IF DSA31ArmSpeedProfileCall.bCallCompleted THEN
DSA31ArmSpeedProfileCall.bCallPB := FALSE;
DSfbGnrProductRecipeMemoryOut.DSGnrCalledArmPnpParameter.DSA1DownTransferMovement.lrZone2SpeedVelo := DSA31ArmSpeedProfileCall.Call_DSArmSpdProfile.lrSpeedVelo;
DSfbGnrProductRecipeMemoryOut.DSGnrCalledArmPnpParameter.DSA1DownTransferMovement.lrZone2Acc := DSA31ArmSpeedProfileCall.Call_DSArmSpdProfile.lrAcc;
DSfbGnrProductRecipeMemoryOut.DSGnrCalledArmPnpParameter.DSA1DownTransferMovement.lrZone2Dcc := DSA31ArmSpeedProfileCall.Call_DSArmSpdProfile.lrDcc;

DSfbGnrProductRecipeMemoryOut.iCallCaseNo:=43;
END_IF

IF rebInvalidSpeedProfileMemoryCall.Q THEN
DSA31ArmSpeedProfileCall.bCallPB := FALSE;

DSfbGnrProductRecipeMemoryOut.iCallCaseNo:=82;
END_IF


41: (* Push DownTransfer Zone1  Velo/Acc/Dcc to DownTransfer Movement*)

DSA31ArmSpeedProfileCall.Call_iArmSpdProfile := DSBufferDownTransferPattern.iZone1SpdProfileNo;
DSA31ArmSpeedProfileCall.bCallPB := TRUE;


IF DSA31ArmSpeedProfileCall.bCallCompleted THEN
DSA31ArmSpeedProfileCall.bCallPB := FALSE;
DSfbGnrProductRecipeMemoryOut.DSGnrCalledArmPnpParameter.DSA1DownTransferMovement.lrZone1SpeedVelo := DSA31ArmSpeedProfileCall.Call_DSArmSpdProfile.lrSpeedVelo;
DSfbGnrProductRecipeMemoryOut.DSGnrCalledArmPnpParameter.DSA1DownTransferMovement.lrZone1Acc := DSA31ArmSpeedProfileCall.Call_DSArmSpdProfile.lrAcc;
DSfbGnrProductRecipeMemoryOut.DSGnrCalledArmPnpParameter.DSA1DownTransferMovement.lrZone1Dcc := DSA31ArmSpeedProfileCall.Call_DSArmSpdProfile.lrDcc;

DSfbGnrProductRecipeMemoryOut.iCallCaseNo:=42;
END_IF

IF rebInvalidSpeedProfileMemoryCall.Q THEN
DSA31ArmSpeedProfileCall.bCallPB := FALSE;

DSfbGnrProductRecipeMemoryOut.iCallCaseNo:=82;
END_IF

(*[][][][][][][][][][][][][][][][][][][][][][][][][][][][][][][][][][][][][][][][][][][][][][][][][][][][][][][][][][][][][][][][][][][][][][][][][][][][][][][][][][][][][][][][][][][][][][][][][][][]*)

(*[][][][][][][][][][][][][][][][][][][][][][][][][][][][][][][][][][][][][][][][][][][][][][][][][][][][][][][][][][][][][][][][][][][][][][][][][][][][][][][][][][][][][][][][][][][][][][][][][][][]*)
34: (* Push UpPick Zone4  Velo/Acc/Dcc to UpPick Movement*)

DSA31ArmSpeedProfileCall.Call_iArmSpdProfile := DSBufferUpPickPattern.iZone4SpdProfileNo;
DSA31ArmSpeedProfileCall.bCallPB := TRUE;


IF DSA31ArmSpeedProfileCall.bCallCompleted THEN
DSA31ArmSpeedProfileCall.bCallPB := FALSE;
DSfbGnrProductRecipeMemoryOut.DSGnrCalledArmPnpParameter.DSA1UpPickMovement.lrZone4SpeedVelo := DSA31ArmSpeedProfileCall.Call_DSArmSpdProfile.lrSpeedVelo;
DSfbGnrProductRecipeMemoryOut.DSGnrCalledArmPnpParameter.DSA1UpPickMovement.lrZone4Acc := DSA31ArmSpeedProfileCall.Call_DSArmSpdProfile.lrAcc;
DSfbGnrProductRecipeMemoryOut.DSGnrCalledArmPnpParameter.DSA1UpPickMovement.lrZone4Dcc := DSA31ArmSpeedProfileCall.Call_DSArmSpdProfile.lrDcc;

DSfbGnrProductRecipeMemoryOut.iCallCaseNo:=41;
END_IF

IF rebInvalidSpeedProfileMemoryCall.Q THEN
DSA31ArmSpeedProfileCall.bCallPB := FALSE;

DSfbGnrProductRecipeMemoryOut.iCallCaseNo:=82;
END_IF



33: (* Push UpPick Zone3  Velo/Acc/Dcc to UpPick Movement*)

DSA31ArmSpeedProfileCall.Call_iArmSpdProfile := DSBufferUpPickPattern.iZone3SpdProfileNo;
DSA31ArmSpeedProfileCall.bCallPB := TRUE;


IF DSA31ArmSpeedProfileCall.bCallCompleted THEN
DSA31ArmSpeedProfileCall.bCallPB := FALSE;
DSfbGnrProductRecipeMemoryOut.DSGnrCalledArmPnpParameter.DSA1UpPickMovement.lrZone3SpeedVelo := DSA31ArmSpeedProfileCall.Call_DSArmSpdProfile.lrSpeedVelo;
DSfbGnrProductRecipeMemoryOut.DSGnrCalledArmPnpParameter.DSA1UpPickMovement.lrZone3Acc := DSA31ArmSpeedProfileCall.Call_DSArmSpdProfile.lrAcc;
DSfbGnrProductRecipeMemoryOut.DSGnrCalledArmPnpParameter.DSA1UpPickMovement.lrZone3Dcc := DSA31ArmSpeedProfileCall.Call_DSArmSpdProfile.lrDcc;

DSfbGnrProductRecipeMemoryOut.iCallCaseNo:=34;
END_IF

IF rebInvalidSpeedProfileMemoryCall.Q THEN
DSA31ArmSpeedProfileCall.bCallPB := FALSE;

DSfbGnrProductRecipeMemoryOut.iCallCaseNo:=82;
END_IF



32: (* Push UpPick Zone2  Velo/Acc/Dcc to UpPick Movement*)

DSA31ArmSpeedProfileCall.Call_iArmSpdProfile := DSBufferUpPickPattern.iZone2SpdProfileNo;
DSA31ArmSpeedProfileCall.bCallPB := TRUE;


IF DSA31ArmSpeedProfileCall.bCallCompleted THEN
DSA31ArmSpeedProfileCall.bCallPB := FALSE;
DSfbGnrProductRecipeMemoryOut.DSGnrCalledArmPnpParameter.DSA1UpPickMovement.lrZone2SpeedVelo := DSA31ArmSpeedProfileCall.Call_DSArmSpdProfile.lrSpeedVelo;
DSfbGnrProductRecipeMemoryOut.DSGnrCalledArmPnpParameter.DSA1UpPickMovement.lrZone2Acc := DSA31ArmSpeedProfileCall.Call_DSArmSpdProfile.lrAcc;
DSfbGnrProductRecipeMemoryOut.DSGnrCalledArmPnpParameter.DSA1UpPickMovement.lrZone2Dcc := DSA31ArmSpeedProfileCall.Call_DSArmSpdProfile.lrDcc;

DSfbGnrProductRecipeMemoryOut.iCallCaseNo:=33;
END_IF

IF rebInvalidSpeedProfileMemoryCall.Q THEN
DSA31ArmSpeedProfileCall.bCallPB := FALSE;

DSfbGnrProductRecipeMemoryOut.iCallCaseNo:=82;
END_IF


31: (* Push UpPick Zone1  Velo/Acc/Dcc to UpPick Movement*)

DSA31ArmSpeedProfileCall.Call_iArmSpdProfile := DSBufferUpPickPattern.iZone1SpdProfileNo;
DSA31ArmSpeedProfileCall.bCallPB := TRUE;


IF DSA31ArmSpeedProfileCall.bCallCompleted THEN
DSA31ArmSpeedProfileCall.bCallPB := FALSE;
DSfbGnrProductRecipeMemoryOut.DSGnrCalledArmPnpParameter.DSA1UpPickMovement.lrZone1SpeedVelo := DSA31ArmSpeedProfileCall.Call_DSArmSpdProfile.lrSpeedVelo;
DSfbGnrProductRecipeMemoryOut.DSGnrCalledArmPnpParameter.DSA1UpPickMovement.lrZone1Acc := DSA31ArmSpeedProfileCall.Call_DSArmSpdProfile.lrAcc;
DSfbGnrProductRecipeMemoryOut.DSGnrCalledArmPnpParameter.DSA1UpPickMovement.lrZone1Dcc := DSA31ArmSpeedProfileCall.Call_DSArmSpdProfile.lrDcc;

DSfbGnrProductRecipeMemoryOut.iCallCaseNo:=32;
END_IF

IF rebInvalidSpeedProfileMemoryCall.Q THEN
DSA31ArmSpeedProfileCall.bCallPB := FALSE;

DSfbGnrProductRecipeMemoryOut.iCallCaseNo:=82;
END_IF

(*[][][][][][][][][][][][][][][][][][][][][][][][][][][][][][][][][][][][][][][][][][][][][][][][][][][][][][][][][][][][][][][][][][][][][][][][][][][][][][][][][][][][][][][][][][][][][][][][][][][]*)


(*[][][][][][][][][][][][][][][][][][][][][][][][][][][][][][][][][][][][][][][][][][][][][][][][][][][][][][][][][][][][][][][][][][][][][][][][][][][][][][][][][][][][][][][][][][][][][][][][][][][]*)
24: (* Push DownPick Zone4  Velo/Acc/Dcc to DownPick Movement*)

DSA31ArmSpeedProfileCall.Call_iArmSpdProfile := DSBufferDownPickPattern.iZone4SpdProfileNo;
DSA31ArmSpeedProfileCall.bCallPB := TRUE;


IF DSA31ArmSpeedProfileCall.bCallCompleted THEN
DSA31ArmSpeedProfileCall.bCallPB := FALSE;
DSfbGnrProductRecipeMemoryOut.DSGnrCalledArmPnpParameter.DSA1DownPickMovement.lrZone4SpeedVelo := DSA31ArmSpeedProfileCall.Call_DSArmSpdProfile.lrSpeedVelo;
DSfbGnrProductRecipeMemoryOut.DSGnrCalledArmPnpParameter.DSA1DownPickMovement.lrZone4Acc := DSA31ArmSpeedProfileCall.Call_DSArmSpdProfile.lrAcc;
DSfbGnrProductRecipeMemoryOut.DSGnrCalledArmPnpParameter.DSA1DownPickMovement.lrZone4Dcc := DSA31ArmSpeedProfileCall.Call_DSArmSpdProfile.lrDcc;

DSfbGnrProductRecipeMemoryOut.iCallCaseNo:=31;
END_IF

IF rebInvalidSpeedProfileMemoryCall.Q THEN
DSA31ArmSpeedProfileCall.bCallPB := FALSE;

DSfbGnrProductRecipeMemoryOut.iCallCaseNo:=82;
END_IF



23: (* Push DownPick Zone3  Velo/Acc/Dcc to DownPick Movement*)

DSA31ArmSpeedProfileCall.Call_iArmSpdProfile := DSBufferDownPickPattern.iZone3SpdProfileNo;
DSA31ArmSpeedProfileCall.bCallPB := TRUE;


IF DSA31ArmSpeedProfileCall.bCallCompleted THEN
DSA31ArmSpeedProfileCall.bCallPB := FALSE;
DSfbGnrProductRecipeMemoryOut.DSGnrCalledArmPnpParameter.DSA1DownPickMovement.lrZone3SpeedVelo := DSA31ArmSpeedProfileCall.Call_DSArmSpdProfile.lrSpeedVelo;
DSfbGnrProductRecipeMemoryOut.DSGnrCalledArmPnpParameter.DSA1DownPickMovement.lrZone3Acc := DSA31ArmSpeedProfileCall.Call_DSArmSpdProfile.lrAcc;
DSfbGnrProductRecipeMemoryOut.DSGnrCalledArmPnpParameter.DSA1DownPickMovement.lrZone3Dcc := DSA31ArmSpeedProfileCall.Call_DSArmSpdProfile.lrDcc;

DSfbGnrProductRecipeMemoryOut.iCallCaseNo:=24;
END_IF

IF rebInvalidSpeedProfileMemoryCall.Q THEN
DSA31ArmSpeedProfileCall.bCallPB := FALSE;

DSfbGnrProductRecipeMemoryOut.iCallCaseNo:=82;
END_IF



22: (* Push DownPick Zone2  Velo/Acc/Dcc to DownPick Movement*)

DSA31ArmSpeedProfileCall.Call_iArmSpdProfile := DSBufferDownPickPattern.iZone2SpdProfileNo;
DSA31ArmSpeedProfileCall.bCallPB := TRUE;


IF DSA31ArmSpeedProfileCall.bCallCompleted THEN
DSA31ArmSpeedProfileCall.bCallPB := FALSE;
DSfbGnrProductRecipeMemoryOut.DSGnrCalledArmPnpParameter.DSA1DownPickMovement.lrZone2SpeedVelo := DSA31ArmSpeedProfileCall.Call_DSArmSpdProfile.lrSpeedVelo;
DSfbGnrProductRecipeMemoryOut.DSGnrCalledArmPnpParameter.DSA1DownPickMovement.lrZone2Acc := DSA31ArmSpeedProfileCall.Call_DSArmSpdProfile.lrAcc;
DSfbGnrProductRecipeMemoryOut.DSGnrCalledArmPnpParameter.DSA1DownPickMovement.lrZone2Dcc := DSA31ArmSpeedProfileCall.Call_DSArmSpdProfile.lrDcc;

DSfbGnrProductRecipeMemoryOut.iCallCaseNo:=23;
END_IF

IF rebInvalidSpeedProfileMemoryCall.Q THEN
DSA31ArmSpeedProfileCall.bCallPB := FALSE;

DSfbGnrProductRecipeMemoryOut.iCallCaseNo:=82;
END_IF


21: (* Push DownPick Zone1  Velo/Acc/Dcc to DownPick Movement*)

DSA31ArmSpeedProfileCall.Call_iArmSpdProfile := DSBufferDownPickPattern.iZone1SpdProfileNo;
DSA31ArmSpeedProfileCall.bCallPB := TRUE;


IF DSA31ArmSpeedProfileCall.bCallCompleted THEN
DSA31ArmSpeedProfileCall.bCallPB := FALSE;
DSfbGnrProductRecipeMemoryOut.DSGnrCalledArmPnpParameter.DSA1DownPickMovement.lrZone1SpeedVelo := DSA31ArmSpeedProfileCall.Call_DSArmSpdProfile.lrSpeedVelo;
DSfbGnrProductRecipeMemoryOut.DSGnrCalledArmPnpParameter.DSA1DownPickMovement.lrZone1Acc := DSA31ArmSpeedProfileCall.Call_DSArmSpdProfile.lrAcc;
DSfbGnrProductRecipeMemoryOut.DSGnrCalledArmPnpParameter.DSA1DownPickMovement.lrZone1Dcc := DSA31ArmSpeedProfileCall.Call_DSArmSpdProfile.lrDcc;

DSfbGnrProductRecipeMemoryOut.iCallCaseNo:=22;
END_IF

IF rebInvalidSpeedProfileMemoryCall.Q THEN
DSA31ArmSpeedProfileCall.bCallPB := FALSE;

DSfbGnrProductRecipeMemoryOut.iCallCaseNo:=82;
END_IF

(*[][][][][][][][][][][][][][][][][][][][][][][][][][][][][][][][][][][][][][][][][][][][][][][][][][][][][][][][][][][][][][][][][][][][][][][][][][][][][][][][][][][][][][][][][][][][][][][][][][][]*)



14: (* Call UpPickPattern*)
DSA21UpDownPatternCall.Call_iUpDownPatternNo := DSA1fbPnpSequenceMemoryCall.Call_DsPnpSequenceMemory.ARiUpTransferPatternNo[iProductRecipeStepCall];
DSA21UpDownPatternCall.bCallPB := TRUE;


IF DSA21UpDownPatternCall.bCallCompleted THEN
DSA21UpDownPatternCall.bCallPB := FALSE;
DSBufferUpTransferPattern := DSA21UpDownPatternCall.Call_DsUpDownPattern;
DSfbGnrProductRecipeMemoryOut.DSGnrCalledArmPnpParameter.DSA1UpTransferMovement.sUpDownPatternDescription := DSA21UpDownPatternCall.Call_DsUpDownPattern.sDescription;
DSfbGnrProductRecipeMemoryOut.iCallCaseNo:=21;
END_IF

13: (* Call DownTransferPattern*)
DSA21UpDownPatternCall.Call_iUpDownPatternNo := DSA1fbPnpSequenceMemoryCall.Call_DsPnpSequenceMemory.ARiDownTransferPatternNo[iProductRecipeStepCall];
DSA21UpDownPatternCall.bCallPB := TRUE;


IF DSA21UpDownPatternCall.bCallCompleted THEN
DSA21UpDownPatternCall.bCallPB := FALSE;
DSBufferDownTransferPattern := DSA21UpDownPatternCall.Call_DsUpDownPattern;
DSfbGnrProductRecipeMemoryOut.DSGnrCalledArmPnpParameter.DSA1DownTransferMovement.sUpDownPatternDescription := DSA21UpDownPatternCall.Call_DsUpDownPattern.sDescription;
DSfbGnrProductRecipeMemoryOut.iCallCaseNo:=14;
END_IF

IF rebInvalidUpDownPatternMemoryCall.Q THEN
DSA21UpDownPatternCall.bCallPB := FALSE;

DSfbGnrProductRecipeMemoryOut.iCallCaseNo:=81;
END_IF

12: (* Call UpPickPattern*)
DSA21UpDownPatternCall.Call_iUpDownPatternNo := DSA1fbPnpSequenceMemoryCall.Call_DsPnpSequenceMemory.ARiUpPickPatternNo[iProductRecipeStepCall];
DSA21UpDownPatternCall.bCallPB := TRUE;


IF DSA21UpDownPatternCall.bCallCompleted THEN
DSA21UpDownPatternCall.bCallPB := FALSE;
DSBufferUpPickPattern := DSA21UpDownPatternCall.Call_DsUpDownPattern;
DSfbGnrProductRecipeMemoryOut.DSGnrCalledArmPnpParameter.DSA1UpPickMovement.sUpDownPatternDescription := DSA21UpDownPatternCall.Call_DsUpDownPattern.sDescription;
DSfbGnrProductRecipeMemoryOut.iCallCaseNo:=13;
END_IF

IF rebInvalidUpDownPatternMemoryCall.Q THEN
DSA21UpDownPatternCall.bCallPB := FALSE;

DSfbGnrProductRecipeMemoryOut.iCallCaseNo:=81;
END_IF

11: (* Call DownPickPattern*)
DSA21UpDownPatternCall.Call_iUpDownPatternNo := DSA1fbPnpSequenceMemoryCall.Call_DsPnpSequenceMemory.ARiDownPickPatternNo[iProductRecipeStepCall];
DSA21UpDownPatternCall.bCallPB := TRUE;


IF DSA21UpDownPatternCall.bCallCompleted THEN
DSA21UpDownPatternCall.bCallPB := FALSE;
DSBufferDownPickPattern := DSA21UpDownPatternCall.Call_DsUpDownPattern;
DSfbGnrProductRecipeMemoryOut.DSGnrCalledArmPnpParameter.DSA1DownPickMovement.sUpDownPatternDescription := DSA21UpDownPatternCall.Call_DsUpDownPattern.sDescription;
DSfbGnrProductRecipeMemoryOut.iCallCaseNo:=12;
END_IF

IF rebInvalidUpDownPatternMemoryCall.Q THEN
DSA21UpDownPatternCall.bCallPB := FALSE;

DSfbGnrProductRecipeMemoryOut.iCallCaseNo:=81;
END_IF


10: (*Push UpDownPattern to Buffer*)
iBufferPickStationNo := DSA1fbPnpSequenceMemoryCall.Call_DsPnpSequenceMemory.ARiPickStationNo[iProductRecipeStepCall];
iBufferTransferStationNo := DSA1fbPnpSequenceMemoryCall.Call_DsPnpSequenceMemory.ARiTransferStationNo[iProductRecipeStepCall];

iBufferDownPickPatternNo := DSA1fbPnpSequenceMemoryCall.Call_DsPnpSequenceMemory.ARiDownPickPatternNo[iProductRecipeStepCall];
iBufferUpPickPatternNo := DSA1fbPnpSequenceMemoryCall.Call_DsPnpSequenceMemory.ARiUpPickPatternNo[iProductRecipeStepCall];
iBufferDownTransferPatternNo := DSA1fbPnpSequenceMemoryCall.Call_DsPnpSequenceMemory.ARiDownTransferPatternNo[iProductRecipeStepCall];
iBufferUpTransferPatternNo := DSA1fbPnpSequenceMemoryCall.Call_DsPnpSequenceMemory.ARiUpTransferPatternNo[iProductRecipeStepCall];

DSfbGnrProductRecipeMemoryOut.DSGnrCalledArmPnpParameter.iStnSeqRecipeNo := DSA1fbPnpSequenceMemoryCall.Call_DsPnpSequenceMemory.ARiStnSeqRepNo[iProductRecipeStepCall];

DSfbGnrProductRecipeMemoryOut.sProductRecipeDescription := DSA1fbPnpSequenceMemoryCall.Call_DsPnpSequenceMemory.sDescription;

DSfbGnrProductRecipeMemoryOut.iCallCaseNo:=11;


71: (*Complete Data Called*)

	IF bEnableCallArmNo THEN
	DSfbGnrProductRecipeMemoryOut.DSGnrCalledArmPnpParameter.iCallArmNo := iCallArmNo;
	ELSE
	DSfbGnrProductRecipeMemoryOut.DSGnrCalledArmPnpParameter.iCallArmNo := DSA1fbPnpSequenceMemoryCall.Call_DsPnpSequenceMemory.ARiCallArmNo[iProductRecipeStepCall];
	END_IF

DSfbGnrProductRecipeMemoryOut.bCallCompleted := TRUE;
CallSelfCheckHR := FALSE;
DSfbGnrProductRecipeMemoryOut.iCallCaseNo:=72;

72:; (*Done without error*)

81:
(*iPreviousProcessStep := iCurrentProcessStep;*)
CallSelfCheckHR := FALSE;
DSfbGnrProductRecipeMemoryOut.bCallUpDownPatternMemoryErr := TRUE;
DSfbGnrProductRecipeMemoryOut.iCallCaseNo:=91;

82:
(*iPreviousProcessStep := iCurrentProcessStep;*)
DSfbGnrProductRecipeMemoryOut.bCallArmSpeedProfileMemoryErr := TRUE;
CallSelfCheckHR := FALSE;
DSfbGnrProductRecipeMemoryOut.iCallCaseNo:=92;

83:
(*iPreviousProcessStep := iCurrentProcessStep;*)
DSfbGnrProductRecipeMemoryOut.bCallPickStationNoErr := TRUE;
CallSelfCheckHR := FALSE;
DSfbGnrProductRecipeMemoryOut.iCallCaseNo:=93;

84:
(*iPreviousProcessStep := iCurrentProcessStep;*)
DSfbGnrProductRecipeMemoryOut.bCallTransferStationNoErr := TRUE;
CallSelfCheckHR := FALSE;
DSfbGnrProductRecipeMemoryOut.iCallCaseNo:=94;



91:; (*Found UpDownPatternMemoryError and Task Not Complete *)

92:; (*Found ArmSpeedProfileMemoryErr and Task Not Complete *)

93:; (*Found PickStationNoErr and Task Not Complete *)

94:; (*Found TransferStationNoErr and Task Not Complete *)



END_CASE

END_FUNCTION_BLOCK

// ---- FBs/B_JKS_NewFB/FBP-Memory_Sub/fbA1_PnpSequenceMemory.TcPOU
FUNCTION_BLOCK fbA1_PnpSequenceMemory

VAR CONSTANT
END_VAR

VAR_INPUT
	bSavePB : BOOL;
	bLoadPB : BOOL;
	bCopyPB : BOOL;
	iCopyToProductRecipeNo : INT;
(*	iLdStnID: INT;
	iUldStnID: INT;
*)END_VAR


VAR_IN_OUT PERSISTENT

	iProductRecipeNo: INT; (* 10 sets of UpDownPattern *)
	DSA1inPnpSequenceMemory : DSA1_PnpSequenceMemory;

	Call_iProductRecipeNo : INT;
	bCallPB: BOOL;

END_VAR
VAR_OUTPUT
	bSaveInd: BOOL;
	bLoadInd: BOOL;
	bCallCompleted : BOOL;
	bInvalidCallProductRecipeNoHold: BOOL;
	bInvalidCallProductRecipeNoPulse: BOOL;
	Call_DSA1PnpSequenceMemory : DSA1_PnpSequenceMemory;

END_VAR
VAR
	SaveIndHr: BOOL;
	LoadIndHr: BOOL;

	SaveTimerDelay: TON;
	LoadTimerDelay: TON;
	SelfCheckTimer: TON;
	bLoadEn: BOOL;
	SelfCheckloopPnpSequence: BOOL;

	LoadDF : R_TRIG;
	LoadENDF : R_TRIG;

	SaveDF: R_TRIG;
	CallIntervalTimer: TON;
	CallIntervalDIFU: R_TRIG;

	bCallCompletedHR: BOOL;
	bCallCompletedHRRE: R_TRIG;
	CallCompletedTimer: TON;
	CallSelfCheckTimer : TON;
	CallSelfCheckloop : BOOL;

	CallSelfCheckRE: R_TRIG;
	CallStep: INT;
	CallSelfCheckHR: BOOL;
	bCallPBRE: R_TRIG;

	LoadFL: INT;
	SaveFL: INT;
	CallSFL: INT;
	febInvalidCallProductRecipeNo: F_TRIG;



	rebInvalidCallProductRecipeNo: R_TRIG;
	CopyDF: R_TRIG;
	PreviousProductRecipeNo: INT;
	PreviousProductRecipeCallNo: INT;
	tInvalidCallProductRecipeNoPulseTimer: TON;
	iFixPickStnFL: INT;
	iCtrlTransferStnFL: INT;
	bTransferStnEndDetected: BOOL;
	iUldStnStepNo: INT;
	iCtrlZeroB4UldStnFL: INT;
	iMaxMinFL: INT;
	iWriteEmptyDesFL: INT;
END_VAR

VAR PERSISTENT

	ARDsPnpSequenceMemory : ARRAY [1..iProductRecipeArrayQty] OF DSA1_PnpSequenceMemory;
	ARsStoragePnpSequenceDescription: ARRAY [0..iProductRecipeArrayQty] OF STRING(50);


END_VAR

IF iProductRecipeNo < 1 THEN
iProductRecipeNo := 1;
END_IF

IF iProductRecipeNo > iProductRecipeArrayQty THEN
iProductRecipeNo := iProductRecipeArrayQty;
END_IF

(*Fix Pick Station No*)
DSA1inPnpSequenceMemory.ARiPickStationNo[1] := iLdStnID;
iFixPickStnFL := 1;

	FOR iFixPickStnFL := 1 TO iProductRecipeStepArrayQty DO

		IF iFixPickStnFL >=1 AND iFixPickStnFL <= iProductRecipeStepArrayQty-1THEN

			IF DSA1inPnpSequenceMemory.ARiTransferStationNo[iFixPickStnFL] <> iUldStnID THEN
			DSA1inPnpSequenceMemory.ARiPickStationNo[iFixPickStnFL+1]:= DSA1inPnpSequenceMemory.ARiTransferStationNo[iFixPickStnFL];
			END_IF

			IF DSA1inPnpSequenceMemory.ARiTransferStationNo[iFixPickStnFL] = iUldStnID THEN
			DSA1inPnpSequenceMemory.ARiPickStationNo[iFixPickStnFL+1]:= 0;
			END_IF

		END_IF

	END_FOR

(*Control Transfer Station No*)
iCtrlTransferStnFL := 1;
bTransferStnEndDetected := FALSE;
iUldStnStepNo := 0;
	FOR iCtrlTransferStnFL := 1 TO iProductRecipeStepArrayQty DO

		IF iCtrlTransferStnFL >=1 AND iCtrlTransferStnFL <= iProductRecipeStepArrayQty THEN

			IF NOT bTransferStnEndDetected AND DSA1inPnpSequenceMemory.ARiTransferStationNo[iCtrlTransferStnFL] > iStnQty THEN
			DSA1inPnpSequenceMemory.ARiTransferStationNo[iCtrlTransferStnFL]:= iUldStnID;
			END_IF

			IF bTransferStnEndDetected THEN
			DSA1inPnpSequenceMemory.ARiTransferStationNo[iCtrlTransferStnFL] := iUldStnID(*0*);
			END_IF

			IF DSA1inPnpSequenceMemory.ARiTransferStationNo[iCtrlTransferStnFL-1] = iUldStnID THEN
			DSA1inPnpSequenceMemory.ARiTransferStationNo[iCtrlTransferStnFL] := iUldStnID(*0*);
			bTransferStnEndDetected := TRUE;
			iUldStnStepNo := iCtrlTransferStnFL-1;
			END_IF

		END_IF

	END_FOR

(*No "0" before Unloading Stn Ctrl*)

IF bTransferStnEndDetected AND iUldStnStepNo > 1 THEN
iCtrlZeroB4UldStnFL := 1;

	FOR iCtrlZeroB4UldStnFL := 1 TO iUldStnStepNo DO

		IF iCtrlZeroB4UldStnFL >=1 AND iCtrlZeroB4UldStnFL <= iUldStnStepNo-1 THEN

			IF DSA1inPnpSequenceMemory.ARiTransferStationNo[iCtrlZeroB4UldStnFL] <= 0 THEN
			DSA1inPnpSequenceMemory.ARiTransferStationNo[iCtrlZeroB4UldStnFL]:= 1;
			END_IF

		END_IF

	END_FOR

END_IF


(*Min / Max Control*)
iMaxMinFL := 1;
	FOR iMaxMinFL := 1 TO iProductRecipeStepArrayQty DO

		IF iMaxMinFL >=1 AND iMaxMinFL <= iProductRecipeStepArrayQty THEN

			IF DSA1inPnpSequenceMemory.ARiDownPickPatternNo[iMaxMinFL] <= 0 THEN
			DSA1inPnpSequenceMemory.ARiDownPickPatternNo[iMaxMinFL]:= 1;
			ELSIF DSA1inPnpSequenceMemory.ARiDownPickPatternNo[iMaxMinFL] > iArmUpDownPatternArrayQty THEN
			DSA1inPnpSequenceMemory.ARiDownPickPatternNo[iMaxMinFL]:= iArmUpDownPatternArrayQty;
			END_IF

			IF DSA1inPnpSequenceMemory.ARiUpPickPatternNo[iMaxMinFL] <= 0 THEN
			DSA1inPnpSequenceMemory.ARiUpPickPatternNo[iMaxMinFL]:= 1;
			ELSIF DSA1inPnpSequenceMemory.ARiUpPickPatternNo[iMaxMinFL] > iArmUpDownPatternArrayQty THEN
			DSA1inPnpSequenceMemory.ARiUpPickPatternNo[iMaxMinFL]:= iArmUpDownPatternArrayQty;
			END_IF

			IF DSA1inPnpSequenceMemory.ARiDownTransferPatternNo[iMaxMinFL] <= 0 THEN
			DSA1inPnpSequenceMemory.ARiDownTransferPatternNo[iMaxMinFL]:= 1;
			ELSIF DSA1inPnpSequenceMemory.ARiDownTransferPatternNo[iMaxMinFL] > iArmUpDownPatternArrayQty THEN
			DSA1inPnpSequenceMemory.ARiDownTransferPatternNo[iMaxMinFL]:= iArmUpDownPatternArrayQty;
			END_IF

			IF DSA1inPnpSequenceMemory.ARiUpTransferPatternNo[iMaxMinFL] <= 0 THEN
			DSA1inPnpSequenceMemory.ARiUpTransferPatternNo[iMaxMinFL]:= 1;
			ELSIF DSA1inPnpSequenceMemory.ARiUpTransferPatternNo[iMaxMinFL] > iArmUpDownPatternArrayQty THEN
			DSA1inPnpSequenceMemory.ARiUpTransferPatternNo[iMaxMinFL]:= iArmUpDownPatternArrayQty;
			END_IF

(*			IF DSA1inPnpSequenceMemory.ARiRepeatUpDownCycle[iMaxMinFL] <= 0 THEN
			DSA1inPnpSequenceMemory.ARiRepeatUpDownCycle[iMaxMinFL]:= 1;
			ELS*)IF DSA1inPnpSequenceMemory.ARiRepeatUpDownCycle[iMaxMinFL] > 99 THEN
			DSA1inPnpSequenceMemory.ARiRepeatUpDownCycle[iMaxMinFL]:= 99;
			END_IF

			IF DSA1inPnpSequenceMemory.ARiCallArmNo[iMaxMinFL] <= 0 THEN
			DSA1inPnpSequenceMemory.ARiCallArmNo[iMaxMinFL]:= 1;
			ELSIF DSA1inPnpSequenceMemory.ARiCallArmNo[iMaxMinFL] > iArmQty THEN
			DSA1inPnpSequenceMemory.ARiCallArmNo[iMaxMinFL]:= iArmQty;
			END_IF

			IF DSA1inPnpSequenceMemory.ARiStnSeqRepNo[iMaxMinFL] <= 0 THEN
			DSA1inPnpSequenceMemory.ARiStnSeqRepNo[iMaxMinFL]:= 1;
			ELSIF DSA1inPnpSequenceMemory.ARiStnSeqRepNo[iMaxMinFL] > iStationSequenceRecipeArrayQty THEN
			DSA1inPnpSequenceMemory.ARiStnSeqRepNo[iMaxMinFL]:= iStationSequenceRecipeArrayQty;
			END_IF

		END_IF

	END_FOR


(*Load and Save Indicator*)
IF bSavePB THEN
SaveIndHr := TRUE;
END_IF

SaveTimerDelay(IN:=SaveIndHr, PT := T#1s, Q=>, ET=>);
IF SaveTimerDelay.Q THEN
SaveIndHr := FALSE;
END_IF

IF SaveIndHr AND NOT SaveTimerDelay.Q THEN
bSaveInd := TRUE;
ELSE
bSaveInd := FALSE;
END_IF

IF bLoadPB THEN
LoadIndHr := TRUE;
END_IF

LoadTimerDelay(IN:=LoadIndHr, PT := T#1s, Q=>, ET=>);
IF loadtimerdelay.Q THEN
LoadIndHr := FALSE;
END_IF

IF loadIndHr AND NOT LoadTimerDelay.Q THEN
bLoadInd := TRUE;
ELSE
bLoadInd := FALSE;
END_IF

IF iProductRecipeNo <> PreviousProductRecipeNo THEN
bLoadEn := TRUE;
ELSE
bLoadEn := FALSE;
END_IF


(* Load Recipe *)

LoadDF(CLK:=bLoadPB,Q=>);
LoadENDF(CLK:=bLoadEn,Q=>);

IF LoadDF.Q OR LoadENDF.Q THEN

DSA1inPnpSequenceMemory := ARDsPnpSequenceMemory[iProductRecipeNo];
PreviousProductRecipeNo := iProductRecipeNo  ;

END_IF


(* Save Recipe *)

SaveDF(CLK:=bSavePB,Q=>);

IF SaveDF.Q THEN

ARDsPnpSequenceMemory[iProductRecipeNo] := DSA1inPnpSequenceMemory;
ARsStoragePnpSequenceDescription[iProductRecipeNo] := DSA1inPnpSequenceMemory.sDescription;

END_IF


(*Copy Recipe*)

CopyDF(CLK:=bCopyPB,Q=>);

IF CopyDF.Q THEN

ARDsPnpSequenceMemory[iCopyToProductRecipeNo] := ARDsPnpSequenceMemory[iProductRecipeNo];
ARsStoragePnpSequenceDescription[iCopyToProductRecipeNo] := ARDsPnpSequenceMemory[iProductRecipeNo].sDescription;

END_IF

(*Write Empty for Empty description *)
ARsStoragePnpSequenceDescription[0] := ' = = = No Basket = = = ';
iWriteEmptyDesFL := 1;
FOR iWriteEmptyDesFL := 1 TO iProductRecipeArrayQty DO
	IF iWriteEmptyDesFL >= 1 AND iWriteEmptyDesFL <= iProductRecipeArrayQty THEN
		IF ARsStoragePnpSequenceDescription[iWriteEmptyDesFL] = '' THEN
		ARsStoragePnpSequenceDescription[iWriteEmptyDesFL] := ' - - -  Empty Recipe - - - ';
		END_IF
	END_IF
END_FOR




(* Call Recipe *)
(* ---- Call Recipe Complete Flag ---*)


IF NOT bCallPB THEN
bCallCompleted := FALSE;
END_IF

bCallPBRE(CLK:=bCallPB , Q=> );

IF (Call_iProductRecipeNo <= 0 OR Call_iProductRecipeNo > iProductRecipeArrayQty) AND bCallPB THEN
bInvalidCallProductRecipeNoHold := TRUE;
ELSE
bInvalidCallProductRecipeNoHold := FALSE;
END_IF


febInvalidCallProductRecipeNo(CLK:= bCallPB AND bInvalidCallProductRecipeNoHold  , Q=> );

IF febInvalidCallProductRecipeNo.Q THEN
bInvalidCallProductRecipeNoPulse := TRUE;
END_IF

tInvalidCallProductRecipeNoPulseTimer(IN:=bInvalidCallProductRecipeNoPulse , PT:=t#0.5s , Q=> , ET=> );

IF tInvalidCallProductRecipeNoPulseTimer.Q OR NOT bCallPB THEN
bInvalidCallProductRecipeNoPulse := FALSE;
END_IF

IF bCallPBRE.Q AND NOT bInvalidCallProductRecipeNoHold THEN
bCallCompleted := FALSE;
CallStep:= 1;
END_IF


CASE CallStep OF

1:

Call_DSA1PnpSequenceMemory := ARDsPnpSequenceMemory[Call_iProductRecipeNo];

CallStep := 11;


10:
bCallCompleted := TRUE;
CallSelfCheckHR := FALSE;
PreviousProductRecipeCallNo := Call_iProductRecipeNo;
CallStep := 99;

11:

bCallCompleted := TRUE;
CallStep := 99;



99:
;
END_CASE

END_FUNCTION_BLOCK

// ---- FBs/B_JKS_NewFB/FBP-Memory_Sub/fbA32_MachineZoneHeight.TcPOU
FUNCTION_BLOCK fbA32_MachineZoneHeight

VAR_IN_OUT PERSISTENT

	DSLdZoneHeight : DSA32_StationZoneHeight;
	ARDSStationZoneHeight : ARRAY [0..iStnQty] OF DSA32_StationZoneHeight;
	DSUldZoneHeight : DSA32_StationZoneHeight;


END_VAR
VAR_OUTPUT
	DSLdZonePosOut : DSA32_StationZonePosOut;
	ARDSStationZonePosOut : ARRAY [0..iStnQty] OF DSA32_StationZonePosOut;
	DSUldZonePosOut : DSA32_StationZonePosOut;

END_VAR
VAR PERSISTENT

	fbLdStationZoneHeight : fbA32_StationZoneHeight;
	ARfbStationZoneHeight : ARRAY [0..iStnQty] OF fbA32_StationZoneHeight;
	fbUldStationZoneHeight : fbA32_StationZoneHeight;

END_VAR
VAR
	Loop: INT;
END_VAR

(*Loading*)
fbLdStationZoneHeight(DSStationZoneHeight:=DSLdZoneHeight , DSStationZonePosOut=>DSLdZonePosOut );

Loop := 1;
IF Loop >= 1 THEN

	FOR Loop := 1 TO iStnQty DO

		(*Station x20*)
		ARfbStationZoneHeight[Loop](DSStationZoneHeight:=ARDSStationZoneHeight[Loop] , DSStationZonePosOut=>ARDSStationZonePosOut[Loop] );

	END_FOR

END_IF

(*Unloading*)
fbUldStationZoneHeight(DSStationZoneHeight:=DSUldZoneHeight , DSStationZonePosOut=>DSUldZonePosOut );

END_FUNCTION_BLOCK

// ---- POUs/MainProgram/CheckBound/CheckRangeUnsigned.TcPOU
FUNCTION CheckRangeUnsigned : UDINT
VAR_INPUT
	value, lower, upper 	: UDINT;
END_VAR
VAR
END_VAR

IF value<lower THEN
	CheckRangeUnsigned := CheckRangeUnsigned + 1;
	CheckRangeUnsigned := lower;
ELSIF value>upper THEN
	CheckRangeUnsigned := CheckRangeUnsigned + 1;
	CheckRangeUnsigned := upper;
ELSE
	CheckRangeUnsigned := value;
END_IF

END_FUNCTION

// ---- FBs/B_JKS_NewFB_V2/FBP-LdUldCVRelated/fbV2_LdUldCvCtrl.TcPOU
FUNCTION_BLOCK fbV2_LdUldCvCtrl
VAR_INPUT
	bEN : BOOL;
	bIndexPB : BOOL;
	bRapidPB : BOOL;
	bLdCvEnable : BOOL;
	bUldCvEnable : BOOL;
	iLdConveyorNo : INT;
	iUldConveyorNo : INT;
	bTimerBasedRapidIndexEn : BOOL;
	iTimerBasedRapidDelaySV_Mins : INT;

	b1stSensor : BOOL;
	bIndexConfirmSensor : BOOL;
	bEndZoneSensor : BOOL;
	rIndexPBDelayTimeSV_Sec : REAL;
	rRapidPBDelayTimeSV_Sec : REAL;
	rIndexConfirmDelayTimeSV_Sec : REAL;
	rEndZoneDelayTimeSV_Sec : REAL;


END_VAR
VAR_IN_OUT


	AR2sDSLdConfirmBasketInfo : ARRAY [1..iLdStnQty, 1..iCvLdQty] OF DSV2_BasketInfo;
	AR2sDSLdTransferBasketInfo : ARRAY [1..iLdStnQty, 1..iCvLdQty] OF DSV2_BasketInfo;
	AR2sDSUldConfirmBasketInfo : ARRAY [1..iUldStnQty, 1..iCvUldQty] OF DSV2_BasketInfo;
	AR2sDSUldTransferBasketInfo : ARRAY [1..iUldStnQty, 1..iCvUldQty] OF DSV2_BasketInfo;

END_VAR

VAR_OUTPUT
	bConveyorStart : BOOL;
	bLdConveyorIdErrorFlag : BOOL;
	bUldConveyorIdErrorFlag: BOOL;
	tIndexPBDelayTimePV : TIME;
	tRapidPBDelayTimePV : TIME;
	tTimerBasedRapidDelayTimePV : TIME;
	tIndexConfirmDelayTimePV : TIME;
	tEndZoneDelayTimePV : TIME;
	sStatus : STRING;



END_VAR
VAR
	DSEmptyBasketInfo :  DSV2_BasketInfo;

	iStep: INT;

	bENRE: R_TRIG;
	bIndexPBDelayTimerRE: R_TRIG;
	bRapidPBDelayTimerRE: R_TRIG;

	iFL: INT;
	iFL1: INT;


	bIndexPBDelayTimer: TON;
	bRapidPBDelayTimer: TON;
	bIndexConfirmDelayTimer: TON;
	bEndZoneDelayTimer: TON;
	bIndexConfirmDelayTimerRE: R_TRIG;
	bEndZoneDelayTimerRE: R_TRIG;
	iLastTransferBasketAddress: INT;
	bMoveEnable: BOOL;
	bRapidEnable: BOOL;
	b1stBasketConfirmEnable: BOOL;
	bTimerBasedRapidDelayTimer: TON;
	diTimerBasedRapidDelaySV_mSec: DINT;
	bTimerBasedRapidSt: BOOL;
	bTimerBasedRapidDelayTimerRE: R_TRIG;
END_VAR

(*Others*)
IF bLdCvEnable THEN
	IF iLdConveyorNo <= 0 OR iLdConveyorNo > iCvLdQty THEN
		bLdConveyorIdErrorFlag := TRUE;
	ELSE
		bLdConveyorIdErrorFlag := FALSE;
	END_IF
ELSE
		bLdConveyorIdErrorFlag := FALSE;
END_IF


IF bUldCvEnable THEN
	IF iUldConveyorNo <= 0 OR iUldConveyorNo > iCvUldQty THEN
		bUldConveyorIdErrorFlag := TRUE;
	ELSE
		bUldConveyorIdErrorFlag := FALSE;
	END_IF
ELSE
		bUldConveyorIdErrorFlag := FALSE;
END_IF



IF NOT bldConveyorIdErrorFlag AND NOT bUldConveyorIdErrorFlag THEN

AR2sDSLdTransferBasketInfo[iLdConveyorNo, iCvLdQty] := DSEmptyBasketInfo;
AR2sDSUldTransferBasketInfo[iUldConveyorNo, iCvUldQty] := DSEmptyBasketInfo;

END_IF




IF (bLdCvEnable AND NOT bUldCvEnable) AND (sStatus = 'Basket Indexing In Progress...' OR NOT AR2sDSLdConfirmBasketInfo[iLdConveyorNo, iCvLdQty].bAvailibility) AND NOT bLdConveyorIdErrorFlag THEN
bMoveEnable := TRUE;
ELSIF (NOT bLdCvEnable AND bUldCvEnable) AND (sStatus = 'Basket Indexing In Progress...' OR NOT AR2sDSUldConfirmBasketInfo[iUldConveyorNo, iCvUldQty].bAvailibility) AND NOT bUldConveyorIdErrorFlag THEN
bMoveEnable := TRUE;
ELSE
bMoveEnable := FALSE;
END_IF

(*Check if thats a basket for Rapid Function*)
IF bLdCvEnable THEN
	bRapidEnable := FALSE;
	iFL1 := 1;
	FOR iFL1 := 1 TO iCVLdQty DO
		IF iFL1 >= 1 AND iFL1 <= iCVLdQty THEN
			IF iFL1 > 1 AND AR2sDSLdConfirmBasketInfo[iLdConveyorNo, iFL1].bAvailibility THEN
			bRapidEnable := TRUE;
			END_IF

			IF iFL1 >= 1 AND AR2sDSLdTransferBasketInfo[iLdConveyorNo, iFL1].bAvailibility THEN
			bRapidEnable := TRUE;
			END_IF

		END_IF
	END_FOR

ELSIF  bUldCvEnable THEN
	bRapidEnable := FALSE;
	iFL1 := 1;
	FOR iFL1 := 1 TO iCVUldQty DO
		IF iFL1 >= 1 AND iFL1 <= iCVUldQty THEN
			IF iFL1 > 1 AND AR2sDSUldConfirmBasketInfo[iUldConveyorNo, iFL1].bAvailibility THEN
			bRapidEnable := TRUE;
			END_IF

			IF iFL1 >= 1 AND AR2sDSUldTransferBasketInfo[iUldConveyorNo, iFL1].bAvailibility THEN
			bRapidEnable := TRUE;
			END_IF

		END_IF
	END_FOR

END_IF

(*Status*)
IF NOT bLdCvEnable AND NOT bUldCvEnable THEN
sStatus := 'Please Enable either "bLdCvEnable" or "bUldCvEnable"';
ELSIF bLdCvEnable AND bUldCvEnable THEN
sStatus := 'Error - Only "bLdCvEnable" or "bUldCvEnable" can be Enable, NOT BOTH';
ELSIF NOT bEN THEN
sStatus := 'Please Enable "bEN" to Continue';
ELSIF NOT bMoveEnable THEN
sStatus := '"End Basket" detected, please clear the basket to continue';
(*ELSIF (NOT b1stSensor AND NOT bRapidEnable) AND (b1stSensor AND NOT AR2sDSLdConfirmBasketInfo[iLdConveyorNo, 1].bAvailibility)  THEN
sStatus := 'Idling';*)
ELSIF iStep >= 11 AND iStep <= 19 THEN
sStatus := 'Basket Indexing In Progress...';
ELSIF iStep >= 21 AND iStep <= 29 THEN
sStatus := 'Basket Rapid Mode In Progress...';
ELSIF b1stSensor AND AR2sDSLdConfirmBasketInfo[iLdConveyorNo, 1].bAvailibility THEN
sStatus := 'Ready - Press "bIndexPB" to start Basket Indexing';
ELSIF NOT b1stSensor AND bRapidEnable THEN
sStatus := 'Ready - Press "bRapidPB" to start Basket Shift into End Station';
ELSIF iStep = 1 THEN
sStatus := 'Idling...';
ELSE
sStatus := 'Status - Unknown';
END_IF

IF (bLdCvEnable AND AR2sDSLdConfirmBasketInfo[iLdConveyorNo, 1].bAvailibility) OR (bUldCvEnable AND AR2sDSUldConfirmBasketInfo[iUldConveyorNo, 1].bAvailibility) THEN
b1stBasketConfirmEnable := TRUE;
ELSE
b1stBasketConfirmEnable := FALSE;
END_IF

(*Timer Based Rapid Programming*)
diTimerBasedRapidDelaySV_mSec := (iTimerBasedRapidDelaySV_Mins*60*1000);
bTimerBasedRapidSt := bTimerBasedRapidIndexEn AND NOT bConveyorStart AND NOT b1stSensor ;


(*Timer, R_TRIG and F_TRIG*)
bIndexPBDelayTimer					(IN:=bIndexPB AND b1stSensor AND b1stBasketConfirmEnable AND bMoveEnable  , 				PT:=REAL_TO_TIME(rIndexPBDelayTimeSV_Sec*1000) , 		Q=> , ET=>tIndexPBDelayTimePV );
bRapidPBDelayTimer					(IN:=bRapidPB AND NOT b1stSensor AND bRapidEnable AND bMoveEnable , 					PT:=REAL_TO_TIME(rRapidPBDelayTimeSV_Sec*1000) , 		Q=> , ET=>tRapidPBDelayTimePV );
bTimerBasedRapidDelayTimer			(IN:=bTimerBasedRapidSt AND bRapidEnable AND bMoveEnable , 								PT:=DINT_TO_TIME(diTimerBasedRapidDelaySV_mSec) , 		Q=> , ET=>tTimerBasedRapidDelayTimePV );
bIndexConfirmDelayTimer				(IN:=bIndexConfirmSensor , 																	PT:=REAL_TO_TIME(rIndexConfirmDelayTimeSV_Sec*1000) , 	Q=> , ET=>tIndexConfirmDelayTimePV );
bEndZoneDelayTimer					(IN:=bEndZoneSensor , 																	PT:=REAL_TO_TIME(rEndZoneDelayTimeSV_Sec*1000) , 		Q=> , ET=>tEndZoneDelayTimePV );


bENRE								(CLK:=bEN , 								Q=> );
bIndexPBDelayTimerRE				(CLK:=bIndexPBDelayTimer.Q , 				Q=> );
bRapidPBDelayTimerRE				(CLK:=bRapidPBDelayTimer.Q , 				Q=> );
bTimerBasedRapidDelayTimerRE		(CLK:=bTimerBasedRapidDelayTimer.Q , 		Q=> );
bIndexConfirmDelayTimerRE			(CLK:=bIndexConfirmDelayTimer.Q ,		 	Q=> );
bEndZoneDelayTimerRE				(CLK:=bEndZoneDelayTimer.Q , 				Q=> );

(*Generate Availability Signal*)
IF bLdCvEnable THEN
	iFL1 := 1;
	FOR iFL1 := 1 TO iCVLdQty DO
		IF iFL1 >= 1 AND iFL1 <= iCVLdQty THEN
			IF AR2sDSLdConfirmBasketInfo[iLdConveyorNo, iFL1].iProductRecipeNo > 0 AND AR2sDSLdConfirmBasketInfo[iLdConveyorNo, iFL1].iProductRecipeNo <= iProductRecipeArrayQty THEN
			AR2sDSLdConfirmBasketInfo[iLdConveyorNo, iFL1].bAvailibility := TRUE;
			ELSE
			AR2sDSLdConfirmBasketInfo[iLdConveyorNo, iFL1].bAvailibility := FALSE;
			END_IF

			IF AR2sDSLdTransferBasketInfo[iLdConveyorNo, iFL1].iProductRecipeNo > 0 AND AR2sDSLdTransferBasketInfo[iLdConveyorNo, iFL1].iProductRecipeNo <= iProductRecipeArrayQty THEN
			AR2sDSLdTransferBasketInfo[iLdConveyorNo, iFL1].bAvailibility := TRUE;
			ELSE
			AR2sDSLdTransferBasketInfo[iLdConveyorNo, iFL1].bAvailibility := FALSE;
			END_IF

		END_IF
	END_FOR

ELSIF bUldCvEnable THEN
	iFL1 := 1;
	FOR iFL1 := 1 TO iCVUldQty DO
		IF iFL1 >= 1 AND iFL1 <= iCVUldQty THEN
			IF AR2sDSUldConfirmBasketInfo[iUldConveyorNo, iFL1].iProductRecipeNo > 0 AND AR2sDSUldConfirmBasketInfo[iUldConveyorNo, iFL1].iProductRecipeNo <= iProductRecipeArrayQty THEN
			AR2sDSUldConfirmBasketInfo[iUldConveyorNo, iFL1].bAvailibility := TRUE;
			ELSE
			AR2sDSUldConfirmBasketInfo[iUldConveyorNo, iFL1].bAvailibility := FALSE;
			END_IF

			IF AR2sDSUldTransferBasketInfo[iUldConveyorNo, iFL1].iProductRecipeNo > 0 AND AR2sDSUldTransferBasketInfo[iUldConveyorNo, iFL1].iProductRecipeNo <= iProductRecipeArrayQty THEN
			AR2sDSUldTransferBasketInfo[iUldConveyorNo, iFL1].bAvailibility := TRUE;
			ELSE
			AR2sDSUldTransferBasketInfo[iUldConveyorNo, iFL1].bAvailibility := FALSE;
			END_IF

		END_IF
	END_FOR


END_IF




(*Enable Control*)
IF NOT bEN OR( (bLdCvEnable AND bUldCvEnable) OR (NOT bLdCvEnable AND NOT bUldCvEnable) )THEN
iStep := 0;
END_IF

IF bENRE.Q AND( (bLdCvEnable AND NOT bUldCvEnable) OR  (NOT bLdCvEnable AND bUldCvEnable))THEN
iStep := 1;
END_IF





IF iStep = 1 THEN

	IF bIndexPBDelayTimerRE.Q THEN
	iStep := 11;
	END_IF

	IF bRapidPBDelayTimerRE.Q OR bTimerBasedRapidDelayTimerRE.Q THEN
	iStep := 21;
	END_IF

END_IF

CASE iStep OF
0: (*RESET*)
bConveyorStart := FALSE;


1: (*StandBy*)
bConveyorStart := FALSE;

11: (*Index - Shift Confirm to Transfer*)

IF bLdCvEnable THEN
	iFL1 := 1;
	FOR iFL1 := 1 TO iCVLdQty-1 DO
		IF iFL1 >= 1 AND iFL1 <= iCVLdQty-1 THEN
			IF AR2sDSLdConfirmBasketInfo[iLdConveyorNo, iFL1].bAvailibility THEN
				AR2sDSLdTransferBasketInfo[iLdConveyorNo, iFL1]		:= AR2sDSLdConfirmBasketInfo[iLdConveyorNo, iFL1];
				AR2sDSLdConfirmBasketInfo[iLdConveyorNo, iFL1] 		:= DSEmptyBasketInfo;
			END_IF
		END_IF
	END_FOR

ELSIF bUldCvEnable THEN
	iFL1 := 1;
	FOR iFL1 := 1 TO iCVUldQty-1 DO
		IF iFL1 >= 1 AND iFL1 <= iCVUldQty-1 THEN
			IF AR2sDSUldConfirmBasketInfo[iUldConveyorNo, iFL1].bAvailibility THEN
				AR2sDSUldTransferBasketInfo[iUldConveyorNo, iFL1]		:= AR2sDSUldConfirmBasketInfo[iUldConveyorNo, iFL1];
				AR2sDSUldConfirmBasketInfo[iUldConveyorNo, iFL1] 		:= DSEmptyBasketInfo;
			END_IF
		END_IF
	END_FOR

END_IF

iStep := 12;

12: (*Index - Index Start*)
bConveyorStart := TRUE;

IF bIndexConfirmDelayTimerRE.Q THEN
iStep := 13;
END_IF

13: (*Index - Index Completed -> Shift Transfer to Confirm *)
bConveyorStart := FALSE;


IF bLdCvEnable THEN
	iFL1 := 1;
	FOR iFL1 := 1 TO iCVLdQty-1 DO
		IF iFL1 >= 1 AND iFL1 <= iCVLdQty-1 THEN
			IF AR2sDSLdTransferBasketInfo[iLdConveyorNo, iFL1].bAvailibility THEN
				AR2sDSLdConfirmBasketInfo[iLdConveyorNo, iFL1+1]		:= AR2sDSLdTransferBasketInfo[iLdConveyorNo, iFL1];
				AR2sDSLdTransferBasketInfo[iLdConveyorNo, iFL1] 		:= DSEmptyBasketInfo;
			END_IF
		END_IF
	END_FOR

ELSIF bUldCvEnable THEN
	iFL1 := 1;
	FOR iFL1 := 1 TO iCVUldQty-1 DO
		IF iFL1 >= 1 AND iFL1 <= iCVUldQty-1 THEN
			IF AR2sDSUldTransferBasketInfo[iUldConveyorNo, iFL1].bAvailibility THEN
				AR2sDSUldConfirmBasketInfo[iUldConveyorNo, iFL1+1]		:= AR2sDSUldTransferBasketInfo[iUldConveyorNo, iFL1];
				AR2sDSUldTransferBasketInfo[iUldConveyorNo, iFL1] 		:= DSEmptyBasketInfo;
			END_IF
		END_IF
	END_FOR

END_IF

iStep := 1; (*Index - DONE*)




21: (*Rapid - Shift Confirm to Transfer*)

IF bLdCvEnable THEN
	iFL1 := 1;
	FOR iFL1 := 1 TO iCVLdQty-1 DO
		IF iFL1 >= 1 AND iFL1 <= iCVLdQty-1 THEN
			IF AR2sDSLdConfirmBasketInfo[iLdConveyorNo, iFL1].bAvailibility THEN
				AR2sDSLdTransferBasketInfo[iLdConveyorNo, iFL1]		:= AR2sDSLdConfirmBasketInfo[iLdConveyorNo, iFL1];
				AR2sDSLdConfirmBasketInfo[iLdConveyorNo, iFL1] 		:= DSEmptyBasketInfo;
			END_IF
		END_IF
	END_FOR

ELSIF bUldCvEnable THEN
	iFL1 := 1;
	FOR iFL1 := 1 TO iCVUldQty-1 DO
		IF iFL1 >= 1 AND iFL1 <= iCVUldQty-1 THEN
			IF AR2sDSUldConfirmBasketInfo[iUldConveyorNo, iFL1].bAvailibility THEN
				AR2sDSUldTransferBasketInfo[iUldConveyorNo, iFL1]		:= AR2sDSUldConfirmBasketInfo[iUldConveyorNo, iFL1];
				AR2sDSUldConfirmBasketInfo[iUldConveyorNo, iFL1] 		:= DSEmptyBasketInfo;
			END_IF
		END_IF
	END_FOR

END_IF

iStep := 22;

22: (*Rapid - Index Start*)
bConveyorStart := TRUE;

IF bEndZoneDelayTimerRE.Q THEN
iStep := 23;
END_IF

23: (*Rapid - Movement Completed -> Shift Transfer to Confirm *)
bConveyorStart := FALSE;


IF bLdCvEnable THEN
	iLastTransferBasketAddress := 0;
	iFL1 := 1;
	FOR iFL1 := 1 TO iCVLdQty-1 DO
		IF iFL1 >= 1 AND iFL1 <= iCVLdQty-1 THEN
			IF AR2sDSLdTransferBasketInfo[iLdConveyorNo, iFL1].bAvailibility THEN
				iLastTransferBasketAddress:= iFL1;
			END_IF
		END_IF
	END_FOR

	iFL1 :=1;
	FOR iFL1 := 1 TO iLastTransferBasketAddress DO
		IF iFL1 >= 1 AND iFL1 <= iLastTransferBasketAddress THEN

			AR2sDSLdConfirmBasketInfo[iLdConveyorNo, iFL1+(iCVLdQty-iLastTransferBasketAddress)]:= AR2sDSLdTransferBasketInfo[iLdConveyorNo, iFL1];
			AR2sDSLdTransferBasketInfo[iLdConveyorNo, iFL1] := DSEmptyBasketInfo;

		END_IF
	END_FOR


ELSIF bUldCvEnable THEN
	iLastTransferBasketAddress := 0;
	iFL1 := 1;
	FOR iFL1 := 1 TO iCVUldQty-1 DO
		IF iFL1 >= 1 AND iFL1 <= iCVUldQty-1 THEN
			IF AR2sDSUldTransferBasketInfo[iUldConveyorNo, iFL1].bAvailibility THEN
				iLastTransferBasketAddress:= iFL1;
			END_IF
		END_IF
	END_FOR

	iFL1 :=1;
	FOR iFL1 := 1 TO iLastTransferBasketAddress DO
		IF iFL1 >= 1 AND iFL1 <= iLastTransferBasketAddress THEN

			AR2sDSUldConfirmBasketInfo[iUldConveyorNo, iFL1+(iCVUldQty-iLastTransferBasketAddress)]:= AR2sDSUldTransferBasketInfo[iUldConveyorNo, iFL1];
			AR2sDSUldTransferBasketInfo[iUldConveyorNo, iFL1] := DSEmptyBasketInfo;

		END_IF
	END_FOR



(*	iFL1 := 1;
	FOR iFL1 := 1 TO iCVUldQty-1 DO
		IF iFL1 >= 1 AND iFL1 <= iCVUldQty-1 THEN
			IF AR2sDSUldTransferBasketInfo[iUldConveyorNo, iFL1].bAvailibility THEN
				AR2sDSUldConfirmBasketInfo[iUldConveyorNo, iFL1+1]		:= AR2sDSUldTransferBasketInfo[iUldConveyorNo, iFL1];
				AR2sDSUldTransferBasketInfo[iUldConveyorNo, iFL1] 		:= DSEmptyBasketInfo;
			END_IF
		END_IF
	END_FOR
*)
END_IF

iStep := 1; (*Index - DONE*)





END_CASE

END_FUNCTION_BLOCK

// ---- FBs/B_JKS_NewFB_V2/FBP-LdUldCVRelated/fbV2_Cv5zonewith5m5sCtrl.TcPOU
FUNCTION_BLOCK fbV2_Cv5zonewith5m5sCtrl
VAR_INPUT

	bEn : BOOL;
	bResetPB : BOOL;
	rConveyorPos1DelayTime_sec : REAL;
	rConveyorPos2DelayTime_sec : REAL;
	rConveyorPos3DelayTime_sec : REAL;
	rConveyorPos4DelayTime_sec : REAL;
	bCvSensor1 : BOOL;
	bCvSensor2 : BOOL;
	bCvSensor3 : BOOL;
	bCvSensor4 : BOOL;
	bCvSensor5 : BOOL;

	bCvZone1BasketConfirm : BOOL;
	bCvZone2BasketConfirm : BOOL;
	bCvZone3BasketConfirm : BOOL;
	bCvZone4BasketConfirm : BOOL;
	bCvZone5BasketConfirm : BOOL;

	bCvZone1BasketTransfer : BOOL;
	bCvZone2BasketTransfer : BOOL;
	bCvZone3BasketTransfer : BOOL;
	bCvZone4BasketTransfer : BOOL;
	bCvZone5BasketTransfer : BOOL;

END_VAR
VAR_OUTPUT

	bUldEndReached : BOOL;
	bCvFullSignal : BOOL;

	bCvMotor1OnOff : BOOL;
	bCvMotor2OnOff : BOOL;
	bCvMotor3OnOff : BOOL;
	bCvMotor4OnOff : BOOL;
	bCvMotor5OnOff : BOOL;

	bConveyorMotorOnOffAbnormal: BOOL;
END_VAR
VAR

	bZone4Enable: BOOL;
	bZone3Enable: BOOL;
	bZone2Enable: BOOL;
	bZone1Enable: BOOL;

	bCvMotor5OnOff2: BOOL;
	bCvMotor5OnOff1: BOOL;
	bCvMotor4OnOff2: BOOL;
	bCvMotor4OnOff1: BOOL;
	bCvMotor3OnOff2: BOOL;
	bCvMotor3OnOff1: BOOL;
	bCvMotor2OnOff2: BOOL;
	bCvMotor2OnOff1: BOOL;
	bCvMotor1OnOff2: BOOL;
	bCvMotor1OnOff1: BOOL;

	bTimerCountdown: BOOL;
	tCountDownDelayTimer: TON;

	bResetPBRE: R_TRIG;

	tConveyorPos1DelayTimer: TON;
	tConveyorPos2DelayTimer: TON;
	tConveyorPos3DelayTimer: TON;
	tConveyorPos4DelayTimer: TON;

END_VAR

IF bCvSensor1 AND bCvSensor2 AND bCvSensor3 AND bCvSensor4 AND bCvSensor5 THEN

bCvFullSignal := TRUE;
ELSE
bCvFullSignal := FALSE;
END_IF

IF bCvSensor5 THEN
bUldEndReached := TRUE;
ELSE
bUldEndReached := FALSE;
END_IF


tConveyorPos1DelayTimer(IN:=bZone1Enable AND bCvSensor2 , PT:= REAL_TO_TIME(rConveyorPos1DelayTime_sec*1000) , Q=> , ET=> );
tConveyorPos2DelayTimer(IN:=bZone2Enable AND bCvSensor3 , PT:= REAL_TO_TIME(rConveyorPos2DelayTime_sec*1000) , Q=> , ET=> );
tConveyorPos3DelayTimer(IN:=bZone3Enable AND bCvSensor4 , PT:= REAL_TO_TIME(rConveyorPos3DelayTime_sec*1000) , Q=> , ET=> );
tConveyorPos4DelayTimer(IN:=bZone4Enable AND bCvSensor5 , PT:= REAL_TO_TIME(rConveyorPos4DelayTime_sec*1000) , Q=> , ET=> );


IF bEn (*AND NOT tCountDownDelayTimer.Q*) THEN

	(* Zone4 to Zone5 *)
	IF bCvSensor4 AND NOT bCvSensor5 AND NOT bZone3Enable AND ( bCvZone4BasketConfirm OR bCvZone4BasketTransfer) AND NOT bCvZone5BasketConfirm THEN
	bZone4Enable := TRUE;
	bCvMotor4OnOff2 := TRUE;
	bCvMotor5OnOff1 := TRUE;
	END_IF

	IF tConveyorPos4DelayTimer.Q (*bZone4Enable (*AND NOT bCvSensor4 *)AND bCvSensor5*) THEN
	bZone4Enable := FALSE;
	bCvMotor4OnOff2 := FALSE;
	bCvMotor5OnOff1 := FALSE;
	END_IF

	(* Zone3 to Zone4 *)
	IF bCvSensor3 AND NOT bCvSensor4 AND NOT bZone2Enable AND NOT bZone4Enable AND ( bCvZone3BasketConfirm OR bCvZone3BasketTransfer) AND NOT bCvZone4BasketConfirm THEN
	bZone3Enable := TRUE;
	bCvMotor3OnOff2 := TRUE;
	bCvMotor4OnOff1 := TRUE;
	END_IF

	IF tConveyorPos3DelayTimer.Q (*bZone3Enable (*AND NOT bCvSensor3 *)AND bCvSensor4*) THEN
	bZone3Enable := FALSE;
	bCvMotor3OnOff2 := FALSE;
	bCvMotor4OnOff1 := FALSE;
	END_IF

	(* Zone2 to Zone3 *)
	IF bCvSensor2 AND NOT bCvSensor3 AND NOT bZone1Enable AND NOT bZone3Enable AND ( bCvZone2BasketConfirm OR bCvZone2BasketTransfer) AND NOT bCvZone3BasketConfirm THEN
	bZone2Enable := TRUE;
	bCvMotor2OnOff2 := TRUE;
	bCvMotor3OnOff1 := TRUE;
	END_IF

	IF tConveyorPos2DelayTimer.Q (*bZone2Enable (*AND NOT bCvSensor2 *)AND bCvSensor3*) THEN
	bZone2Enable := FALSE;
	bCvMotor2OnOff2 := FALSE;
	bCvMotor3OnOff1 := FALSE;
	END_IF

	(* Zone1 to Zone2 *)
	IF bCvSensor1 AND NOT bCvSensor2 AND NOT bZone2Enable AND ( bCvZone1BasketConfirm OR bCvZone1BasketTransfer ) AND NOT bCvZone2BasketConfirm THEN
	bZone1Enable := TRUE;
	bCvMotor1OnOff1 := TRUE;
	bCvMotor2OnOff1 := TRUE;
	END_IF

	IF tConveyorPos1DelayTimer.Q (*bZone1Enable (*AND NOT bCvSensor1 *)AND bCvSensor2*) THEN
	bZone1Enable := FALSE;
	bCvMotor1OnOff1 := FALSE;
	bCvMotor2OnOff1 := FALSE;
	END_IF

ELSE
	bCvMotor1OnOff1 := FALSE;
	bCvMotor2OnOff1 := FALSE;
	bCvMotor3OnOff1 := FALSE;
	bCvMotor4OnOff1 := FALSE;
	bCvMotor5OnOff1 := FALSE;

	bCvMotor1OnOff2 := FALSE;
	bCvMotor2OnOff2 := FALSE;
	bCvMotor3OnOff2 := FALSE;
	bCvMotor4OnOff2 := FALSE;
	bCvMotor5OnOff2 := FALSE;

	bZone1Enable := FALSE;
	bZone2Enable := FALSE;
	bZone3Enable := FALSE;
	bZone4Enable := FALSE;

END_IF


IF bCvMotor1OnOff1 OR bCvMotor1OnOff2 THEN
bCvMotor1OnOff := TRUE;
ELSE
bCvMotor1OnOff := FALSE;
END_IF

IF bCvMotor2OnOff1 OR bCvMotor2OnOff2 THEN
bCvMotor2OnOff := TRUE;
ELSE
bCvMotor2OnOff := FALSE;
END_IF

IF bCvMotor3OnOff1 OR bCvMotor3OnOff2 THEN
bCvMotor3OnOff := TRUE;
ELSE
bCvMotor3OnOff := FALSE;
END_IF

IF bCvMotor4OnOff1 OR bCvMotor4OnOff2 THEN
bCvMotor4OnOff := TRUE;
ELSE
bCvMotor4OnOff := FALSE;
END_IF

IF bCvMotor5OnOff1 OR bCvMotor5OnOff2 THEN
bCvMotor5OnOff := TRUE;
ELSE
bCvMotor5OnOff := FALSE;
END_IF


bResetPBRE(CLK:= bResetPB , Q=> );

IF (bZone4Enable OR bZone3Enable OR bZone2Enable OR bZone1Enable) AND ( NOT bCvSensor1 OR NOT bCvSensor2 OR NOT  bCvSensor3 OR NOT  bCvSensor4 OR NOT bCvSensor5 ) AND NOT bResetPBRE.Q THEN
bTimerCountdown := TRUE;
ELSE
bTimerCountdown := FALSE;
END_IF


tCountDownDelayTimer(IN:=bTimerCountdown , PT:=t#90s , Q=> , ET=> );

IF tCountDownDelayTimer.Q THEN
bConveyorMotorOnOffAbnormal := TRUE;
END_IF

IF bConveyorMotorOnOffAbnormal AND NOT bCvZone1BasketTransfer AND NOT bCvZone2BasketTransfer AND NOT bCvZone3BasketTransfer AND NOT bCvZone4BasketTransfer AND NOT bCvZone5BasketTransfer THEN
bConveyorMotorOnOffAbnormal := FALSE;
END_IF

IF bResetPBRE.Q THEN
bConveyorMotorOnOffAbnormal := FALSE;
END_IF

END_FUNCTION_BLOCK

// ---- FBs/B_JKS_NewFB_V2/FBP-LdUldCVRelated/fbV2_Cv4zonewith4m4sCtrl.TcPOU
FUNCTION_BLOCK fbV2_Cv4zonewith4m4sCtrl
VAR_INPUT

	bEn : BOOL;
	bResetPB : BOOL;
	rConveyorPos1DelayTime_sec : REAL;
	rConveyorPos2DelayTime_sec : REAL;
	rConveyorPos3DelayTime_sec : REAL;
	bCvSensor1 : BOOL;
	bCvSensor2 : BOOL;
	bCvSensor3 : BOOL;
	bCvSensor4 : BOOL;

	bCvZone1BasketConfirm : BOOL;
	bCvZone2BasketConfirm : BOOL;
	bCvZone3BasketConfirm : BOOL;
	bCvZone4BasketConfirm : BOOL;

	bCvZone1BasketTransfer : BOOL;
	bCvZone2BasketTransfer : BOOL;
	bCvZone3BasketTransfer : BOOL;
	bCvZone4BasketTransfer : BOOL;

END_VAR
VAR_OUTPUT

	bUldEndReached : BOOL;
	bCvFullSignal : BOOL;

	bCvMotor1OnOff : BOOL;
	bCvMotor2OnOff : BOOL;
	bCvMotor3OnOff : BOOL;
	bCvMotor4OnOff : BOOL;

	bConveyorMotorOnOffAbnormal: BOOL;
END_VAR
VAR

	bZone3Enable: BOOL;
	bZone2Enable: BOOL;
	bZone1Enable: BOOL;

	bCvMotor4OnOff2: BOOL;
	bCvMotor4OnOff1: BOOL;
	bCvMotor3OnOff2: BOOL;
	bCvMotor3OnOff1: BOOL;
	bCvMotor2OnOff2: BOOL;
	bCvMotor2OnOff1: BOOL;
	bCvMotor1OnOff2: BOOL;
	bCvMotor1OnOff1: BOOL;

	bTimerCountdown: BOOL;
	tCountDownDelayTimer: TON;

	bResetPBRE: R_TRIG;

	tConveyorPos1DelayTimer: TON;
	tConveyorPos2DelayTimer: TON;
	tConveyorPos3DelayTimer: TON;

END_VAR

IF bCvSensor1 AND bCvSensor2 AND bCvSensor3 AND bCvSensor4 THEN

bCvFullSignal := TRUE;
ELSE
bCvFullSignal := FALSE;
END_IF

IF bCvSensor4 THEN
bUldEndReached := TRUE;
ELSE
bUldEndReached := FALSE;
END_IF


tConveyorPos1DelayTimer(IN:=bZone1Enable AND bCvSensor2 , PT:= REAL_TO_TIME(rConveyorPos1DelayTime_sec*1000) , Q=> , ET=> );
tConveyorPos2DelayTimer(IN:=bZone2Enable AND bCvSensor3 , PT:= REAL_TO_TIME(rConveyorPos2DelayTime_sec*1000) , Q=> , ET=> );
tConveyorPos3DelayTimer(IN:=bZone3Enable AND bCvSensor4 , PT:= REAL_TO_TIME(rConveyorPos3DelayTime_sec*1000) , Q=> , ET=> );


IF bEn (*AND NOT tCountDownDelayTimer.Q*) THEN

	(* Zone3 to Zone4 *)
	IF bCvSensor3 AND NOT bCvSensor4 AND NOT bZone2Enable AND ( bCvZone3BasketConfirm OR bCvZone3BasketTransfer) AND NOT bCvZone4BasketConfirm THEN
	bZone3Enable := TRUE;
	bCvMotor3OnOff2 := TRUE;
	bCvMotor4OnOff1 := TRUE;
	END_IF

	IF tConveyorPos3DelayTimer.Q (*bZone3Enable (*AND NOT bCvSensor3 *)AND bCvSensor4*) THEN
	bZone3Enable := FALSE;
	bCvMotor3OnOff2 := FALSE;
	bCvMotor4OnOff1 := FALSE;
	END_IF

	(* Zone2 to Zone3 *)
	IF bCvSensor2 AND NOT bCvSensor3 AND NOT bZone1Enable AND NOT bZone3Enable AND ( bCvZone2BasketConfirm OR bCvZone2BasketTransfer) AND NOT bCvZone3BasketConfirm THEN
	bZone2Enable := TRUE;
	bCvMotor2OnOff2 := TRUE;
	bCvMotor3OnOff1 := TRUE;
	END_IF

	IF tConveyorPos2DelayTimer.Q (*bZone2Enable (*AND NOT bCvSensor2 *)AND bCvSensor3*) THEN
	bZone2Enable := FALSE;
	bCvMotor2OnOff2 := FALSE;
	bCvMotor3OnOff1 := FALSE;
	END_IF

	(* Zone1 to Zone2 *)
	IF bCvSensor1 AND NOT bCvSensor2 AND NOT bZone2Enable AND ( bCvZone1BasketConfirm OR bCvZone1BasketTransfer ) AND NOT bCvZone2BasketConfirm THEN
	bZone1Enable := TRUE;
	bCvMotor1OnOff1 := TRUE;
	bCvMotor2OnOff1 := TRUE;
	END_IF

	IF tConveyorPos1DelayTimer.Q (*bZone1Enable (*AND NOT bCvSensor1 *)AND bCvSensor2*) THEN
	bZone1Enable := FALSE;
	bCvMotor1OnOff1 := FALSE;
	bCvMotor2OnOff1 := FALSE;
	END_IF

ELSE
	bCvMotor1OnOff1 := FALSE;
	bCvMotor2OnOff1 := FALSE;
	bCvMotor3OnOff1 := FALSE;
	bCvMotor4OnOff1 := FALSE;

	bCvMotor1OnOff2 := FALSE;
	bCvMotor2OnOff2 := FALSE;
	bCvMotor3OnOff2 := FALSE;
	bCvMotor4OnOff2 := FALSE;

	bZone1Enable := FALSE;
	bZone2Enable := FALSE;
	bZone3Enable := FALSE;

END_IF


IF bCvMotor1OnOff1 OR bCvMotor1OnOff2 THEN
bCvMotor1OnOff := TRUE;
ELSE
bCvMotor1OnOff := FALSE;
END_IF

IF bCvMotor2OnOff1 OR bCvMotor2OnOff2 THEN
bCvMotor2OnOff := TRUE;
ELSE
bCvMotor2OnOff := FALSE;
END_IF

IF bCvMotor3OnOff1 OR bCvMotor3OnOff2 THEN
bCvMotor3OnOff := TRUE;
ELSE
bCvMotor3OnOff := FALSE;
END_IF

IF bCvMotor4OnOff1 OR bCvMotor4OnOff2 THEN
bCvMotor4OnOff := TRUE;
ELSE
bCvMotor4OnOff := FALSE;
END_IF


bResetPBRE(CLK:= bResetPB , Q=> );

IF (bZone3Enable OR bZone2Enable OR bZone1Enable) AND ( NOT bCvSensor1 OR NOT bCvSensor2 OR NOT  bCvSensor3 OR NOT  bCvSensor4  ) AND NOT bResetPBRE.Q THEN
bTimerCountdown := TRUE;
ELSE
bTimerCountdown := FALSE;
END_IF

tCountDownDelayTimer(IN:=bTimerCountdown , PT:=t#90s , Q=> , ET=> );

IF tCountDownDelayTimer.Q THEN
bConveyorMotorOnOffAbnormal := TRUE;
END_IF

IF bConveyorMotorOnOffAbnormal AND NOT bCvZone1BasketTransfer AND NOT bCvZone2BasketTransfer AND NOT bCvZone3BasketTransfer AND NOT bCvZone4BasketTransfer THEN
bConveyorMotorOnOffAbnormal := FALSE;
END_IF

IF bResetPBRE.Q THEN
bConveyorMotorOnOffAbnormal := FALSE;
END_IF

END_FUNCTION_BLOCK

// ---- FBs/B_JKS_NewFB_V2/FBP-LdUldCVRelated/fbV2_Cv3zonewith3m3sCtrl.TcPOU
FUNCTION_BLOCK fbV2_Cv3zonewith3m3sCtrl
VAR_INPUT

	bEn : BOOL;
	bResetPB : BOOL;
	rConveyorPos1DelayTime_sec : REAL;
	rConveyorPos2DelayTime_sec : REAL;
	bCvSensor1 : BOOL;
	bCvSensor2 : BOOL;
	bCvSensor3 : BOOL;

	bCvZone1BasketConfirm : BOOL;
	bCvZone2BasketConfirm : BOOL;
	bCvZone3BasketConfirm : BOOL;

	bCvZone1BasketTransfer : BOOL;
	bCvZone2BasketTransfer : BOOL;
	bCvZone3BasketTransfer : BOOL;

END_VAR
VAR_OUTPUT

	bUldEndReached : BOOL;
	bCvFullSignal : BOOL;

	bCvMotor1OnOff : BOOL;
	bCvMotor2OnOff : BOOL;
	bCvMotor3OnOff : BOOL;

	bConveyorMotorOnOffAbnormal: BOOL;
END_VAR
VAR

	bZone2Enable: BOOL;
	bZone1Enable: BOOL;

	bCvMotor3OnOff2: BOOL;
	bCvMotor3OnOff1: BOOL;
	bCvMotor2OnOff2: BOOL;
	bCvMotor2OnOff1: BOOL;
	bCvMotor1OnOff2: BOOL;
	bCvMotor1OnOff1: BOOL;

	bTimerCountdown: BOOL;
	tCountDownDelayTimer: TON;

	bResetPBRE: R_TRIG;

	tConveyorPos1DelayTimer: TON;
	tConveyorPos2DelayTimer: TON;

END_VAR

IF bCvSensor1 AND bCvSensor2 AND bCvSensor3 THEN

bCvFullSignal := TRUE;
ELSE
bCvFullSignal := FALSE;
END_IF

IF bCvSensor3 THEN
bUldEndReached := TRUE;
ELSE
bUldEndReached := FALSE;
END_IF


tConveyorPos1DelayTimer(IN:=bZone1Enable AND bCvSensor2 , PT:= REAL_TO_TIME(rConveyorPos1DelayTime_sec*1000) , Q=> , ET=> );
tConveyorPos2DelayTimer(IN:=bZone2Enable AND bCvSensor3 , PT:= REAL_TO_TIME(rConveyorPos2DelayTime_sec*1000) , Q=> , ET=> );


IF bEn (*AND NOT tCountDownDelayTimer.Q*) THEN

	(* Zone2 to Zone3 *)
	IF bCvSensor2 AND NOT bCvSensor3 AND NOT bZone1Enable AND ( bCvZone2BasketConfirm OR bCvZone2BasketTransfer) AND NOT bCvZone3BasketConfirm THEN
	bZone2Enable := TRUE;
	bCvMotor2OnOff2 := TRUE;
	bCvMotor3OnOff1 := TRUE;
	END_IF

	IF tConveyorPos2DelayTimer.Q (*bZone2Enable (*AND NOT bCvSensor2 *)AND bCvSensor3*) THEN
	bZone2Enable := FALSE;
	bCvMotor2OnOff2 := FALSE;
	bCvMotor3OnOff1 := FALSE;
	END_IF

	(* Zone1 to Zone2 *)
	IF bCvSensor1 AND NOT bCvSensor2 AND NOT bZone2Enable AND ( bCvZone1BasketConfirm OR bCvZone1BasketTransfer ) AND NOT bCvZone2BasketConfirm THEN
	bZone1Enable := TRUE;
	bCvMotor1OnOff1 := TRUE;
	bCvMotor2OnOff1 := TRUE;
	END_IF

	IF tConveyorPos1DelayTimer.Q (*bZone1Enable (*AND NOT bCvSensor1 *)AND bCvSensor2*) THEN
	bZone1Enable := FALSE;
	bCvMotor1OnOff1 := FALSE;
	bCvMotor2OnOff1 := FALSE;
	END_IF

ELSE
	bCvMotor1OnOff1 := FALSE;
	bCvMotor2OnOff1 := FALSE;
	bCvMotor3OnOff1 := FALSE;

	bCvMotor1OnOff2 := FALSE;
	bCvMotor2OnOff2 := FALSE;
	bCvMotor3OnOff2 := FALSE;

	bZone1Enable := FALSE;
	bZone2Enable := FALSE;

END_IF


IF bCvMotor1OnOff1 OR bCvMotor1OnOff2 THEN
bCvMotor1OnOff := TRUE;
ELSE
bCvMotor1OnOff := FALSE;
END_IF

IF bCvMotor2OnOff1 OR bCvMotor2OnOff2 THEN
bCvMotor2OnOff := TRUE;
ELSE
bCvMotor2OnOff := FALSE;
END_IF

IF bCvMotor3OnOff1 OR bCvMotor3OnOff2 THEN
bCvMotor3OnOff := TRUE;
ELSE
bCvMotor3OnOff := FALSE;
END_IF


bResetPBRE(CLK:= bResetPB , Q=> );

IF (bZone2Enable OR bZone1Enable) AND ( NOT bCvSensor1 OR NOT bCvSensor2 OR NOT  bCvSensor3 ) AND NOT bResetPBRE.Q THEN
bTimerCountdown := TRUE;
ELSE
bTimerCountdown := FALSE;
END_IF


tCountDownDelayTimer(IN:=bTimerCountdown , PT:=t#90s , Q=> , ET=> );

IF tCountDownDelayTimer.Q THEN
bConveyorMotorOnOffAbnormal := TRUE;
END_IF

IF bConveyorMotorOnOffAbnormal AND NOT bCvZone1BasketTransfer AND NOT bCvZone2BasketTransfer AND NOT bCvZone3BasketTransfer THEN
bConveyorMotorOnOffAbnormal := FALSE;
END_IF

IF bResetPBRE.Q THEN
bConveyorMotorOnOffAbnormal := FALSE;
END_IF

END_FUNCTION_BLOCK

// ---- FBs/FB_Others TBD/fbV3_TotalProcessTimeTracker.TcPOU
FUNCTION_BLOCK fbV3_TotalProcessTimeTracker
VAR_INPUT
	bEN : BOOL;
	iUserDefineProductRecipeNo : INT;
END_VAR
VAR_OUTPUT
	ARiStationMinTimeDisplay : ARRAY [1..iStnQty] OF INT;
	sStationDescriptionDisplay : STRING;
END_VAR
VAR
	ARiStationMinTimeEmpty : ARRAY [1..iStnQty] OF INT;
	sStationDescriptionEmpty : STRING;
	iSMTFL: INT;
	iSMTSFL: INT;
END_VAR

IF NOT bEN THEN
ARiStationMinTimeDisplay := ARiStationMinTimeEmpty;
sStationDescriptionDisplay := sStationDescriptionEmpty;
END_IF

IF bEN THEN

	iSMTFL := 1;

	ARiStationMinTimeDisplay := ARiStationMinTimeEmpty;
	sStationDescriptionDisplay := sStationDescriptionEmpty;

	FOR iSMTFL := 1 TO iStnQty DO
			IF iSMTFL >= 1 AND iSMTFL <= iStnQty THEN

				iSMTSFL := 1;
				(*ARiStationMinTimeDisplay[iSMTFL] := 0;*)
					FOR iSMTSFL := 1 TO iProductRecipeStepArrayQty DO
						IF iSMTSFL >= 1 AND iSMTSFL <= iProductRecipeStepArrayQty THEN
							IF PnPstorageMemory_Arm.fbGnrProductRecipeMemory_Main.fbA1PnpSequenceMemory.ARDsPnpSequenceMemory[iUserDefineProductRecipeNo].ARiTransferStationNo[iSMTSFL] = iSMTFL THEN

								ARiStationMinTimeDisplay[iSMTFL] := (*ARiStationMinTimeDisplay[iSMTFL] +*) fbMainStationProcess_Stn[iSMTFL].StnSeqProcessfb.fbStationSequenceRecipefb.ARDsStorageStationSequenceRecipeMemory[(**)PnPstorageMemory_Arm.fbGnrProductRecipeMemory_Main.fbA1PnpSequenceMemory.ARDsPnpSequenceMemory[iUserDefineProductRecipeNo].ARiStnSeqRepNo[iSMTSFL](**)].iProcessMinTime;
								sStationDescriptionDisplay := PnPstorageMemory_Arm.fbGnrProductRecipeMemory_Main.fbA1PnpSequenceMemory.ARDsPnpSequenceMemory[iUserDefineProductRecipeNo].sDescription;
							(**)	iSMTSFL := iStnQty + 1;

							END_IF
						END_IF
					END_FOR
			END_IF
	END_FOR
END_IF

iUserDefineProductRecipeNo;

PnPstorageMemory_Arm.fbGnrProductRecipeMemory_Main.fbA1PnpSequenceMemory.ARDsPnpSequenceMemory[iUserDefineProductRecipeNo].ARiTransferStationNo[iSMTSFL];
PnPstorageMemory_Arm.fbGnrProductRecipeMemory_Main.fbA1PnpSequenceMemory.ARDsPnpSequenceMemory[iUserDefineProductRecipeNo].ARiStnSeqRepNo[iSMTSFL];



fbMainStationProcess_Stn[iSMTFL].StnSeqProcessfb.fbStationSequenceRecipefb.ARDsStorageStationSequenceRecipeMemory[(**)PnPstorageMemory_Arm.fbGnrProductRecipeMemory_Main.fbA1PnpSequenceMemory.ARDsPnpSequenceMemory[iUserDefineProductRecipeNo].ARiStnSeqRepNo[iSMTSFL](**)].iProcessMinTime;

END_FUNCTION_BLOCK

// ---- FBs/b_JKS_RecycleFB/fb_V3JRSModuleWithChiller.TcPOU
FUNCTION_BLOCK fb_V3JRSModuleWithChiller
VAR_INPUT
	bBuiltInTemperetureController : BOOL;
	bBuiltInVacuumSensorController : BOOL;
	bBuiltInVacuumNegativeSignal : BOOL;
END_VAR
VAR_OUTPUT
END_VAR
VAR_IN_OUT
	DS_Alarm :DSV3_JRS_Alarm; (*Channel 200 ~ 204*)
	DS_HMI : DSV3_JRS_HMI; (*Channel of Other Digitial IO and DT*)
	DS_Input : DSV3_JRS_Input; (*Channel 0 ~ 3 *)
	DS_Output : DSV3_JRS_Output; (*Channel 100 ~ 103*)
END_VAR
VAR

	(*Analog Declaration*)
	iThermalOilTempAnalogInput			AT %I* : INT;
	iTopDistillatorTempAnalogInput			AT %I* : INT;
	iBottomDistillatorTempAnalogInput		AT %I* : INT;
	iVaporGenerationTempAnalogInput		AT %I* : INT;
	iColdWaterTankTempAnalogInput 		AT %I* : INT;

	iVacuumSensorAnalogInput				AT %I* : INT;



	(*AlarmControl*)
	arfbTimerAlarm: ARRAY [1..49] OF TIMER_ALARM;
	ARiBuzzerOut : ARRAY [1..4] OF INT;
	ARiAlarmFlag : ARRAY [1..4] OF INT;
	arCMP: ARRAY [1..32] OF CMP_OC_W1;


	(*Others*)
	EQGT: ARRAY [1..10] OF EQ_GT;


	tCompressorOnTimer: TON;
	tCompressorOffTimer: TON;
	tPowerOnDelayTimer: TON;
	tVaporGenTopUpDelayOff: TON;
	tThermalOilChangeResetPBTimer: TON;

	bPowerOnDelay: BOOL;

	t1SecCP: TON;

	tFreshHCCircPumpDelayOffTimer: TON;

	ARtAutoModeTimer: ARRAY [1..4] OF TON;
	ARtManualBoilingTimer: ARRAY [1..4] OF TON;
	diAutoModeDelayTimeSV_Sec: DINT := 20;

	bRecycleStartPBRE: R_TRIG;
	t1SecCPRE: R_TRIG;

	(*Auto BoilDown*)
	t570_AutoBoilingStartDelayTimer: TON;
	t571_AutoBoilDownCompletedDelayTimer: TON;
	t572_AutoBoilSludgeDrainCompletedDelayTimer: TON;
	t573_AutoBoilDistillatorDrainCompletedDelayTimer: TON;
	t574_AutoBoilSludgeDrainCoolingCompletedDelayTimer: TON;        (************* New extra request by customer - YCH************)

	bAutoBoilProcessCompletedFlag: BOOL;
	bAutoBoilDownCompletedFlag: BOOL;
	bAutoBoilSludgeDrainCompletedFlag: BOOL;
	bAutoBoilDistillatorDrainCompletedFlag: BOOL;
	bAutoBoilSludgeDrainCoolingCompletedFlag: BOOL;        (************* New extra request by customer - YCH************)

	(*Manual BoilDown*)
	t590_ManualBoilDownCompletedDelayTimer: TON;
	t591_ManualBoilSludgeCoolingCompletedDelayTimer: TON;
	t592_ManualBoilSludgeDrainCompletedDelayTimer: TON;
	bManualBoilDownCompletedFlag: BOOL;
	bManualBoilSludgeCoolingCompletedFlag: BOOL;
	bManualBoilSludgeDrainCompletedFlag: BOOL;
	bManualBoilSludgeDrainCompletedRE: R_TRIG;
	bManualBoilDownStartPBRE: R_TRIG;

	t592_ManualBoilSludgeDrainCompletedDelayTimerRE: R_TRIG;
	ARfbV2TempControl: ARRAY [1..5] OF fbV2_TempControl;
	rNIL: REAL;

	fbKeyenceVacSensorTuningkPa_Vacuum: fbKeyenceVacSensorTuningkPa;
	bVacuumAchieveFlag: BOOL;

	fbJRSMachine_Routine								: fbV2_EquipmentServiceCounter_Day;
	fbJRSMachine_Major									: fbV2_EquipmentServiceCounter_Day;

	bManulBoilPageOn:BOOL;
(*
	bInternalInput_b000_04_ThermalOilTempCtrlHighTempAlarmSignal : BOOL;
	bInternalInput_b000_05_ThermalOilTempCtrlReadySignal : BOOL;
	bInternalInput_b000_06_ThermalOilTempCtrlOnOffSignal : BOOL;
	bInternalInput_b000_04_ThermalOilTempCtrlHighTempAlarmSignal  : BOOL;
	bInternalInput_b000_05_ThermalOilTempCtrlReadySignal  : BOOL;
	bInternalInput_b000_06_ThermalOilTempCtrlOnOffSignal   : BOOL;

	bInternalInput_b000_07_TopDistillatorTempCtrlHighTempAlarmSignal : BOOL;
	bInternalInput_b000_08_TopDistillatorTempCtrlReadySignal : BOOL;
	bInternalInput_b000_09_TopDistillatorTempCtrlOnOffSignal : BOOL;
	bInternalInput_b000_07_TopDistillatorTempCtrlHighTempAlarmSignal  : BOOL;
	bInternalInput_b000_08_TopDistillatorTempCtrlReadySignal  : BOOL;
	bInternalInput_b000_09_TopDistillatorTempCtrlOnOffSignal   : BOOL;

	bInternalInput_b001_08_BottomDistillatorTempCtrlHighTempAlarmSignal : BOOL;
	bInternalInput_b001_09_BottomDistillatorTempCtrlReadySignal : BOOL;
	bInternalInput_b001_10_BottomDistillatorTempCtrlOnOffSignal : BOOL;
	bInternalInput_b001_08_BottomDistillatorTempCtrlHighTempAlarmSignal  : BOOL;
	bInternalInput_b001_09_BottomDistillatorTempCtrlReadySignal  : BOOL;
	bInternalInput_b001_10_BottomDistillatorTempCtrlOnOffSignal   : BOOL;

	bInternalInput_b002_00_VaporGenerationTempCtrlHighTempAlarmSignal : BOOL;
	bInternalInput_b002_01_VaporGenerationTempCtrlReadySignal : BOOL;
	bInternalInput_b002_02_VaporGenerationTempCtrlOnOffSignal : BOOL;
	bInternalInput_b002_00_VaporGenerationTempCtrlHighTempAlarmSignal  : BOOL;
	bInternalInput_b002_01_VaporGenerationTempCtrlReadySignal  : BOOL;
	bInternalInput_b002_02_VaporGenerationTempCtrlOnOffSignal  : BOOL;


	bInternalInput_b003_03_ColdWaterTankTempCtrlHighTempAlarmSignal : BOOL;
	bInternalInput_b003_04_ColdWaterTankTempCtrlReadySignal : BOOL;
	bInternalInput_b003_05_ColdWaterTankTempCtrlOnOffSignal	 : BOOL;
	bInternalInput_b003_03_ColdWaterTankTempCtrlHighTempAlarmSignal  : BOOL;
	bInternalInput_b003_04_ColdWaterTankTempCtrlReadySignal  : BOOL;
	bInternalInput_b003_05_ColdWaterTankTempCtrlOnOffSignal  : BOOL;

	bInternalInput_b001_04_VacuumNotAchieveSignal	: BOOL;
	bInternalInput_b001_04_VacuumNotAchieveSignal  : BOOL;

*)

	(*Internal Signal Declaration*)
	bInternalAlarm_b200_00_FreshHCTankCircPumpTORAlarm   : BOOL;
	bInternalAlarm_b200_01_CircTankCircPumpTORAlarm   : BOOL;
	bInternalAlarm_b200_02_ThermalOilPumpTORAlarm   : BOOL;
	bInternalAlarm_b200_03_ThermalOilLowLevelAlarm   : BOOL;
	bInternalAlarm_b200_04_ThermalOilTempHighAlarm   : BOOL;
	bInternalAlarm_b200_05_ThermalOilTempNotReadyAlarm   : BOOL;
	bInternalAlarm_b200_06_ThermalOilHeaterOnOffAlarm   : BOOL;
	bInternalAlarm_b200_07_TopDistillatorTempHighAlarm   : BOOL;
	bInternalAlarm_b200_08_TopDistillatorTempNotReadyAlarm   : BOOL;
	bInternalAlarm_b200_09_TopDistillatorHeaterOnOffAlarm   : BOOL;
	bInternalAlarm_b200_10_RecycleStartStopPBAlarm   : BOOL;
	bInternalAlarm_b200_11_EstopPBAlarm   : BOOL;

	bInternalAlarm_b201_00_PhaseSeqenceRelayAlarm   : BOOL;
	bInternalAlarm_b201_01_ThermalOilUpThermostatAlarm   : BOOL;
	bInternalAlarm_b201_02_SludgeTankHighLevelAlarm   : BOOL;
	bInternalAlarm_b201_03_FreshHCTankLowLevelAlarm   : BOOL;
	bInternalAlarm_b201_04_VacuumNotAchieveAlarm   : BOOL;
	bInternalAlarm_b201_05_IncomingCDALowPressureAlarm   : BOOL;
	bInternalAlarm_b201_06_CoolingWaterLowFlowAlarm   : BOOL;
	bInternalAlarm_b201_07_CircularTankLowLevelAlarm   : BOOL;
	bInternalAlarm_b201_08_BottomDistillatorTempHighAlarm   : BOOL;
	bInternalAlarm_b201_09_BottomDistillatorTempNotReadyAlarm   : BOOL;
	bInternalAlarm_b201_10_BottomDistillatorHeaterOnOffAlarm   : BOOL;
	bInternalAlarm_b201_11_ThermalOilDownThermostatAlarm   : BOOL;
	bInternalAlarm_b201_12_ThermalOilMidThermostatAlarm   : BOOL;

	bInternalAlarm_b202_00_VaporGenerationTempHighAlarm   : BOOL;
	bInternalAlarm_b202_01_VaporGenerationTempNotReadyAlarm   : BOOL;
	bInternalAlarm_b202_02_VaporGenerationHeaterOnOffAlarm   : BOOL;
	bInternalAlarm_b202_03_WasteCollectionTankLowLevelAlarm   : BOOL;
	bInternalAlarm_b202_04_VaporGenerationTankLowLevelAlarm   : BOOL;
	bInternalAlarm_b202_05_HCPurgingAV3_1Alarm   : BOOL;
	bInternalAlarm_b202_06_MainMachineWasteTankLowLevelAlarm   : BOOL;
	bInternalAlarm_b202_07_MainMachineWasteTankHighLevelAlarm   : BOOL;
	bInternalAlarm_b202_08_ReservedAlarm   : BOOL;
	bInternalAlarm_b202_09_ReservedAlarm   : BOOL;
	bInternalAlarm_b202_10_ReservedAlarm   : BOOL;
	bInternalAlarm_b202_11_ReservedAlarm   : BOOL;

	bInternalAlarm_b203_00_ChillerSelectorOnOffAlarm   : BOOL;
	bInternalAlarm_b203_01_ColdWaterTankLowLevelAlarm   : BOOL;
	bInternalAlarm_b203_02_SludgeTankMissingAlarm   : BOOL;
	bInternalAlarm_b203_03_ColdWaterTankTempHighAlarm   : BOOL;
	bInternalAlarm_b203_04_ColdWaterTankTempNotReadyAlarm   : BOOL;
	bInternalAlarm_b203_05_ColdWaterTankHeaterOnOffAlarm   : BOOL;
	bInternalAlarm_b203_06_ChillerPumpTORAlarm   : BOOL;
	bInternalAlarm_b203_07_ChillerFlowSwitchAlarm   : BOOL;
	bInternalAlarm_b203_08_ChillerInterlockRelayAlarm   : BOOL;
	bInternalAlarm_b203_09_ReservedAlarm   : BOOL;
	bInternalAlarm_b203_10_ThermalOilChangeWarning   : BOOL;
	bInternalAlarm_b203_11_ThermalOilChangeAlarm   : BOOL;



	bInternalInput_b000_00_FreshHCTankCircPumpTOR   : BOOL;
	bInternalInput_b000_01_CircTankCircPumpTOR   : BOOL;
	bInternalInput_b000_02_ThermalOilPumpTOR  : BOOL;
	bInternalInput_b000_03_ThermalOilLevelSensor  : BOOL;
	bInternalInput_b000_04_ThermalOilTempCtrlHighTempAlarmSignal  : BOOL;
	bInternalInput_b000_05_ThermalOilTempCtrlReadySignal  : BOOL;
	bInternalInput_b000_06_ThermalOilTempCtrlOnOffSignal   : BOOL;
	bInternalInput_b000_07_TopDistillatorTempCtrlHighTempAlarmSignal  : BOOL;
	bInternalInput_b000_08_TopDistillatorTempCtrlReadySignal  : BOOL;
	bInternalInput_b000_09_TopDistillatorTempCtrlOnOffSignal   : BOOL;
	bInternalInput_b000_10_RecycleStartStopPB  : BOOL;
	bInternalInput_b000_11_EStopPB  : BOOL;


	bInternalInput_b001_00_PhaseSequenceRelayAlarm  : BOOL;
	bInternalInput_b001_01_ThermalOilUpThermostat   : BOOL;
	bInternalInput_b001_02_SludgeTankLevelSensor  : BOOL;
	bInternalInput_b001_03_FreshHCTankLevelSensor  : BOOL;
	bInternalInput_b001_04_VacuumNotAchieveSignal  : BOOL;
	bInternalInput_b001_05_IncomingCDAPressureSwitch  : BOOL;
	bInternalInput_b001_06_CoolingWaterFlowSwitch  : BOOL;
	bInternalInput_b001_07_CircularTankLevelSensor  : BOOL;
	bInternalInput_b001_08_BottomDistillatorTempCtrlHighTempAlarmSignal  : BOOL;
	bInternalInput_b001_09_BottomDistillatorTempCtrlReadySignal  : BOOL;
	bInternalInput_b001_10_BottomDistillatorTempCtrlOnOffSignal   : BOOL;
	bInternalInput_b001_11_ThermalOilDownThermostat  : BOOL;
	bInternalInput_b001_12_ThermalOilMidThermostat  : BOOL;

	bInternalInput_b002_00_VaporGenerationTempCtrlHighTempAlarmSignal  : BOOL;
	bInternalInput_b002_01_VaporGenerationTempCtrlReadySignal  : BOOL;
	bInternalInput_b002_02_VaporGenerationTempCtrlOnOffSignal  : BOOL;
	bInternalInput_b002_03_WasteCollectionTankLevelSensor  : BOOL;
	bInternalInput_b002_04_VaporGenerationTankLowLevelSensor  : BOOL;
	bInternalInput_b002_05_HCPurgingAV  : BOOL;
	bInternalInput_b002_06_MainMachineWasteCollectTankLowLevelSignal  : BOOL;
	bInternalInput_b002_07_MainMachineWasteCollectTankHighLevelSignal  : BOOL;
	bInternalInput_b002_08_FromMainMachineSignal3  : BOOL;
	bInternalInput_b002_09_FromMainMachineSignal4  : BOOL;
	bInternalInput_b002_10_FromMainMachineSignal5  : BOOL;
	bInternalInput_b002_11_ReservedAlarmSignal  : BOOL;


	bInternalInput_b003_00_ChillerSelectorOnOff  : BOOL;
	bInternalInput_b003_01_ColdWaterTankLowLevelSensor  : BOOL;
	bInternalInput_b003_02_SludgeTankPresentSensor  : BOOL;
	bInternalInput_b003_03_ColdWaterTankTempCtrlHighTempAlarmSignal  : BOOL;
	bInternalInput_b003_04_ColdWaterTankTempCtrlReadySignal  : BOOL;
	bInternalInput_b003_05_ColdWaterTankTempCtrlOnOffSignal  : BOOL;
	bInternalInput_b003_06_ChillerPumpTOR  : BOOL;
	bInternalInput_b003_07_ChillerFlowSwitch  : BOOL;
	bInternalInput_b003_08_ChillerInterlockRelay  : BOOL;
	bInternalInput_b003_09_ReservedAlarmSignal  : BOOL;
	bInternalInput_b003_10_ReservedAlarmSignal  : BOOL;
	bInternalInput_b003_11_ReservedAlarmSignal  : BOOL;


	bInternalOutput_b100_00_FreshHCTankCircPumpOnOff   : BOOL;
	bInternalOutput_b100_01_CircTankCircPumpOnOff  : BOOL;
	bInternalOutput_b100_02_ThermalOilPumpOnOff  : BOOL;
	bInternalOutput_b100_03_ThermalOilHeaterOnOff  : BOOL;
	bInternalOutput_b100_04_Buzzer  : BOOL;
	bInternalOutput_b100_05_RecycleStartStopIndicator  : BOOL;
	bInternalOutput_b100_06_Reserved  : BOOL;
	bInternalOutput_b100_07_UFOVacuumRelease32WayAV  : BOOL;


	bInternalOutput_b101_00_CondenserTankVacuumReleaseAV  : BOOL;
	bInternalOutput_b101_01_WasteSludgeCollectionDrumAV   : BOOL;
	bInternalOutput_b101_02_DistillationTankDrainAV  : BOOL;
	bInternalOutput_b101_03_EconomizerAV  : BOOL;
	bInternalOutput_b101_04_Reserved  : BOOL;
	bInternalOutput_b101_05_Reserved  : BOOL;
	bInternalOutput_b101_06_VaporGenerationAV  : BOOL;
	bInternalOutput_b101_07_VacuumSharingAV  : BOOL;


	bInternalOutput_b102_00_RecycleReadySignal  : BOOL;
	bInternalOutput_b102_01_VaporNotAvailableForRequestSignal  : BOOL;
	bInternalOutput_b102_02_ToMainMachineSignal3  : BOOL;
	bInternalOutput_b102_03_ToMainMachineSignal4  : BOOL;
	bInternalOutput_b102_04_ToMainMachineSignal5  : BOOL;
	bInternalOutput_b102_05_Reserved  : BOOL;
	bInternalOutput_b102_06_Reserved  : BOOL;
	bInternalOutput_b102_07_Reserved  : BOOL;


	bInternalOutput_b103_00_ChillerPumpOnOff  : BOOL;
	bInternalOutput_b103_01_Reserved  : BOOL;
	bInternalOutput_b103_02_Reserved  : BOOL;
	bInternalOutput_b103_03_Reserved  : BOOL;
	bInternalOutput_b103_04_ChillerSelectorOnOffIndicator  : BOOL;
	bInternalOutput_b103_05_ChillerReadySignal  : BOOL;
	bInternalOutput_b103_06_ChillerCompressorOnOff  : BOOL;
	bInternalOutput_b103_07_Reserved  : BOOL;


END_VAR
VAR // added by the converter: edge detectors and wires of the graphical bodies
    _w1, _w3, _w4, _w5, _w6, _w7, _w8, _w9 : ANY;
    _w2 : BOOL;
END_VAR

	(*Timer*)
	t1SecCP(IN:=NOT t1SecCP.Q , PT:=t#1s , Q=> , ET=> );


	(*R_TRIG*)
	t1SecCPRE(CLK:=t1SecCP.Q , Q=> );
	bRecycleStartPBRE(CLK:=bInternalInput_b000_10_RecycleStartStopPB , Q=> );


	(*Sub Program Execution*)
	Z_Mapping();
	Other_LD();
	Other_ST();
	FixOutput_LD();
	OutputCtrl_LD();
	AlarmCtrl_LD();
	BuzzerCtrl_ST();
	MessageDisplayCtrl_ST();
	AutoHCTopUp_LD();
	HighLowLimitCtrl_ST();
	AutoCtrl_LD();
	ManualCtrl_ST();
	
	AutoBoilingCtrl_LD();
	AutoBoilingCtrl_ST();

	ManualBoilingCtrl_LD();
	ManualBoilingCtrl_ST();


	ThermalOilChangeHRMeter_ST();
	ChillerCtrl_LD();
	SystemRestore_LD();
	Z_BuiltInTempCtrl_ST();

	Z_BuiltInVacuumCtrl_ST();

	JRSMachineServiceCtrl_LD();

ACTION AlarmCtrl_LD:
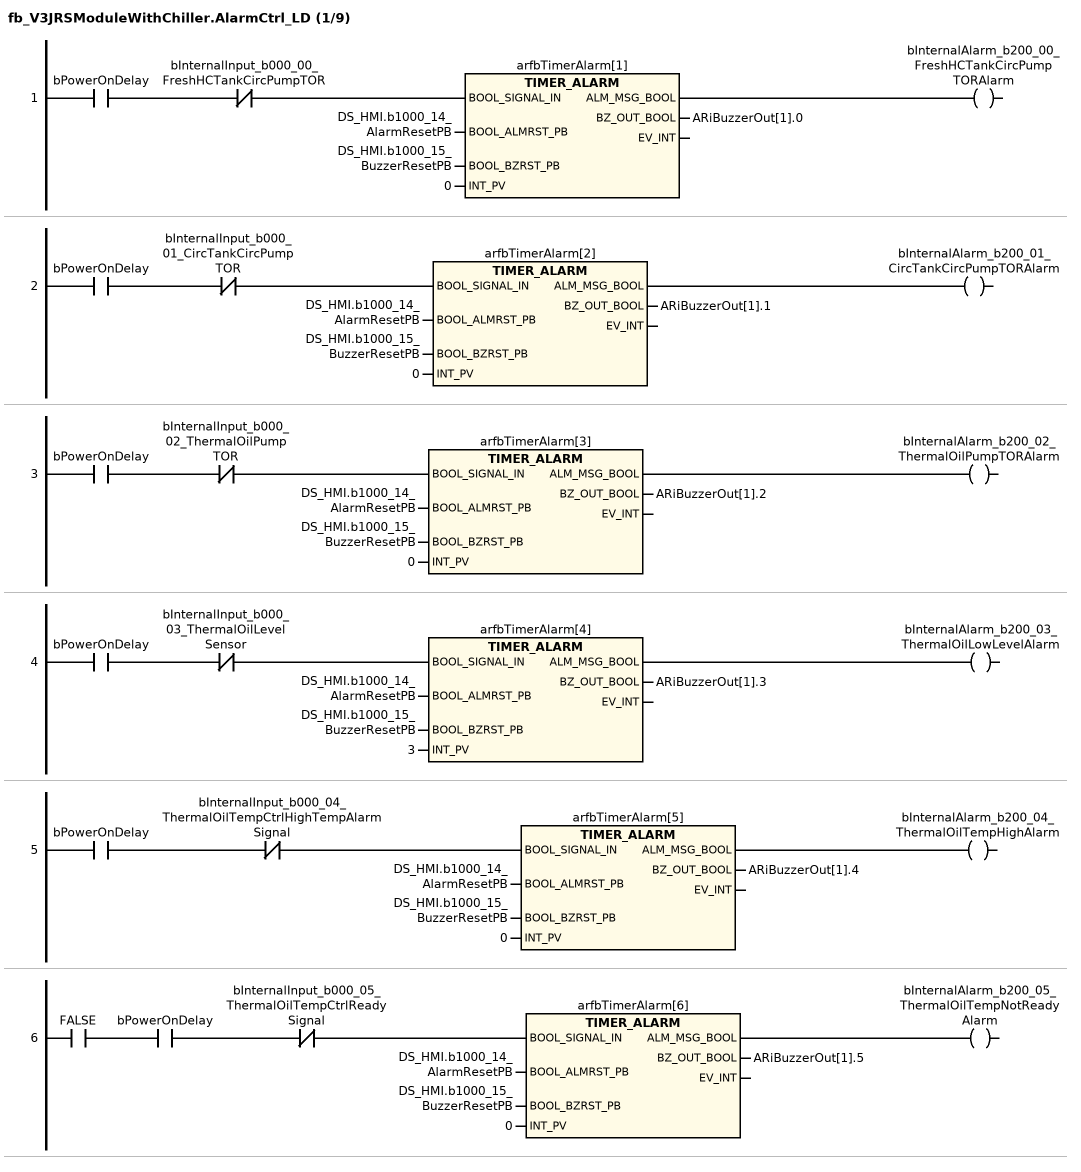
// NETWORK 1
arfbTimerAlarm[1](
    BOOL_SIGNAL_IN := bPowerOnDelay AND NOT bInternalInput_b000_00_FreshHCTankCircPumpTOR,
    BOOL_ALMRST_PB := DS_HMI.b1000_14_AlarmResetPB,
    BOOL_BZRST_PB := DS_HMI.b1000_15_BuzzerResetPB,
    INT_PV := 0,
    BZ_OUT_BOOL => ARiBuzzerOut[1].0); // TIMER_ALARM
bInternalAlarm_b200_00_FreshHCTankCircPumpTORAlarm := arfbTimerAlarm[1].ALM_MSG_BOOL;

// NETWORK 2
arfbTimerAlarm[2](
    BOOL_SIGNAL_IN := bPowerOnDelay AND NOT bInternalInput_b000_01_CircTankCircPumpTOR,
    BOOL_ALMRST_PB := DS_HMI.b1000_14_AlarmResetPB,
    BOOL_BZRST_PB := DS_HMI.b1000_15_BuzzerResetPB,
    INT_PV := 0,
    BZ_OUT_BOOL => ARiBuzzerOut[1].1); // TIMER_ALARM
bInternalAlarm_b200_01_CircTankCircPumpTORAlarm := arfbTimerAlarm[2].ALM_MSG_BOOL;

// NETWORK 3
arfbTimerAlarm[3](
    BOOL_SIGNAL_IN := bPowerOnDelay AND NOT bInternalInput_b000_02_ThermalOilPumpTOR,
    BOOL_ALMRST_PB := DS_HMI.b1000_14_AlarmResetPB,
    BOOL_BZRST_PB := DS_HMI.b1000_15_BuzzerResetPB,
    INT_PV := 0,
    BZ_OUT_BOOL => ARiBuzzerOut[1].2); // TIMER_ALARM
bInternalAlarm_b200_02_ThermalOilPumpTORAlarm := arfbTimerAlarm[3].ALM_MSG_BOOL;

// NETWORK 4
arfbTimerAlarm[4](
    BOOL_SIGNAL_IN := bPowerOnDelay AND NOT bInternalInput_b000_03_ThermalOilLevelSensor,
    BOOL_ALMRST_PB := DS_HMI.b1000_14_AlarmResetPB,
    BOOL_BZRST_PB := DS_HMI.b1000_15_BuzzerResetPB,
    INT_PV := 3,
    BZ_OUT_BOOL => ARiBuzzerOut[1].3); // TIMER_ALARM
bInternalAlarm_b200_03_ThermalOilLowLevelAlarm := arfbTimerAlarm[4].ALM_MSG_BOOL;

// NETWORK 5
arfbTimerAlarm[5](
    BOOL_SIGNAL_IN := bPowerOnDelay AND NOT bInternalInput_b000_04_ThermalOilTempCtrlHighTempAlarmSignal,
    BOOL_ALMRST_PB := DS_HMI.b1000_14_AlarmResetPB,
    BOOL_BZRST_PB := DS_HMI.b1000_15_BuzzerResetPB,
    INT_PV := 0,
    BZ_OUT_BOOL => ARiBuzzerOut[1].4); // TIMER_ALARM
bInternalAlarm_b200_04_ThermalOilTempHighAlarm := arfbTimerAlarm[5].ALM_MSG_BOOL;

// NETWORK 6
arfbTimerAlarm[6](
    BOOL_SIGNAL_IN := FALSE AND bPowerOnDelay AND NOT bInternalInput_b000_05_ThermalOilTempCtrlReadySignal,
    BOOL_ALMRST_PB := DS_HMI.b1000_14_AlarmResetPB,
    BOOL_BZRST_PB := DS_HMI.b1000_15_BuzzerResetPB,
    INT_PV := 0,
    BZ_OUT_BOOL => ARiBuzzerOut[1].5); // TIMER_ALARM
bInternalAlarm_b200_05_ThermalOilTempNotReadyAlarm := arfbTimerAlarm[6].ALM_MSG_BOOL;

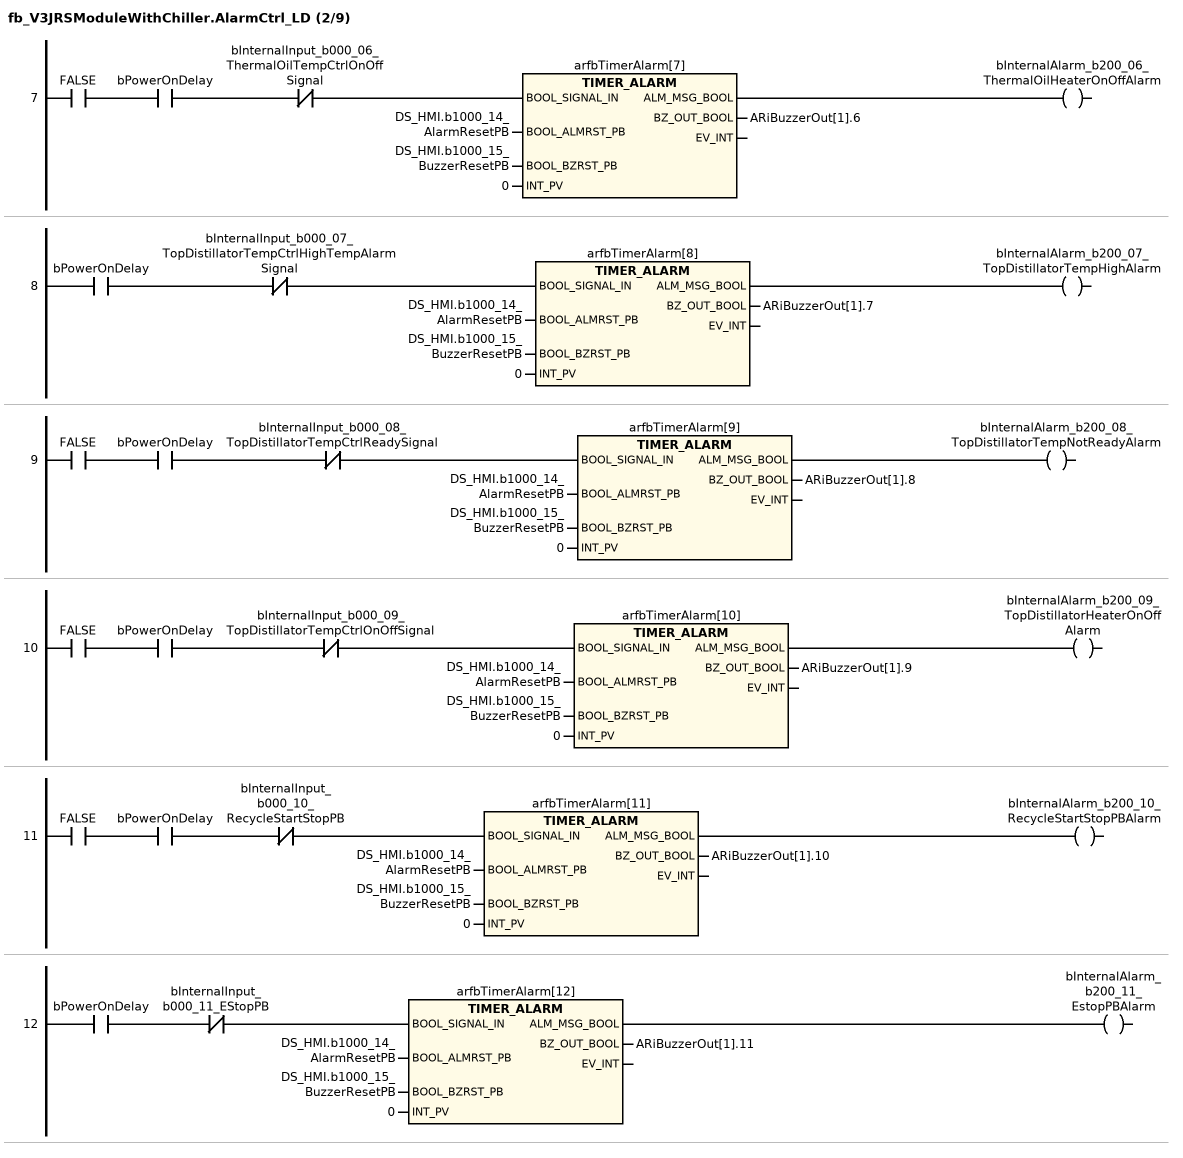
// NETWORK 7
arfbTimerAlarm[7](
    BOOL_SIGNAL_IN := FALSE AND bPowerOnDelay AND NOT bInternalInput_b000_06_ThermalOilTempCtrlOnOffSignal,
    BOOL_ALMRST_PB := DS_HMI.b1000_14_AlarmResetPB,
    BOOL_BZRST_PB := DS_HMI.b1000_15_BuzzerResetPB,
    INT_PV := 0,
    BZ_OUT_BOOL => ARiBuzzerOut[1].6); // TIMER_ALARM
bInternalAlarm_b200_06_ThermalOilHeaterOnOffAlarm := arfbTimerAlarm[7].ALM_MSG_BOOL;

// NETWORK 8
arfbTimerAlarm[8](
    BOOL_SIGNAL_IN := bPowerOnDelay AND NOT bInternalInput_b000_07_TopDistillatorTempCtrlHighTempAlarmSignal,
    BOOL_ALMRST_PB := DS_HMI.b1000_14_AlarmResetPB,
    BOOL_BZRST_PB := DS_HMI.b1000_15_BuzzerResetPB,
    INT_PV := 0,
    BZ_OUT_BOOL => ARiBuzzerOut[1].7); // TIMER_ALARM
bInternalAlarm_b200_07_TopDistillatorTempHighAlarm := arfbTimerAlarm[8].ALM_MSG_BOOL;

// NETWORK 9
arfbTimerAlarm[9](
    BOOL_SIGNAL_IN := FALSE AND bPowerOnDelay AND NOT bInternalInput_b000_08_TopDistillatorTempCtrlReadySignal,
    BOOL_ALMRST_PB := DS_HMI.b1000_14_AlarmResetPB,
    BOOL_BZRST_PB := DS_HMI.b1000_15_BuzzerResetPB,
    INT_PV := 0,
    BZ_OUT_BOOL => ARiBuzzerOut[1].8); // TIMER_ALARM
bInternalAlarm_b200_08_TopDistillatorTempNotReadyAlarm := arfbTimerAlarm[9].ALM_MSG_BOOL;

// NETWORK 10
arfbTimerAlarm[10](
    BOOL_SIGNAL_IN := FALSE AND bPowerOnDelay AND NOT bInternalInput_b000_09_TopDistillatorTempCtrlOnOffSignal,
    BOOL_ALMRST_PB := DS_HMI.b1000_14_AlarmResetPB,
    BOOL_BZRST_PB := DS_HMI.b1000_15_BuzzerResetPB,
    INT_PV := 0,
    BZ_OUT_BOOL => ARiBuzzerOut[1].9); // TIMER_ALARM
bInternalAlarm_b200_09_TopDistillatorHeaterOnOffAlarm := arfbTimerAlarm[10].ALM_MSG_BOOL;

// NETWORK 11
arfbTimerAlarm[11](
    BOOL_SIGNAL_IN := FALSE AND bPowerOnDelay AND NOT bInternalInput_b000_10_RecycleStartStopPB,
    BOOL_ALMRST_PB := DS_HMI.b1000_14_AlarmResetPB,
    BOOL_BZRST_PB := DS_HMI.b1000_15_BuzzerResetPB,
    INT_PV := 0,
    BZ_OUT_BOOL => ARiBuzzerOut[1].10); // TIMER_ALARM
bInternalAlarm_b200_10_RecycleStartStopPBAlarm := arfbTimerAlarm[11].ALM_MSG_BOOL;

// NETWORK 12
arfbTimerAlarm[12](
    BOOL_SIGNAL_IN := bPowerOnDelay AND NOT bInternalInput_b000_11_EStopPB,
    BOOL_ALMRST_PB := DS_HMI.b1000_14_AlarmResetPB,
    BOOL_BZRST_PB := DS_HMI.b1000_15_BuzzerResetPB,
    INT_PV := 0,
    BZ_OUT_BOOL => ARiBuzzerOut[1].11); // TIMER_ALARM
bInternalAlarm_b200_11_EstopPBAlarm := arfbTimerAlarm[12].ALM_MSG_BOOL;

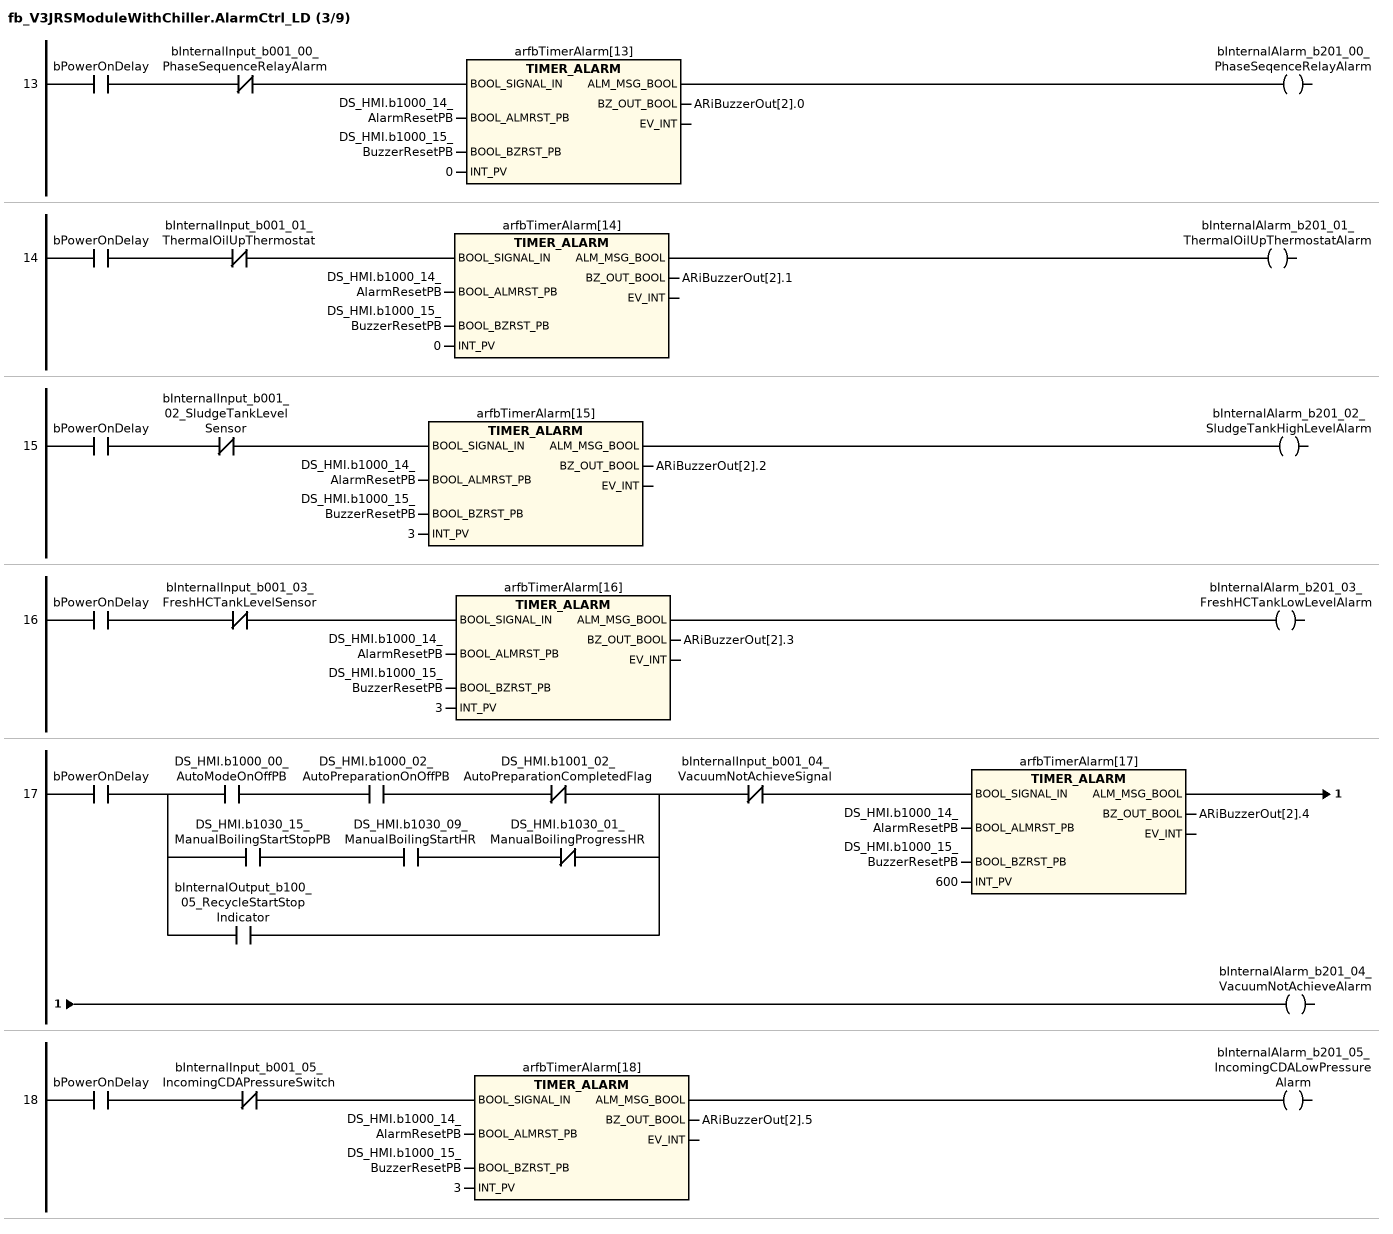
// NETWORK 13
arfbTimerAlarm[13](
    BOOL_SIGNAL_IN := bPowerOnDelay AND NOT bInternalInput_b001_00_PhaseSequenceRelayAlarm,
    BOOL_ALMRST_PB := DS_HMI.b1000_14_AlarmResetPB,
    BOOL_BZRST_PB := DS_HMI.b1000_15_BuzzerResetPB,
    INT_PV := 0,
    BZ_OUT_BOOL => ARiBuzzerOut[2].0); // TIMER_ALARM
bInternalAlarm_b201_00_PhaseSeqenceRelayAlarm := arfbTimerAlarm[13].ALM_MSG_BOOL;

// NETWORK 14
arfbTimerAlarm[14](
    BOOL_SIGNAL_IN := bPowerOnDelay AND NOT bInternalInput_b001_01_ThermalOilUpThermostat,
    BOOL_ALMRST_PB := DS_HMI.b1000_14_AlarmResetPB,
    BOOL_BZRST_PB := DS_HMI.b1000_15_BuzzerResetPB,
    INT_PV := 0,
    BZ_OUT_BOOL => ARiBuzzerOut[2].1); // TIMER_ALARM
bInternalAlarm_b201_01_ThermalOilUpThermostatAlarm := arfbTimerAlarm[14].ALM_MSG_BOOL;

// NETWORK 15
arfbTimerAlarm[15](
    BOOL_SIGNAL_IN := bPowerOnDelay AND NOT bInternalInput_b001_02_SludgeTankLevelSensor,
    BOOL_ALMRST_PB := DS_HMI.b1000_14_AlarmResetPB,
    BOOL_BZRST_PB := DS_HMI.b1000_15_BuzzerResetPB,
    INT_PV := 3,
    BZ_OUT_BOOL => ARiBuzzerOut[2].2); // TIMER_ALARM
bInternalAlarm_b201_02_SludgeTankHighLevelAlarm := arfbTimerAlarm[15].ALM_MSG_BOOL;

// NETWORK 16
arfbTimerAlarm[16](
    BOOL_SIGNAL_IN := bPowerOnDelay AND NOT bInternalInput_b001_03_FreshHCTankLevelSensor,
    BOOL_ALMRST_PB := DS_HMI.b1000_14_AlarmResetPB,
    BOOL_BZRST_PB := DS_HMI.b1000_15_BuzzerResetPB,
    INT_PV := 3,
    BZ_OUT_BOOL => ARiBuzzerOut[2].3); // TIMER_ALARM
bInternalAlarm_b201_03_FreshHCTankLowLevelAlarm := arfbTimerAlarm[16].ALM_MSG_BOOL;

// NETWORK 17
arfbTimerAlarm[17](
    BOOL_SIGNAL_IN := (bPowerOnDelay AND (DS_HMI.b1000_00_AutoModeOnOffPB AND DS_HMI.b1000_02_AutoPreparationOnOffPB AND NOT DS_HMI.b1001_02_AutoPreparationCompletedFlag OR DS_HMI.b1030_15_ManualBoilingStartStopPB AND DS_HMI.b1030_09_ManualBoilingStartHR AND NOT DS_HMI.b1030_01_ManualBoilingProgressHR OR bInternalOutput_b100_05_RecycleStartStopIndicator)) AND NOT bInternalInput_b001_04_VacuumNotAchieveSignal,
    BOOL_ALMRST_PB := DS_HMI.b1000_14_AlarmResetPB,
    BOOL_BZRST_PB := DS_HMI.b1000_15_BuzzerResetPB,
    INT_PV := 600,
    BZ_OUT_BOOL => ARiBuzzerOut[2].4); // TIMER_ALARM
bInternalAlarm_b201_04_VacuumNotAchieveAlarm := arfbTimerAlarm[17].ALM_MSG_BOOL;

// NETWORK 18
arfbTimerAlarm[18](
    BOOL_SIGNAL_IN := bPowerOnDelay AND NOT bInternalInput_b001_05_IncomingCDAPressureSwitch,
    BOOL_ALMRST_PB := DS_HMI.b1000_14_AlarmResetPB,
    BOOL_BZRST_PB := DS_HMI.b1000_15_BuzzerResetPB,
    INT_PV := 3,
    BZ_OUT_BOOL => ARiBuzzerOut[2].5); // TIMER_ALARM
bInternalAlarm_b201_05_IncomingCDALowPressureAlarm := arfbTimerAlarm[18].ALM_MSG_BOOL;

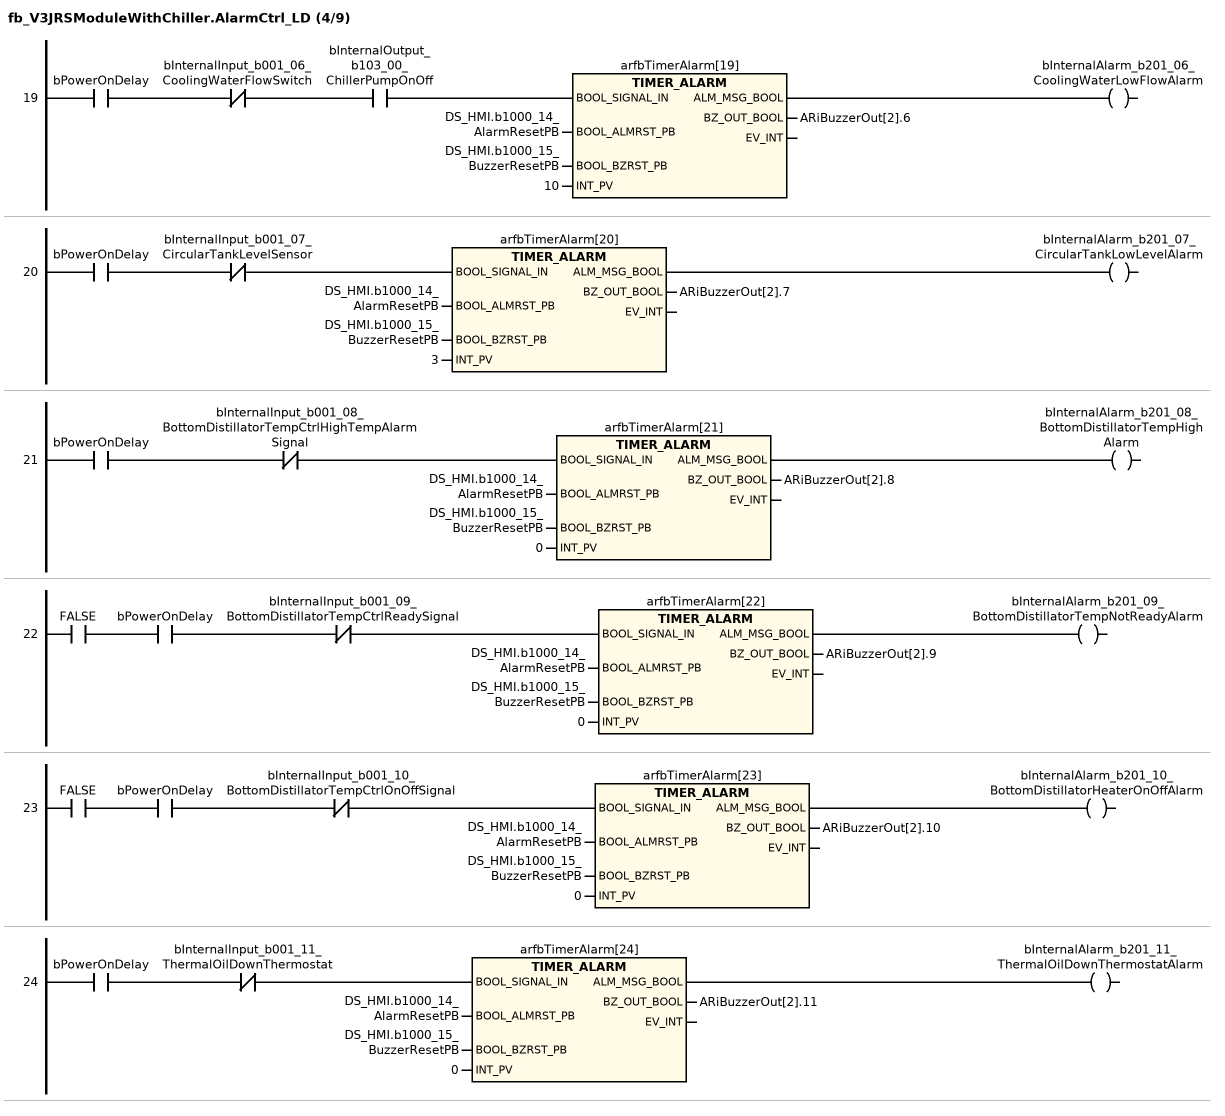
// NETWORK 19
arfbTimerAlarm[19](
    BOOL_SIGNAL_IN := bPowerOnDelay AND NOT bInternalInput_b001_06_CoolingWaterFlowSwitch AND bInternalOutput_b103_00_ChillerPumpOnOff,
    BOOL_ALMRST_PB := DS_HMI.b1000_14_AlarmResetPB,
    BOOL_BZRST_PB := DS_HMI.b1000_15_BuzzerResetPB,
    INT_PV := 10,
    BZ_OUT_BOOL => ARiBuzzerOut[2].6); // TIMER_ALARM
bInternalAlarm_b201_06_CoolingWaterLowFlowAlarm := arfbTimerAlarm[19].ALM_MSG_BOOL;

// NETWORK 20
arfbTimerAlarm[20](
    BOOL_SIGNAL_IN := bPowerOnDelay AND NOT bInternalInput_b001_07_CircularTankLevelSensor,
    BOOL_ALMRST_PB := DS_HMI.b1000_14_AlarmResetPB,
    BOOL_BZRST_PB := DS_HMI.b1000_15_BuzzerResetPB,
    INT_PV := 3,
    BZ_OUT_BOOL => ARiBuzzerOut[2].7); // TIMER_ALARM
bInternalAlarm_b201_07_CircularTankLowLevelAlarm := arfbTimerAlarm[20].ALM_MSG_BOOL;

// NETWORK 21
arfbTimerAlarm[21](
    BOOL_SIGNAL_IN := bPowerOnDelay AND NOT bInternalInput_b001_08_BottomDistillatorTempCtrlHighTempAlarmSignal,
    BOOL_ALMRST_PB := DS_HMI.b1000_14_AlarmResetPB,
    BOOL_BZRST_PB := DS_HMI.b1000_15_BuzzerResetPB,
    INT_PV := 0,
    BZ_OUT_BOOL => ARiBuzzerOut[2].8); // TIMER_ALARM
bInternalAlarm_b201_08_BottomDistillatorTempHighAlarm := arfbTimerAlarm[21].ALM_MSG_BOOL;

// NETWORK 22
arfbTimerAlarm[22](
    BOOL_SIGNAL_IN := FALSE AND bPowerOnDelay AND NOT bInternalInput_b001_09_BottomDistillatorTempCtrlReadySignal,
    BOOL_ALMRST_PB := DS_HMI.b1000_14_AlarmResetPB,
    BOOL_BZRST_PB := DS_HMI.b1000_15_BuzzerResetPB,
    INT_PV := 0,
    BZ_OUT_BOOL => ARiBuzzerOut[2].9); // TIMER_ALARM
bInternalAlarm_b201_09_BottomDistillatorTempNotReadyAlarm := arfbTimerAlarm[22].ALM_MSG_BOOL;

// NETWORK 23
arfbTimerAlarm[23](
    BOOL_SIGNAL_IN := FALSE AND bPowerOnDelay AND NOT bInternalInput_b001_10_BottomDistillatorTempCtrlOnOffSignal,
    BOOL_ALMRST_PB := DS_HMI.b1000_14_AlarmResetPB,
    BOOL_BZRST_PB := DS_HMI.b1000_15_BuzzerResetPB,
    INT_PV := 0,
    BZ_OUT_BOOL => ARiBuzzerOut[2].10); // TIMER_ALARM
bInternalAlarm_b201_10_BottomDistillatorHeaterOnOffAlarm := arfbTimerAlarm[23].ALM_MSG_BOOL;

// NETWORK 24
arfbTimerAlarm[24](
    BOOL_SIGNAL_IN := bPowerOnDelay AND NOT bInternalInput_b001_11_ThermalOilDownThermostat,
    BOOL_ALMRST_PB := DS_HMI.b1000_14_AlarmResetPB,
    BOOL_BZRST_PB := DS_HMI.b1000_15_BuzzerResetPB,
    INT_PV := 0,
    BZ_OUT_BOOL => ARiBuzzerOut[2].11); // TIMER_ALARM
bInternalAlarm_b201_11_ThermalOilDownThermostatAlarm := arfbTimerAlarm[24].ALM_MSG_BOOL;

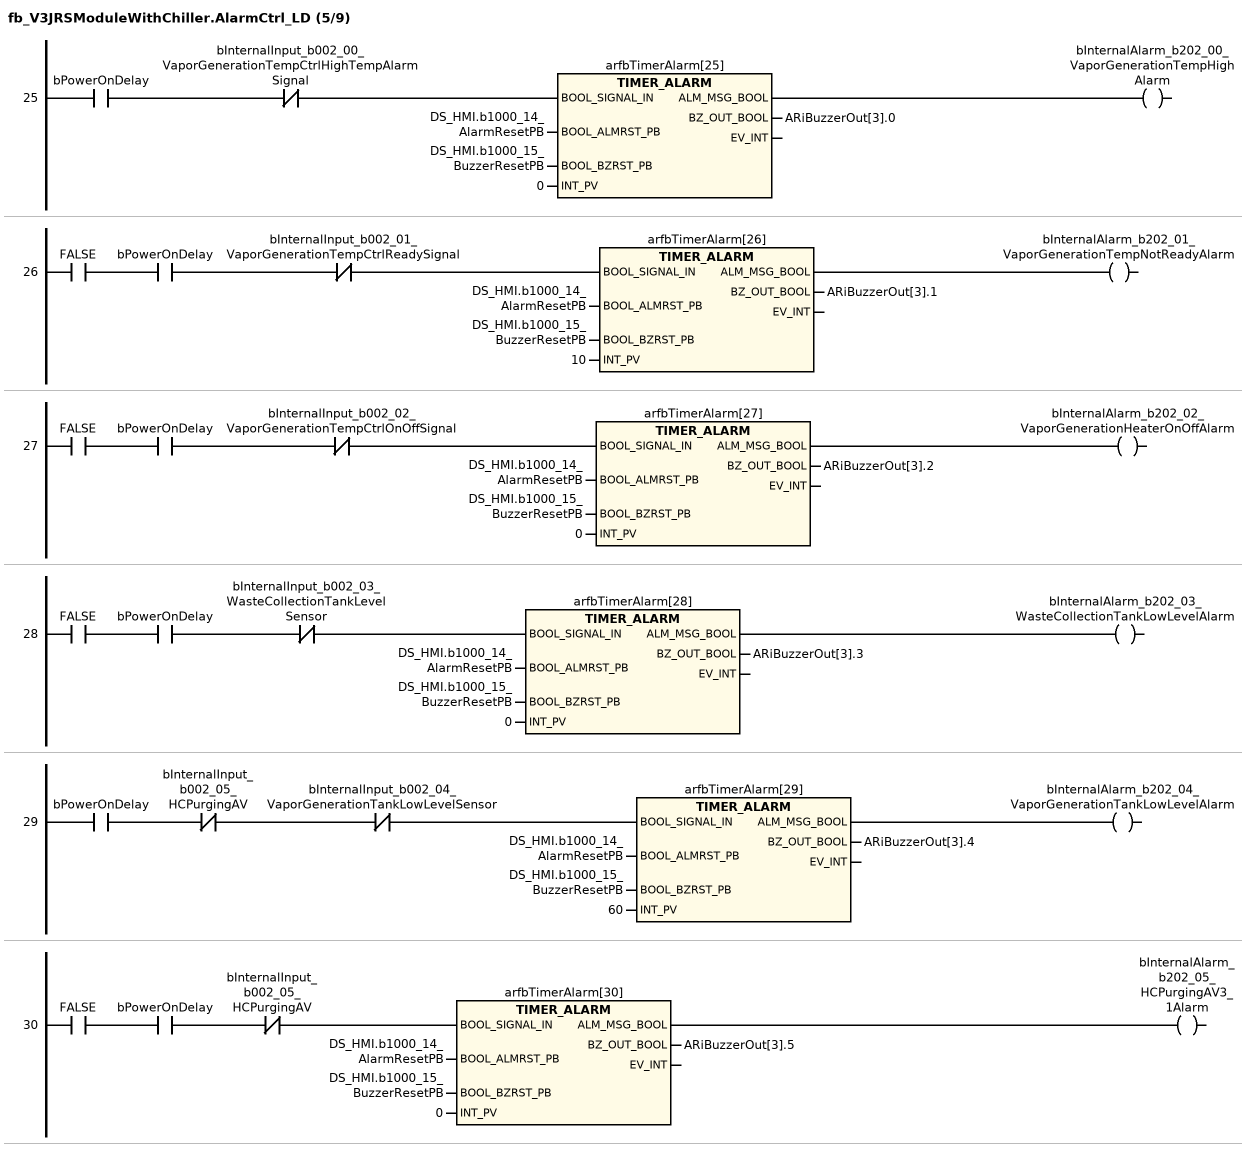
// NETWORK 25
arfbTimerAlarm[25](
    BOOL_SIGNAL_IN := bPowerOnDelay AND NOT bInternalInput_b002_00_VaporGenerationTempCtrlHighTempAlarmSignal,
    BOOL_ALMRST_PB := DS_HMI.b1000_14_AlarmResetPB,
    BOOL_BZRST_PB := DS_HMI.b1000_15_BuzzerResetPB,
    INT_PV := 0,
    BZ_OUT_BOOL => ARiBuzzerOut[3].0); // TIMER_ALARM
bInternalAlarm_b202_00_VaporGenerationTempHighAlarm := arfbTimerAlarm[25].ALM_MSG_BOOL;

// NETWORK 26
arfbTimerAlarm[26](
    BOOL_SIGNAL_IN := FALSE AND bPowerOnDelay AND NOT bInternalInput_b002_01_VaporGenerationTempCtrlReadySignal,
    BOOL_ALMRST_PB := DS_HMI.b1000_14_AlarmResetPB,
    BOOL_BZRST_PB := DS_HMI.b1000_15_BuzzerResetPB,
    INT_PV := 10,
    BZ_OUT_BOOL => ARiBuzzerOut[3].1); // TIMER_ALARM
bInternalAlarm_b202_01_VaporGenerationTempNotReadyAlarm := arfbTimerAlarm[26].ALM_MSG_BOOL;

// NETWORK 27
arfbTimerAlarm[27](
    BOOL_SIGNAL_IN := FALSE AND bPowerOnDelay AND NOT bInternalInput_b002_02_VaporGenerationTempCtrlOnOffSignal,
    BOOL_ALMRST_PB := DS_HMI.b1000_14_AlarmResetPB,
    BOOL_BZRST_PB := DS_HMI.b1000_15_BuzzerResetPB,
    INT_PV := 0,
    BZ_OUT_BOOL => ARiBuzzerOut[3].2); // TIMER_ALARM
bInternalAlarm_b202_02_VaporGenerationHeaterOnOffAlarm := arfbTimerAlarm[27].ALM_MSG_BOOL;

// NETWORK 28
arfbTimerAlarm[28](
    BOOL_SIGNAL_IN := FALSE AND bPowerOnDelay AND NOT bInternalInput_b002_03_WasteCollectionTankLevelSensor,
    BOOL_ALMRST_PB := DS_HMI.b1000_14_AlarmResetPB,
    BOOL_BZRST_PB := DS_HMI.b1000_15_BuzzerResetPB,
    INT_PV := 0,
    BZ_OUT_BOOL => ARiBuzzerOut[3].3); // TIMER_ALARM
bInternalAlarm_b202_03_WasteCollectionTankLowLevelAlarm := arfbTimerAlarm[28].ALM_MSG_BOOL;

// NETWORK 29
arfbTimerAlarm[29](
    BOOL_SIGNAL_IN := bPowerOnDelay AND NOT bInternalInput_b002_05_HCPurgingAV AND NOT bInternalInput_b002_04_VaporGenerationTankLowLevelSensor,
    BOOL_ALMRST_PB := DS_HMI.b1000_14_AlarmResetPB,
    BOOL_BZRST_PB := DS_HMI.b1000_15_BuzzerResetPB,
    INT_PV := 60,
    BZ_OUT_BOOL => ARiBuzzerOut[3].4); // TIMER_ALARM
bInternalAlarm_b202_04_VaporGenerationTankLowLevelAlarm := arfbTimerAlarm[29].ALM_MSG_BOOL;

// NETWORK 30
arfbTimerAlarm[30](
    BOOL_SIGNAL_IN := FALSE AND bPowerOnDelay AND NOT bInternalInput_b002_05_HCPurgingAV,
    BOOL_ALMRST_PB := DS_HMI.b1000_14_AlarmResetPB,
    BOOL_BZRST_PB := DS_HMI.b1000_15_BuzzerResetPB,
    INT_PV := 0,
    BZ_OUT_BOOL => ARiBuzzerOut[3].5); // TIMER_ALARM
bInternalAlarm_b202_05_HCPurgingAV3_1Alarm := arfbTimerAlarm[30].ALM_MSG_BOOL;

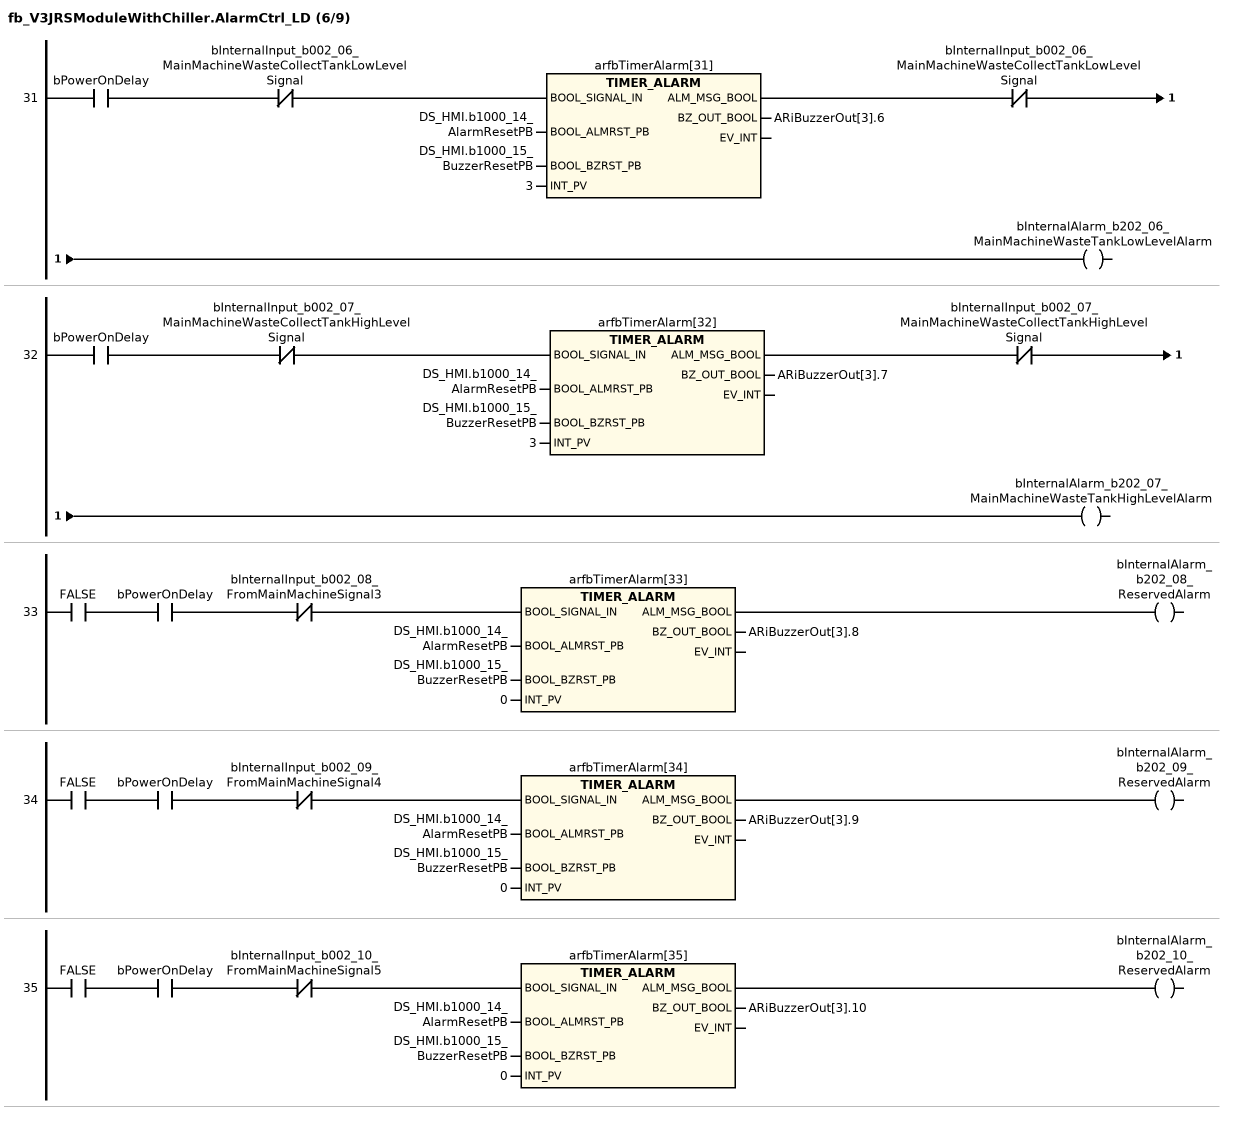
// NETWORK 31
arfbTimerAlarm[31](
    BOOL_SIGNAL_IN := bPowerOnDelay AND NOT bInternalInput_b002_06_MainMachineWasteCollectTankLowLevelSignal,
    BOOL_ALMRST_PB := DS_HMI.b1000_14_AlarmResetPB,
    BOOL_BZRST_PB := DS_HMI.b1000_15_BuzzerResetPB,
    INT_PV := 3,
    BZ_OUT_BOOL => ARiBuzzerOut[3].6); // TIMER_ALARM
bInternalAlarm_b202_06_MainMachineWasteTankLowLevelAlarm := arfbTimerAlarm[31].ALM_MSG_BOOL AND NOT bInternalInput_b002_06_MainMachineWasteCollectTankLowLevelSignal;

// NETWORK 32
arfbTimerAlarm[32](
    BOOL_SIGNAL_IN := bPowerOnDelay AND NOT bInternalInput_b002_07_MainMachineWasteCollectTankHighLevelSignal,
    BOOL_ALMRST_PB := DS_HMI.b1000_14_AlarmResetPB,
    BOOL_BZRST_PB := DS_HMI.b1000_15_BuzzerResetPB,
    INT_PV := 3,
    BZ_OUT_BOOL => ARiBuzzerOut[3].7); // TIMER_ALARM
bInternalAlarm_b202_07_MainMachineWasteTankHighLevelAlarm := arfbTimerAlarm[32].ALM_MSG_BOOL AND NOT bInternalInput_b002_07_MainMachineWasteCollectTankHighLevelSignal;

// NETWORK 33
arfbTimerAlarm[33](
    BOOL_SIGNAL_IN := FALSE AND bPowerOnDelay AND NOT bInternalInput_b002_08_FromMainMachineSignal3,
    BOOL_ALMRST_PB := DS_HMI.b1000_14_AlarmResetPB,
    BOOL_BZRST_PB := DS_HMI.b1000_15_BuzzerResetPB,
    INT_PV := 0,
    BZ_OUT_BOOL => ARiBuzzerOut[3].8); // TIMER_ALARM
bInternalAlarm_b202_08_ReservedAlarm := arfbTimerAlarm[33].ALM_MSG_BOOL;

// NETWORK 34
arfbTimerAlarm[34](
    BOOL_SIGNAL_IN := FALSE AND bPowerOnDelay AND NOT bInternalInput_b002_09_FromMainMachineSignal4,
    BOOL_ALMRST_PB := DS_HMI.b1000_14_AlarmResetPB,
    BOOL_BZRST_PB := DS_HMI.b1000_15_BuzzerResetPB,
    INT_PV := 0,
    BZ_OUT_BOOL => ARiBuzzerOut[3].9); // TIMER_ALARM
bInternalAlarm_b202_09_ReservedAlarm := arfbTimerAlarm[34].ALM_MSG_BOOL;

// NETWORK 35
arfbTimerAlarm[35](
    BOOL_SIGNAL_IN := FALSE AND bPowerOnDelay AND NOT bInternalInput_b002_10_FromMainMachineSignal5,
    BOOL_ALMRST_PB := DS_HMI.b1000_14_AlarmResetPB,
    BOOL_BZRST_PB := DS_HMI.b1000_15_BuzzerResetPB,
    INT_PV := 0,
    BZ_OUT_BOOL => ARiBuzzerOut[3].10); // TIMER_ALARM
bInternalAlarm_b202_10_ReservedAlarm := arfbTimerAlarm[35].ALM_MSG_BOOL;

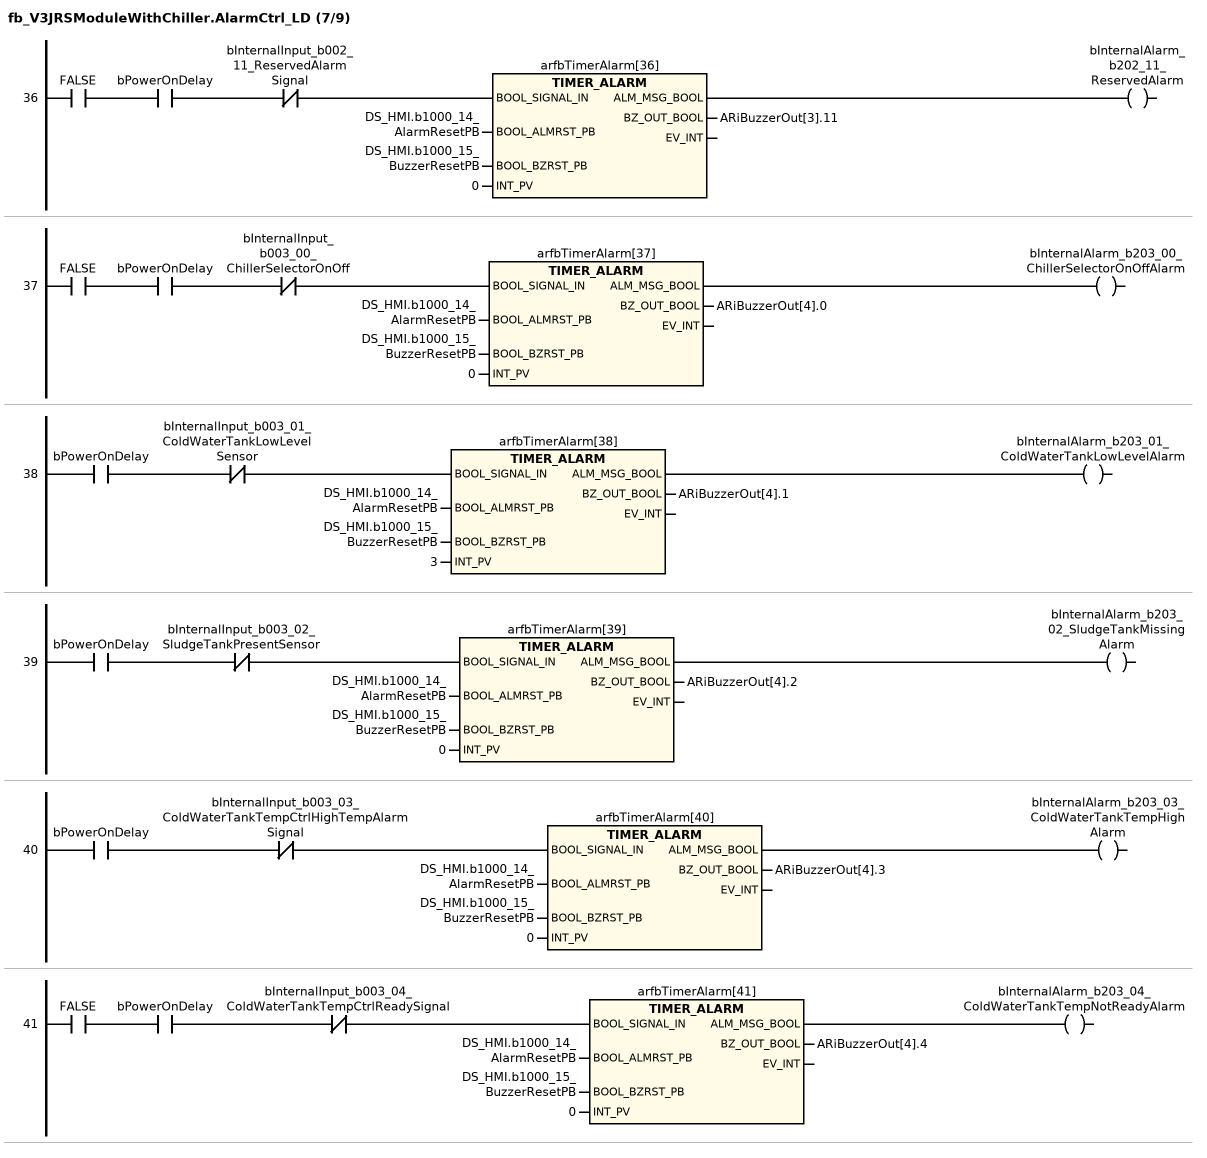
// NETWORK 36
arfbTimerAlarm[36](
    BOOL_SIGNAL_IN := FALSE AND bPowerOnDelay AND NOT bInternalInput_b002_11_ReservedAlarmSignal,
    BOOL_ALMRST_PB := DS_HMI.b1000_14_AlarmResetPB,
    BOOL_BZRST_PB := DS_HMI.b1000_15_BuzzerResetPB,
    INT_PV := 0,
    BZ_OUT_BOOL => ARiBuzzerOut[3].11); // TIMER_ALARM
bInternalAlarm_b202_11_ReservedAlarm := arfbTimerAlarm[36].ALM_MSG_BOOL;

// NETWORK 37
arfbTimerAlarm[37](
    BOOL_SIGNAL_IN := FALSE AND bPowerOnDelay AND NOT bInternalInput_b003_00_ChillerSelectorOnOff,
    BOOL_ALMRST_PB := DS_HMI.b1000_14_AlarmResetPB,
    BOOL_BZRST_PB := DS_HMI.b1000_15_BuzzerResetPB,
    INT_PV := 0,
    BZ_OUT_BOOL => ARiBuzzerOut[4].0); // TIMER_ALARM
bInternalAlarm_b203_00_ChillerSelectorOnOffAlarm := arfbTimerAlarm[37].ALM_MSG_BOOL;

// NETWORK 38
arfbTimerAlarm[38](
    BOOL_SIGNAL_IN := bPowerOnDelay AND NOT bInternalInput_b003_01_ColdWaterTankLowLevelSensor,
    BOOL_ALMRST_PB := DS_HMI.b1000_14_AlarmResetPB,
    BOOL_BZRST_PB := DS_HMI.b1000_15_BuzzerResetPB,
    INT_PV := 3,
    BZ_OUT_BOOL => ARiBuzzerOut[4].1); // TIMER_ALARM
bInternalAlarm_b203_01_ColdWaterTankLowLevelAlarm := arfbTimerAlarm[38].ALM_MSG_BOOL;

// NETWORK 39
arfbTimerAlarm[39](
    BOOL_SIGNAL_IN := bPowerOnDelay AND NOT bInternalInput_b003_02_SludgeTankPresentSensor,
    BOOL_ALMRST_PB := DS_HMI.b1000_14_AlarmResetPB,
    BOOL_BZRST_PB := DS_HMI.b1000_15_BuzzerResetPB,
    INT_PV := 0,
    BZ_OUT_BOOL => ARiBuzzerOut[4].2); // TIMER_ALARM
bInternalAlarm_b203_02_SludgeTankMissingAlarm := arfbTimerAlarm[39].ALM_MSG_BOOL;

// NETWORK 40
arfbTimerAlarm[40](
    BOOL_SIGNAL_IN := bPowerOnDelay AND NOT bInternalInput_b003_03_ColdWaterTankTempCtrlHighTempAlarmSignal,
    BOOL_ALMRST_PB := DS_HMI.b1000_14_AlarmResetPB,
    BOOL_BZRST_PB := DS_HMI.b1000_15_BuzzerResetPB,
    INT_PV := 0,
    BZ_OUT_BOOL => ARiBuzzerOut[4].3); // TIMER_ALARM
bInternalAlarm_b203_03_ColdWaterTankTempHighAlarm := arfbTimerAlarm[40].ALM_MSG_BOOL;

// NETWORK 41
arfbTimerAlarm[41](
    BOOL_SIGNAL_IN := FALSE AND bPowerOnDelay AND NOT bInternalInput_b003_04_ColdWaterTankTempCtrlReadySignal,
    BOOL_ALMRST_PB := DS_HMI.b1000_14_AlarmResetPB,
    BOOL_BZRST_PB := DS_HMI.b1000_15_BuzzerResetPB,
    INT_PV := 0,
    BZ_OUT_BOOL => ARiBuzzerOut[4].4); // TIMER_ALARM
bInternalAlarm_b203_04_ColdWaterTankTempNotReadyAlarm := arfbTimerAlarm[41].ALM_MSG_BOOL;

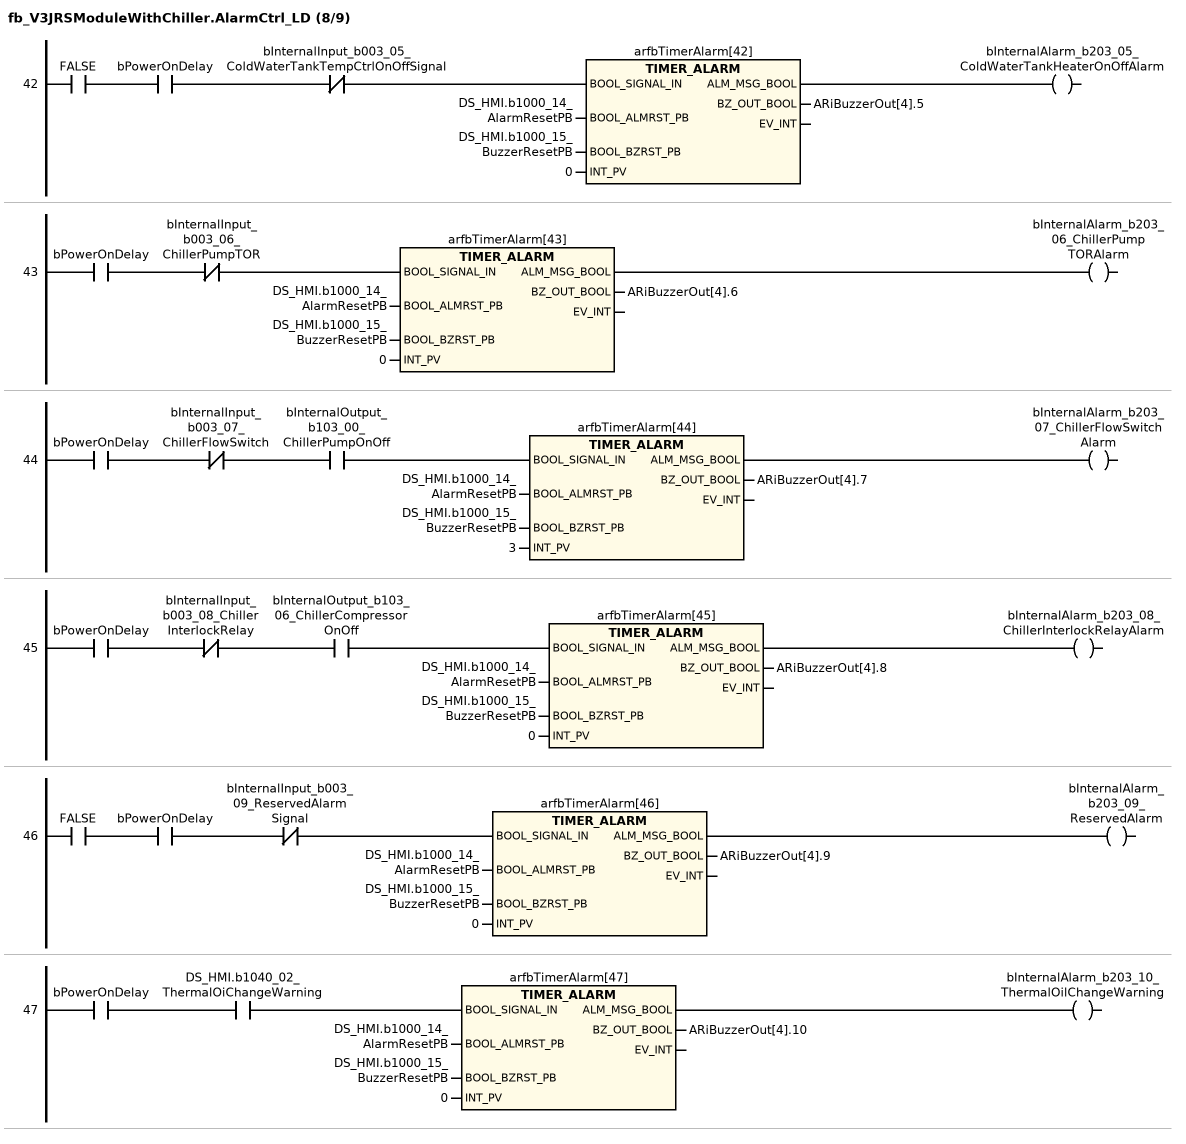
// NETWORK 42
arfbTimerAlarm[42](
    BOOL_SIGNAL_IN := FALSE AND bPowerOnDelay AND NOT bInternalInput_b003_05_ColdWaterTankTempCtrlOnOffSignal,
    BOOL_ALMRST_PB := DS_HMI.b1000_14_AlarmResetPB,
    BOOL_BZRST_PB := DS_HMI.b1000_15_BuzzerResetPB,
    INT_PV := 0,
    BZ_OUT_BOOL => ARiBuzzerOut[4].5); // TIMER_ALARM
bInternalAlarm_b203_05_ColdWaterTankHeaterOnOffAlarm := arfbTimerAlarm[42].ALM_MSG_BOOL;

// NETWORK 43
arfbTimerAlarm[43](
    BOOL_SIGNAL_IN := bPowerOnDelay AND NOT bInternalInput_b003_06_ChillerPumpTOR,
    BOOL_ALMRST_PB := DS_HMI.b1000_14_AlarmResetPB,
    BOOL_BZRST_PB := DS_HMI.b1000_15_BuzzerResetPB,
    INT_PV := 0,
    BZ_OUT_BOOL => ARiBuzzerOut[4].6); // TIMER_ALARM
bInternalAlarm_b203_06_ChillerPumpTORAlarm := arfbTimerAlarm[43].ALM_MSG_BOOL;

// NETWORK 44
arfbTimerAlarm[44](
    BOOL_SIGNAL_IN := bPowerOnDelay AND NOT bInternalInput_b003_07_ChillerFlowSwitch AND bInternalOutput_b103_00_ChillerPumpOnOff,
    BOOL_ALMRST_PB := DS_HMI.b1000_14_AlarmResetPB,
    BOOL_BZRST_PB := DS_HMI.b1000_15_BuzzerResetPB,
    INT_PV := 3,
    BZ_OUT_BOOL => ARiBuzzerOut[4].7); // TIMER_ALARM
bInternalAlarm_b203_07_ChillerFlowSwitchAlarm := arfbTimerAlarm[44].ALM_MSG_BOOL;

// NETWORK 45
arfbTimerAlarm[45](
    BOOL_SIGNAL_IN := bPowerOnDelay AND NOT bInternalInput_b003_08_ChillerInterlockRelay AND bInternalOutput_b103_06_ChillerCompressorOnOff,
    BOOL_ALMRST_PB := DS_HMI.b1000_14_AlarmResetPB,
    BOOL_BZRST_PB := DS_HMI.b1000_15_BuzzerResetPB,
    INT_PV := 0,
    BZ_OUT_BOOL => ARiBuzzerOut[4].8); // TIMER_ALARM
bInternalAlarm_b203_08_ChillerInterlockRelayAlarm := arfbTimerAlarm[45].ALM_MSG_BOOL;

// NETWORK 46
arfbTimerAlarm[46](
    BOOL_SIGNAL_IN := FALSE AND bPowerOnDelay AND NOT bInternalInput_b003_09_ReservedAlarmSignal,
    BOOL_ALMRST_PB := DS_HMI.b1000_14_AlarmResetPB,
    BOOL_BZRST_PB := DS_HMI.b1000_15_BuzzerResetPB,
    INT_PV := 0,
    BZ_OUT_BOOL => ARiBuzzerOut[4].9); // TIMER_ALARM
bInternalAlarm_b203_09_ReservedAlarm := arfbTimerAlarm[46].ALM_MSG_BOOL;

// NETWORK 47
arfbTimerAlarm[47](
    BOOL_SIGNAL_IN := bPowerOnDelay AND DS_HMI.b1040_02_ThermalOiChangeWarning,
    BOOL_ALMRST_PB := DS_HMI.b1000_14_AlarmResetPB,
    BOOL_BZRST_PB := DS_HMI.b1000_15_BuzzerResetPB,
    INT_PV := 0,
    BZ_OUT_BOOL => ARiBuzzerOut[4].10); // TIMER_ALARM
bInternalAlarm_b203_10_ThermalOilChangeWarning := arfbTimerAlarm[47].ALM_MSG_BOOL;

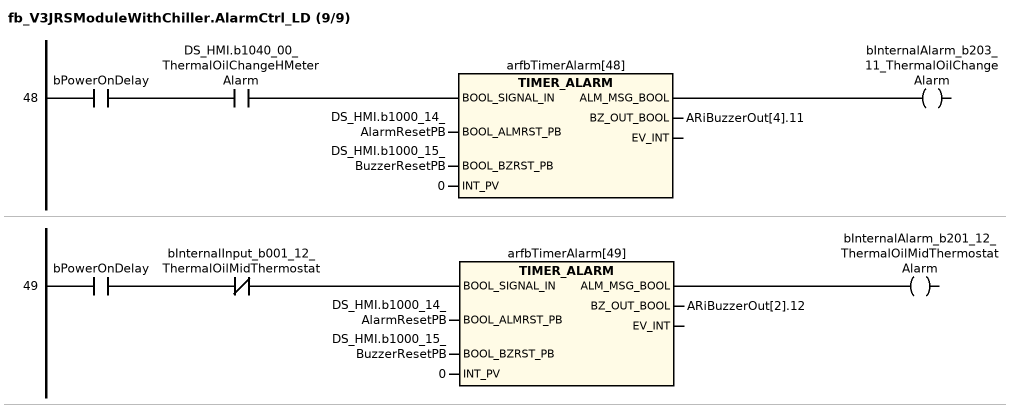
// NETWORK 48
arfbTimerAlarm[48](
    BOOL_SIGNAL_IN := bPowerOnDelay AND DS_HMI.b1040_00_ThermalOilChangeHMeterAlarm,
    BOOL_ALMRST_PB := DS_HMI.b1000_14_AlarmResetPB,
    BOOL_BZRST_PB := DS_HMI.b1000_15_BuzzerResetPB,
    INT_PV := 0,
    BZ_OUT_BOOL => ARiBuzzerOut[4].11); // TIMER_ALARM
bInternalAlarm_b203_11_ThermalOilChangeAlarm := arfbTimerAlarm[48].ALM_MSG_BOOL;

// NETWORK 49
arfbTimerAlarm[49](
    BOOL_SIGNAL_IN := bPowerOnDelay AND NOT bInternalInput_b001_12_ThermalOilMidThermostat,
    BOOL_ALMRST_PB := DS_HMI.b1000_14_AlarmResetPB,
    BOOL_BZRST_PB := DS_HMI.b1000_15_BuzzerResetPB,
    INT_PV := 0,
    BZ_OUT_BOOL => ARiBuzzerOut[2].12); // TIMER_ALARM
bInternalAlarm_b201_12_ThermalOilMidThermostatAlarm := arfbTimerAlarm[49].ALM_MSG_BOOL;
END_ACTION

ACTION AutoBoilingCtrl_LD:
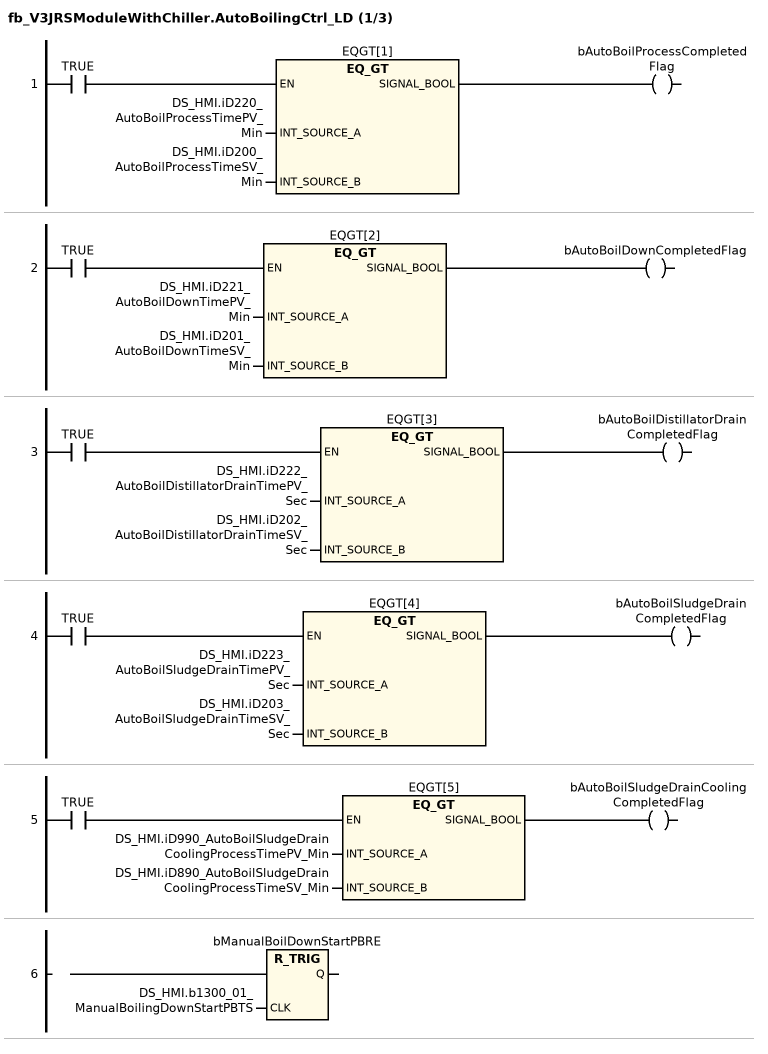
// NETWORK 1
EQGT[1](INT_SOURCE_A := DS_HMI.iD220_AutoBoilProcessTimePV_Min, INT_SOURCE_B := DS_HMI.iD200_AutoBoilProcessTimeSV_Min); // EQ_GT
bAutoBoilProcessCompletedFlag := EQGT[1].SIGNAL_BOOL;

// NETWORK 2
EQGT[2](INT_SOURCE_A := DS_HMI.iD221_AutoBoilDownTimePV_Min, INT_SOURCE_B := DS_HMI.iD201_AutoBoilDownTimeSV_Min); // EQ_GT
bAutoBoilDownCompletedFlag := EQGT[2].SIGNAL_BOOL;

// NETWORK 3
EQGT[3](INT_SOURCE_A := DS_HMI.iD222_AutoBoilDistillatorDrainTimePV_Sec, INT_SOURCE_B := DS_HMI.iD202_AutoBoilDistillatorDrainTimeSV_Sec); // EQ_GT
bAutoBoilDistillatorDrainCompletedFlag := EQGT[3].SIGNAL_BOOL;

// NETWORK 4
EQGT[4](INT_SOURCE_A := DS_HMI.iD223_AutoBoilSludgeDrainTimePV_Sec, INT_SOURCE_B := DS_HMI.iD203_AutoBoilSludgeDrainTimeSV_Sec); // EQ_GT
bAutoBoilSludgeDrainCompletedFlag := EQGT[4].SIGNAL_BOOL;

// NETWORK 5
EQGT[5](INT_SOURCE_A := DS_HMI.iD990_AutoBoilSludgeDrainCoolingProcessTimePV_Min, INT_SOURCE_B := DS_HMI.iD890_AutoBoilSludgeDrainCoolingProcessTimeSV_Min); // EQ_GT
bAutoBoilSludgeDrainCoolingCompletedFlag := EQGT[5].SIGNAL_BOOL;

// NETWORK 6
bManualBoilDownStartPBRE(CLK := DS_HMI.b1300_01_ManualBoilingDownStartPBTS); // R_TRIG

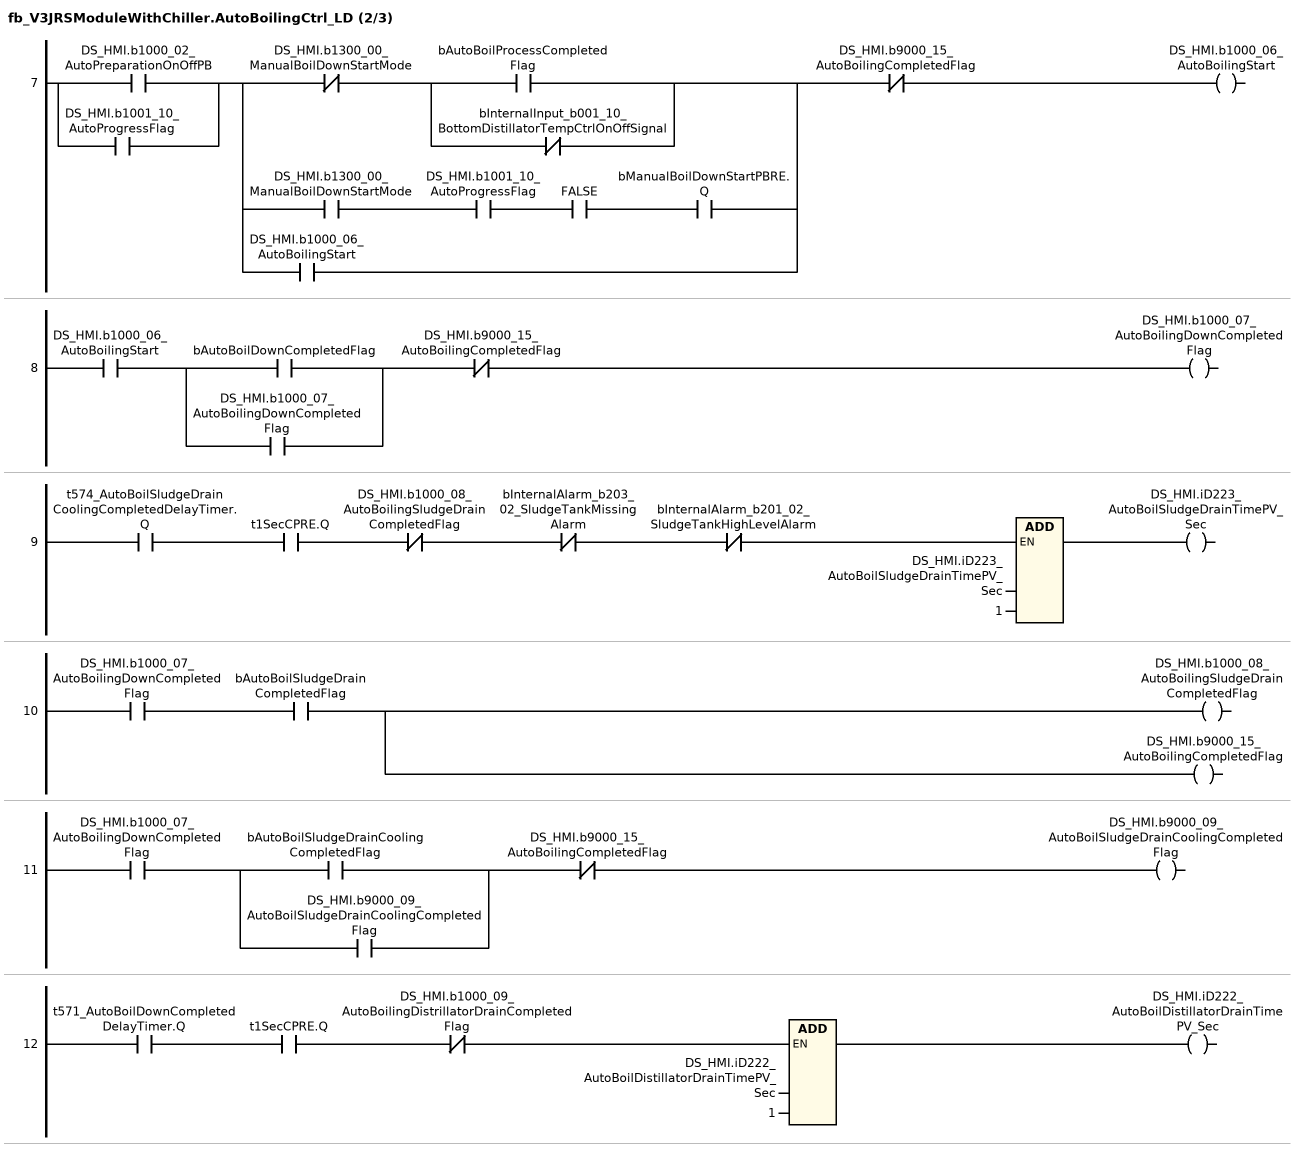
// NETWORK 7
DS_HMI.b1000_06_AutoBoilingStart := ((DS_HMI.b1000_02_AutoPreparationOnOffPB OR DS_HMI.b1001_10_AutoProgressFlag) AND (NOT DS_HMI.b1300_00_ManualBoilDownStartMode AND (bAutoBoilProcessCompletedFlag OR NOT bInternalInput_b001_10_BottomDistillatorTempCtrlOnOffSignal) OR DS_HMI.b1300_00_ManualBoilDownStartMode AND DS_HMI.b1001_10_AutoProgressFlag AND FALSE AND bManualBoilDownStartPBRE.Q OR DS_HMI.b1000_06_AutoBoilingStart)) AND NOT DS_HMI.b9000_15_AutoBoilingCompletedFlag;

// NETWORK 8
DS_HMI.b1000_07_AutoBoilingDownCompletedFlag := (DS_HMI.b1000_06_AutoBoilingStart AND (bAutoBoilDownCompletedFlag OR DS_HMI.b1000_07_AutoBoilingDownCompletedFlag)) AND NOT DS_HMI.b9000_15_AutoBoilingCompletedFlag;

// NETWORK 9
IF t574_AutoBoilSludgeDrainCoolingCompletedDelayTimer.Q AND t1SecCPRE.Q AND NOT DS_HMI.b1000_08_AutoBoilingSludgeDrainCompletedFlag AND NOT bInternalAlarm_b203_02_SludgeTankMissingAlarm AND NOT bInternalAlarm_b201_02_SludgeTankHighLevelAlarm THEN
    _w1 := DS_HMI.iD223_AutoBoilSludgeDrainTimePV_Sec + 1;
END_IF
DS_HMI.iD223_AutoBoilSludgeDrainTimePV_Sec := _w1;

// NETWORK 10
_w2 := DS_HMI.b1000_07_AutoBoilingDownCompletedFlag AND bAutoBoilSludgeDrainCompletedFlag;
DS_HMI.b1000_08_AutoBoilingSludgeDrainCompletedFlag := _w2;
DS_HMI.b9000_15_AutoBoilingCompletedFlag := _w2;

// NETWORK 11
DS_HMI.b9000_09_AutoBoilSludgeDrainCoolingCompletedFlag := (DS_HMI.b1000_07_AutoBoilingDownCompletedFlag AND (bAutoBoilSludgeDrainCoolingCompletedFlag OR DS_HMI.b9000_09_AutoBoilSludgeDrainCoolingCompletedFlag)) AND NOT DS_HMI.b9000_15_AutoBoilingCompletedFlag;

// NETWORK 12
IF t571_AutoBoilDownCompletedDelayTimer.Q AND t1SecCPRE.Q AND NOT DS_HMI.b1000_09_AutoBoilingDistrillatorDrainCompletedFlag THEN
    _w3 := DS_HMI.iD222_AutoBoilDistillatorDrainTimePV_Sec + 1;
END_IF
DS_HMI.iD222_AutoBoilDistillatorDrainTimePV_Sec := _w3;

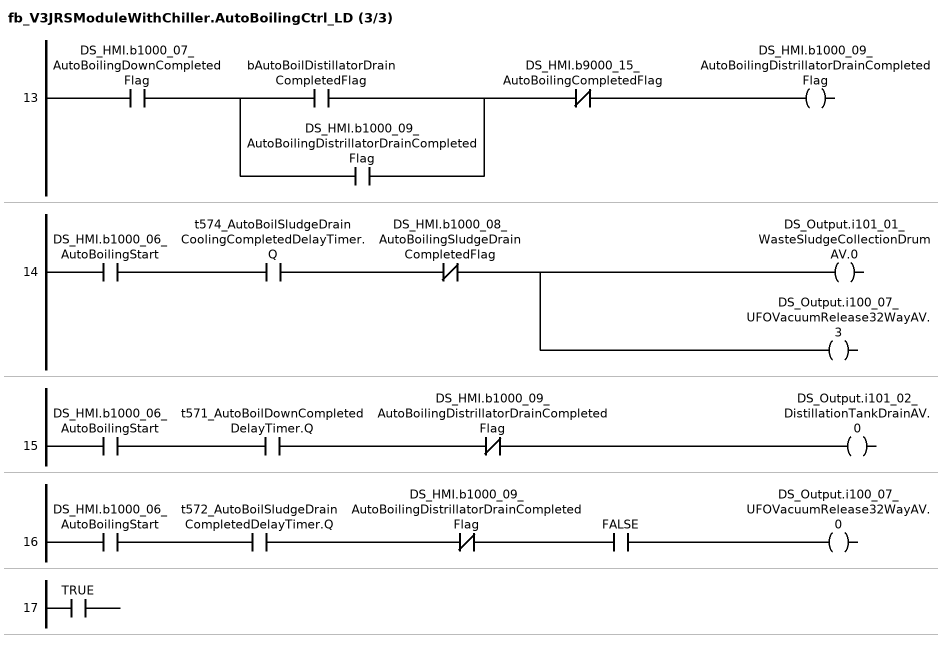
// NETWORK 13
DS_HMI.b1000_09_AutoBoilingDistrillatorDrainCompletedFlag := (DS_HMI.b1000_07_AutoBoilingDownCompletedFlag AND (bAutoBoilDistillatorDrainCompletedFlag OR DS_HMI.b1000_09_AutoBoilingDistrillatorDrainCompletedFlag)) AND NOT DS_HMI.b9000_15_AutoBoilingCompletedFlag;

// NETWORK 14
_w4 := DS_HMI.b1000_06_AutoBoilingStart AND t574_AutoBoilSludgeDrainCoolingCompletedDelayTimer.Q AND NOT DS_HMI.b1000_08_AutoBoilingSludgeDrainCompletedFlag;
DS_Output.i101_01_WasteSludgeCollectionDrumAV.0 := _w4;
DS_Output.i100_07_UFOVacuumRelease32WayAV.3 := _w4;

// NETWORK 15
DS_Output.i101_02_DistillationTankDrainAV.0 := DS_HMI.b1000_06_AutoBoilingStart AND t571_AutoBoilDownCompletedDelayTimer.Q AND NOT DS_HMI.b1000_09_AutoBoilingDistrillatorDrainCompletedFlag;

// NETWORK 16
DS_Output.i100_07_UFOVacuumRelease32WayAV.0 := DS_HMI.b1000_06_AutoBoilingStart AND t572_AutoBoilSludgeDrainCompletedDelayTimer.Q AND NOT DS_HMI.b1000_09_AutoBoilingDistrillatorDrainCompletedFlag AND FALSE;

// NETWORK 17
END_ACTION

ACTION AutoBoilingCtrl_ST:
	(*Timer*)
	t570_AutoBoilingStartDelayTimer(IN:=DS_HMI.b1000_06_AutoBoilingStart , PT:=t#1s , Q=> , ET=> );
	t571_AutoBoilDownCompletedDelayTimer(IN:=DS_HMI.b1000_07_AutoBoilingDownCompletedFlag , PT:=t#1s , Q=> , ET=> );
	t572_AutoBoilSludgeDrainCompletedDelayTimer(IN:=DS_HMI.b1000_08_AutoBoilingSludgeDrainCompletedFlag , PT:=t#1s , Q=> , ET=> );
	t573_AutoBoilDistillatorDrainCompletedDelayTimer(IN:=DS_HMI.b1000_09_AutoBoilingDistrillatorDrainCompletedFlag , PT:=t#1s , Q=> , ET=> );

	t574_AutoBoilSludgeDrainCoolingCompletedDelayTimer(IN:=DS_HMI.b9000_09_AutoBoilSludgeDrainCoolingCompletedFlag , PT:=t#1s , Q=> , ET=> );  (************* New extra request by customer - YCH************)


	(*AutoBoiling Boil Process Time Counting*)
	IF DS_HMI.b1001_10_AutoProgressFlag
	AND NOT DS_HMI.b1300_00_ManualBoilDownStartMode
	AND t1SecCPRE.Q
	THEN

		IF NOT DS_HMI.b1000_06_AutoBoilingStart THEN

			DS_HMI.iD225_AutoBoilProcessTimePV_Sec := DS_HMI.iD225_AutoBoilProcessTimePV_Sec + 1;

			IF DS_HMI.iD225_AutoBoilProcessTimePV_Sec > 59 THEN
				DS_HMI.iD220_AutoBoilProcessTimePV_Min := DS_HMI.iD220_AutoBoilProcessTimePV_Min + 1;
				DS_HMI.iD225_AutoBoilProcessTimePV_Sec := 0;
			END_IF

		END_IF

	END_IF

	(*AutoBoiling Boil Down Time Counting*)

	IF t570_AutoBoilingStartDelayTimer.Q
	AND t1SecCPRE.Q
	THEN

		IF NOT DS_HMI.b1000_07_AutoBoilingDownCompletedFlag THEN

			DS_HMI.iD226_AutoBoilDownTimePV_Sec := DS_HMI.iD226_AutoBoilDownTimePV_Sec + 1;

			IF DS_HMI.iD226_AutoBoilDownTimePV_Sec > 59 THEN
				DS_HMI.iD221_AutoBoilDownTimePV_Min := DS_HMI.iD221_AutoBoilDownTimePV_Min + 1;
				DS_HMI.iD226_AutoBoilDownTimePV_Sec := 0;
			END_IF

		END_IF

	END_IF


	(*AutoBoiling Sludge Drain Cooling Time Counting*)       (************* New extra request by customer - YCH************)

	IF t573_AutoBoilDistillatorDrainCompletedDelayTimer.Q
	AND t1SecCPRE.Q
	THEN

		IF NOT DS_HMI.b9000_09_AutoBoilSludgeDrainCoolingCompletedFlag THEN

			DS_HMI.iD991_AutoBoilSludgeDrainCoolingProcessTimePV_Sec := DS_HMI.iD991_AutoBoilSludgeDrainCoolingProcessTimePV_Sec + 1;

			IF DS_HMI.iD991_AutoBoilSludgeDrainCoolingProcessTimePV_Sec > 59 THEN
				DS_HMI.iD990_AutoBoilSludgeDrainCoolingProcessTimePV_Min := DS_HMI.iD990_AutoBoilSludgeDrainCoolingProcessTimePV_Min + 1;
				DS_HMI.iD991_AutoBoilSludgeDrainCoolingProcessTimePV_Sec := 0;
			END_IF

		END_IF

	END_IF


	(*Auto Boiling Reset*)
	IF DS_HMI.b9000_15_AutoBoilingCompletedFlag OR  t592_ManualBoilSludgeDrainCompletedDelayTimer.Q (*t572_AutoBoilSludgeDrainCompletedDelayTimer.Q*) THEN
	
		DS_HMI.iD220_AutoBoilProcessTimePV_Min						:= 0;
		DS_HMI.iD221_AutoBoilDownTimePV_Min						:= 0;
		DS_HMI.iD990_AutoBoilSludgeDrainCoolingProcessTimePV_Min 	:= 0; (************* New extra request by customer - YCH************)
		DS_HMI.iD222_AutoBoilDistillatorDrainTimePV_Sec				:= 0;
		DS_HMI.iD223_AutoBoilSludgeDrainTimePV_Sec					:= 0;
		DS_HMI.iD225_AutoBoilProcessTimePV_Sec						:= 0;
		DS_HMI.iD226_AutoBoilDownTimePV_Sec						:= 0;
		DS_HMI.iD991_AutoBoilSludgeDrainCoolingProcessTimePV_Sec 	:= 0; (************* New extra request by customer - YCH************)

		DS_HMI.b1300_01_ManualBoilingDownStartPBTS 			:= FALSE;

	END_IF

	IF NOT DS_HMI.b1300_00_ManualBoilDownStartMode THEN
		DS_HMI.b1300_01_ManualBoilingDownStartPBTS 			:= FALSE;
	END_IF
END_ACTION

ACTION AutoCtrl_LD:
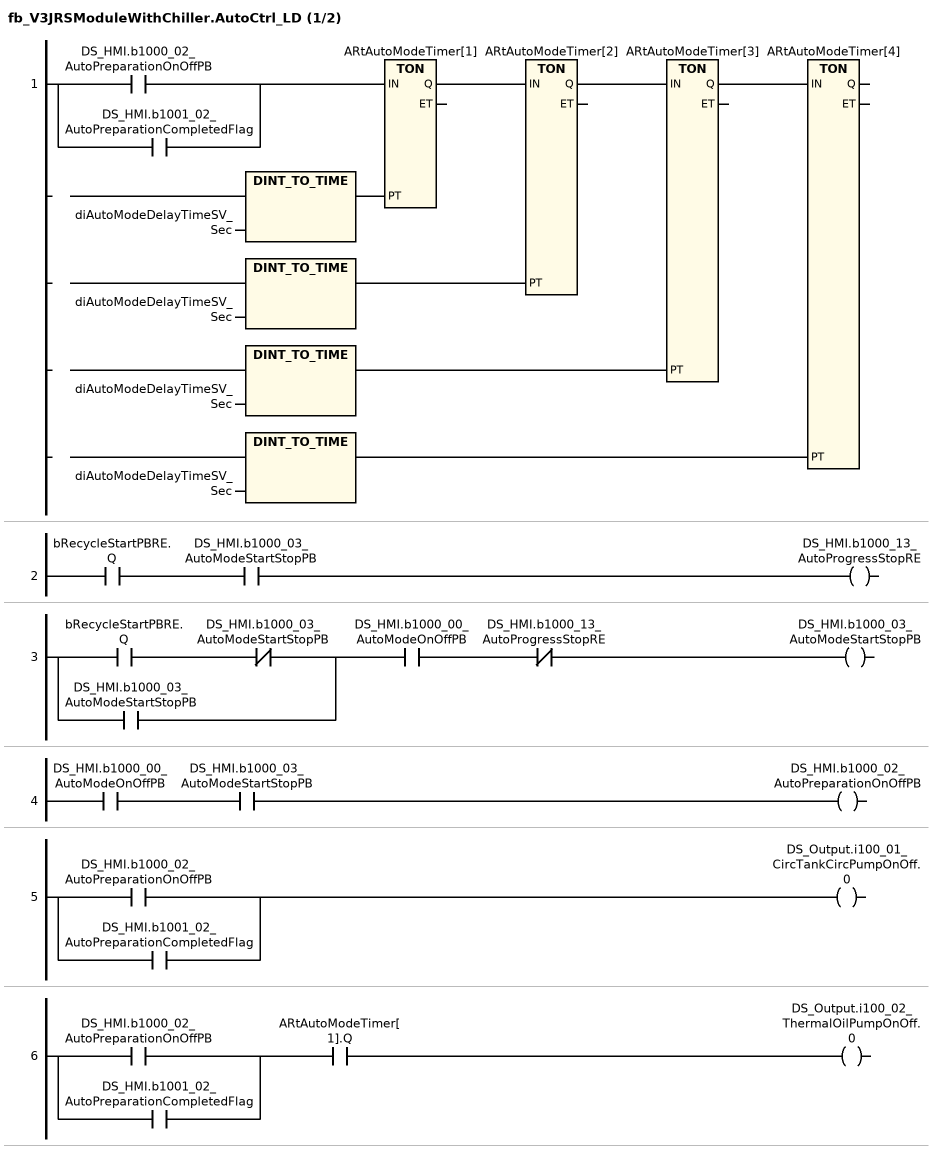
// NETWORK 1
ARtAutoModeTimer[1](IN := DS_HMI.b1000_02_AutoPreparationOnOffPB OR DS_HMI.b1001_02_AutoPreparationCompletedFlag, PT := DINT_TO_TIME(diAutoModeDelayTimeSV_Sec)); // TON
ARtAutoModeTimer[2](IN := ARtAutoModeTimer[1].Q, PT := DINT_TO_TIME(diAutoModeDelayTimeSV_Sec)); // TON
ARtAutoModeTimer[3](IN := ARtAutoModeTimer[2].Q, PT := DINT_TO_TIME(diAutoModeDelayTimeSV_Sec)); // TON
ARtAutoModeTimer[4](IN := ARtAutoModeTimer[3].Q, PT := DINT_TO_TIME(diAutoModeDelayTimeSV_Sec)); // TON

// NETWORK 2
DS_HMI.b1000_13_AutoProgressStopRE := bRecycleStartPBRE.Q AND DS_HMI.b1000_03_AutoModeStartStopPB;

// NETWORK 3
DS_HMI.b1000_03_AutoModeStartStopPB := (bRecycleStartPBRE.Q AND NOT DS_HMI.b1000_03_AutoModeStartStopPB OR DS_HMI.b1000_03_AutoModeStartStopPB) AND DS_HMI.b1000_00_AutoModeOnOffPB AND NOT DS_HMI.b1000_13_AutoProgressStopRE;

// NETWORK 4
DS_HMI.b1000_02_AutoPreparationOnOffPB := DS_HMI.b1000_00_AutoModeOnOffPB AND DS_HMI.b1000_03_AutoModeStartStopPB;

// NETWORK 5
DS_Output.i100_01_CircTankCircPumpOnOff.0 := DS_HMI.b1000_02_AutoPreparationOnOffPB OR DS_HMI.b1001_02_AutoPreparationCompletedFlag;

// NETWORK 6
DS_Output.i100_02_ThermalOilPumpOnOff.0 := (DS_HMI.b1000_02_AutoPreparationOnOffPB OR DS_HMI.b1001_02_AutoPreparationCompletedFlag) AND ARtAutoModeTimer[1].Q;

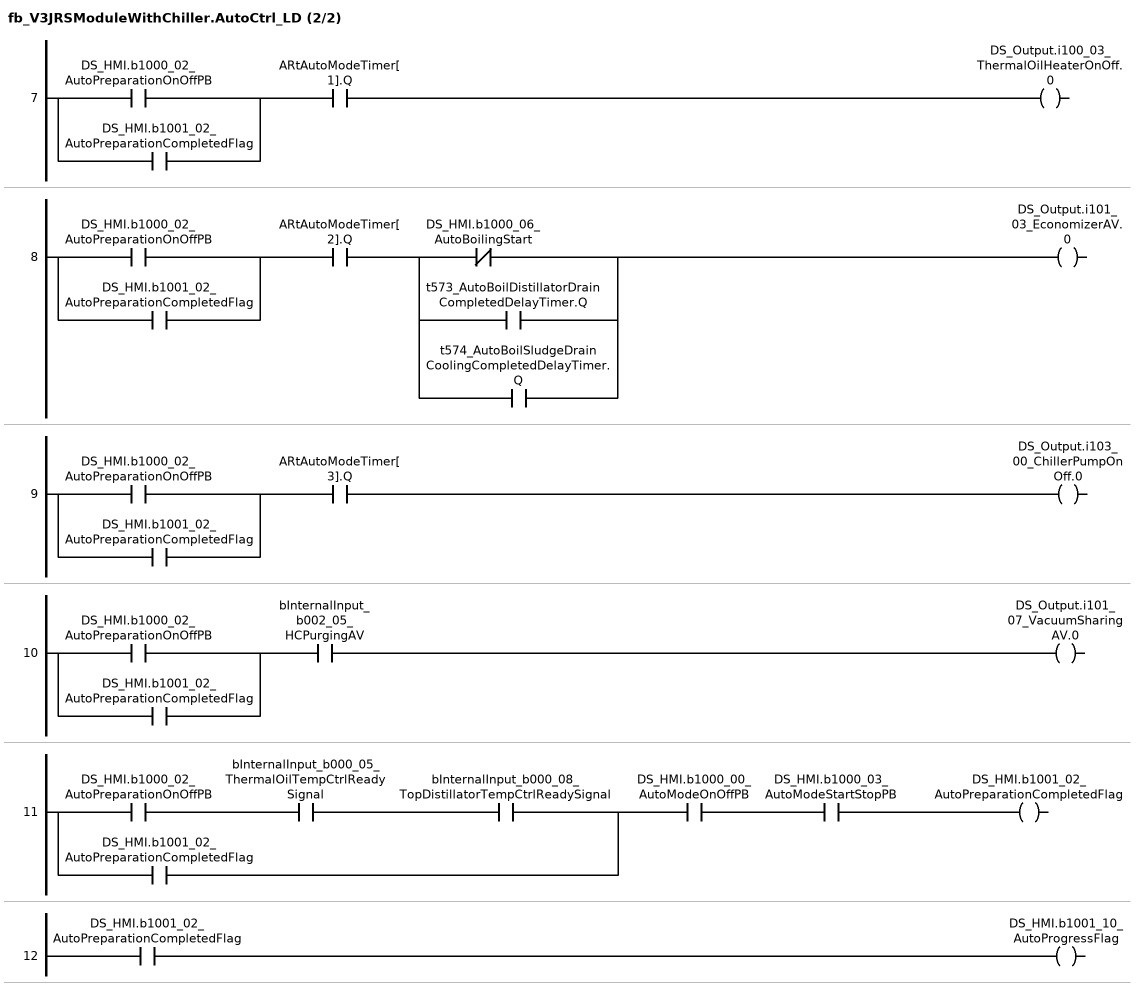
// NETWORK 7
DS_Output.i100_03_ThermalOilHeaterOnOff.0 := (DS_HMI.b1000_02_AutoPreparationOnOffPB OR DS_HMI.b1001_02_AutoPreparationCompletedFlag) AND ARtAutoModeTimer[1].Q;

// NETWORK 8
DS_Output.i101_03_EconomizerAV.0 := (DS_HMI.b1000_02_AutoPreparationOnOffPB OR DS_HMI.b1001_02_AutoPreparationCompletedFlag) AND ARtAutoModeTimer[2].Q AND (NOT DS_HMI.b1000_06_AutoBoilingStart OR t573_AutoBoilDistillatorDrainCompletedDelayTimer.Q OR t574_AutoBoilSludgeDrainCoolingCompletedDelayTimer.Q);

// NETWORK 9
DS_Output.i103_00_ChillerPumpOnOff.0 := (DS_HMI.b1000_02_AutoPreparationOnOffPB OR DS_HMI.b1001_02_AutoPreparationCompletedFlag) AND ARtAutoModeTimer[3].Q;

// NETWORK 10
DS_Output.i101_07_VacuumSharingAV.0 := (DS_HMI.b1000_02_AutoPreparationOnOffPB OR DS_HMI.b1001_02_AutoPreparationCompletedFlag) AND bInternalInput_b002_05_HCPurgingAV;

